// TIA Portal V17 export
// export: Created 2025-03-13T10:29:33.9206583Z, ExportSetting WithDefaults, DisplayName Totally Integrated Automation Portal, DisplayVersion V17 Update 8, DisplayName TIA Portal Openness, DisplayVersion V17 Update 8, DisplayName TIA Portal Version Control Interface, DisplayVersion V17, DisplayName SINAMICS Startdrive Advanced, DisplayVersion V17 SP2, DisplayName SINAMICS Startdrive G110M, G120, G120C, G120D, G120P, G115D, DisplayVersion V17 SP2, DisplayName SINAMICS Startdrive G130, G150, S120, S150, SINAMICS MV, S210, DisplayVersion V17 SP2, DisplayName STEP 7 Professional, DisplayVersion V17 Update 8, DisplayName SINUMERIK ONE STEP 7 Toolbox, DisplayVersion V17 Update 12, DisplayName SINUMERIK 840D sl STEP 7 Toolbox, DisplayVersion V17 Update 12, DisplayName STEP 7 Safety, DisplayVersion V17 Update 6, DisplayName WinCC Advanced, DisplayVersion V17 Update 8
FUNCTION_BLOCK "FB1013_SAFETY_CLADDING"   // FB1013, F_LAD
{ S7_Optimized_Access := 'TRUE' }
AUTHOR : ETXETAR
VERSION : 1.0
// stored: AutoNumber false, IsIECCheckEnabled false, UDAEnableTagReadback false
   VAR
      F_IEC_Timer_PWR_EN_DEL_2 : TOF;
      F_IEC_Timer_PWR_EN_DEL_3 : TOF;
      F_IEC_Timer_PWR_EN_DEL_4 : TOF;
      F_IEC_Timer_PWR_EN_RES_DEL : TON;
      F_IEC_Timer_PWR_EN_FDBCK : TON;
      F_IEC_Timer_GNTR_DR_FDBCK : TON;
      F_IEC_Timer_FIXT_WRK_COND_FDBCK : TON;
      F_IEC_Timer_MACHINE_E_STOP : TON;
      F_IEC_Timer_CLNT_OFF_01R : TOF;
      F_IEC_Timer_CLNT_OFF_01L : TOF;
      F_IEC_Timer_BIMANUAL_CLOSE : TON;
   END_VAR
   // F_IEC_Timer_PWR_EN_FDBCK.PT := T#30ms;
   // F_IEC_Timer_GNTR_DR_FDBCK.PT := T#30ms;
   // F_IEC_Timer_FIXT_WRK_COND_FDBCK.PT := T#30ms;
   // F_IEC_Timer_MACHINE_E_STOP.PT := T#30ms;
   // F_IEC_Timer_BIMANUAL_CLOSE.PT := T#30ms;
BEGIN

REGION Network 1: *************** EMERGENCY STOP ***************
END_REGION

REGION Network 2: FB E-STOP
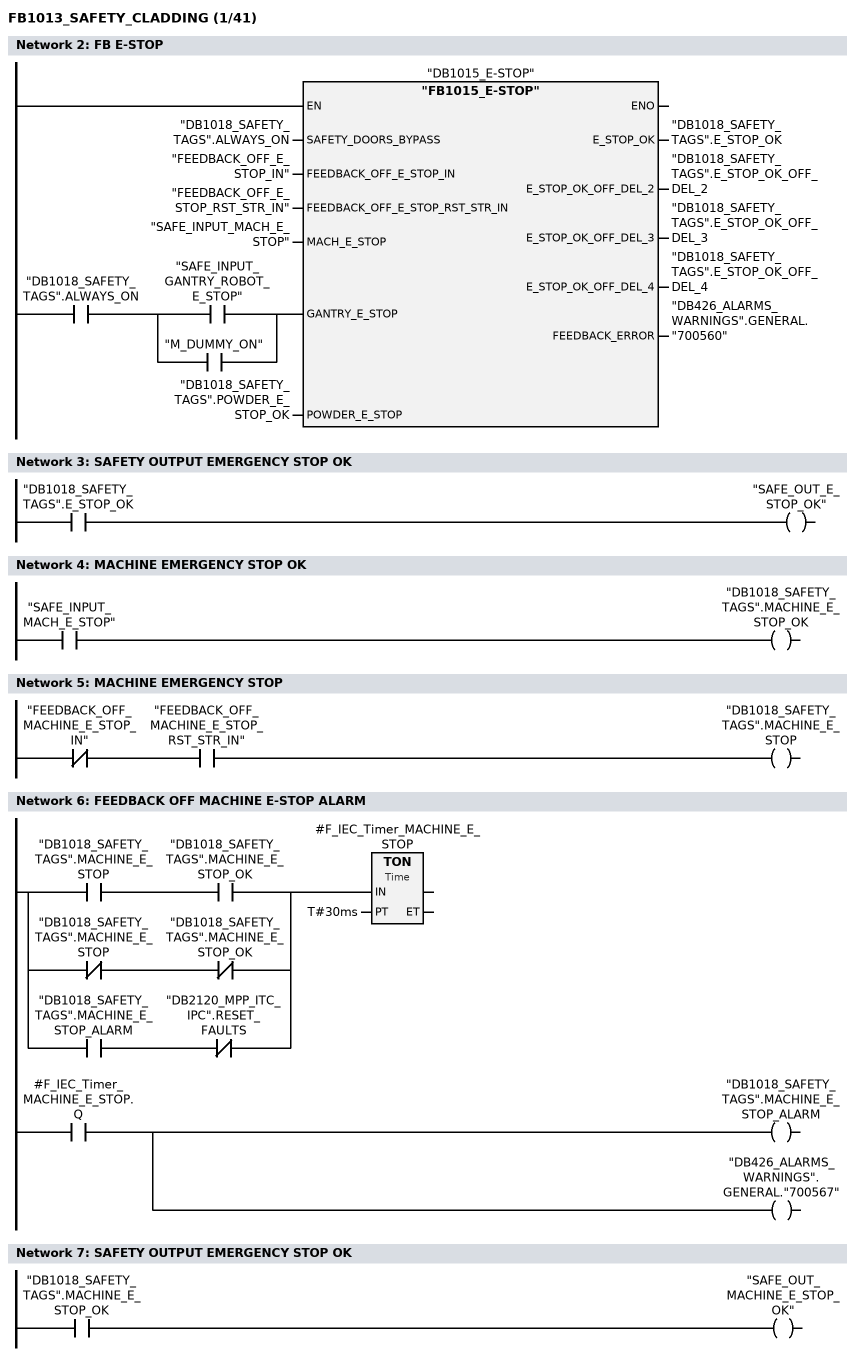
   RUNG wire#powerrail
      "DB1015_E-STOP"(GANTRY_E_STOP := wire#w2, SAFETY_DOORS_BYPASS := "DB1018_SAFETY_TAGS".ALWAYS_ON, FEEDBACK_OFF_E_STOP_IN := "FEEDBACK_OFF_E_STOP_IN", FEEDBACK_OFF_E_STOP_RST_STR_IN := "FEEDBACK_OFF_E_STOP_RST_STR_IN", MACH_E_STOP := "SAFE_INPUT_MACH_E_STOP", POWDER_E_STOP := "DB1018_SAFETY_TAGS".POWDER_E_STOP_OK, E_STOP_OK => "DB1018_SAFETY_TAGS".E_STOP_OK, E_STOP_OK_OFF_DEL_2 => "DB1018_SAFETY_TAGS".E_STOP_OK_OFF_DEL_2, E_STOP_OK_OFF_DEL_3 => "DB1018_SAFETY_TAGS".E_STOP_OK_OFF_DEL_3, E_STOP_OK_OFF_DEL_4 => "DB1018_SAFETY_TAGS".E_STOP_OK_OFF_DEL_4, FEEDBACK_ERROR => "DB426_ALARMS_WARNINGS".GENERAL."700560")
   END_RUNG
   RUNG wire#powerrail
      Contact( "DB1018_SAFETY_TAGS".ALWAYS_ON )
      wire#w1
      Contact( "SAFE_INPUT_GANTRY_ROBOT_E_STOP" )
   END_RUNG wire#w2
   RUNG wire#w1
      Contact( "M_DUMMY_ON" )
   END_RUNG wire#w2
   // the same network as SCL:
   "DB1015_E-STOP"(SAFETY_DOORS_BYPASS := "DB1018_SAFETY_TAGS".ALWAYS_ON,   // "FB1015_E-STOP"
                   FEEDBACK_OFF_E_STOP_IN := "FEEDBACK_OFF_E_STOP_IN",
                   FEEDBACK_OFF_E_STOP_RST_STR_IN := "FEEDBACK_OFF_E_STOP_RST_STR_IN",
                   MACH_E_STOP := "SAFE_INPUT_MACH_E_STOP",
                   GANTRY_E_STOP := "DB1018_SAFETY_TAGS".ALWAYS_ON AND ("SAFE_INPUT_GANTRY_ROBOT_E_STOP" OR "M_DUMMY_ON"),
                   POWDER_E_STOP := "DB1018_SAFETY_TAGS".POWDER_E_STOP_OK,
                   E_STOP_OK => "DB1018_SAFETY_TAGS".E_STOP_OK,
                   E_STOP_OK_OFF_DEL_2 => "DB1018_SAFETY_TAGS".E_STOP_OK_OFF_DEL_2,
                   E_STOP_OK_OFF_DEL_3 => "DB1018_SAFETY_TAGS".E_STOP_OK_OFF_DEL_3,
                   E_STOP_OK_OFF_DEL_4 => "DB1018_SAFETY_TAGS".E_STOP_OK_OFF_DEL_4,
                   FEEDBACK_ERROR => "DB426_ALARMS_WARNINGS".GENERAL."700560");
END_REGION

REGION Network 3: SAFETY OUTPUT EMERGENCY STOP OK
   RUNG wire#powerrail
      Contact( "DB1018_SAFETY_TAGS".E_STOP_OK )
      Coil( "SAFE_OUT_E_STOP_OK" )
   END_RUNG
   // the same network as SCL:
   "SAFE_OUT_E_STOP_OK" := "DB1018_SAFETY_TAGS".E_STOP_OK;
END_REGION

REGION Network 4: MACHINE EMERGENCY STOP OK
   RUNG wire#powerrail
      Contact( "SAFE_INPUT_MACH_E_STOP" )
      Coil( "DB1018_SAFETY_TAGS".MACHINE_E_STOP_OK )
   END_RUNG
   // the same network as SCL:
   "DB1018_SAFETY_TAGS".MACHINE_E_STOP_OK := "SAFE_INPUT_MACH_E_STOP";
END_REGION

REGION Network 5: MACHINE EMERGENCY STOP
   RUNG wire#powerrail
      I_Contact( "FEEDBACK_OFF_MACHINE_E_STOP_IN" )
      Contact( "FEEDBACK_OFF_MACHINE_E_STOP_RST_STR_IN" )
      Coil( "DB1018_SAFETY_TAGS".MACHINE_E_STOP )
   END_RUNG
   // the same network as SCL:
   "DB1018_SAFETY_TAGS".MACHINE_E_STOP := NOT "FEEDBACK_OFF_MACHINE_E_STOP_IN" AND "FEEDBACK_OFF_MACHINE_E_STOP_RST_STR_IN";
END_REGION

REGION Network 6: FEEDBACK OFF MACHINE E-STOP ALARM
   RUNG wire#powerrail
      Contact( "DB1018_SAFETY_TAGS".MACHINE_E_STOP )
      Contact( "DB1018_SAFETY_TAGS".MACHINE_E_STOP_OK )
      wire#w1
      { S7_Templates := "[time_type := Time, codedbool_type := DInt]" } #F_IEC_Timer_MACHINE_E_STOP.TON(pt := T#30ms, et =>)
   END_RUNG
   RUNG wire#powerrail
      I_Contact( "DB1018_SAFETY_TAGS".MACHINE_E_STOP )
      I_Contact( "DB1018_SAFETY_TAGS".MACHINE_E_STOP_OK )
   END_RUNG wire#w1
   RUNG wire#powerrail
      Contact( "DB1018_SAFETY_TAGS".MACHINE_E_STOP_ALARM )
      I_Contact( "DB2120_MPP_ITC_IPC".RESET_FAULTS )
   END_RUNG wire#w1
   RUNG wire#powerrail
      Contact( #F_IEC_Timer_MACHINE_E_STOP.Q )
      wire#w2
      Coil( "DB1018_SAFETY_TAGS".MACHINE_E_STOP_ALARM )
   END_RUNG
   RUNG wire#w2
      Coil( "DB426_ALARMS_WARNINGS".GENERAL."700567" )
   END_RUNG
   // the same network as SCL:
   #F_IEC_Timer_MACHINE_E_STOP.TON(IN := ("DB1018_SAFETY_TAGS".MACHINE_E_STOP AND "DB1018_SAFETY_TAGS".MACHINE_E_STOP_OK) OR (NOT "DB1018_SAFETY_TAGS".MACHINE_E_STOP AND NOT "DB1018_SAFETY_TAGS".MACHINE_E_STOP_OK) OR ("DB1018_SAFETY_TAGS".MACHINE_E_STOP_ALARM AND NOT "DB2120_MPP_ITC_IPC".RESET_FAULTS),
                           PT := T#30ms);
   "DB1018_SAFETY_TAGS".MACHINE_E_STOP_ALARM := #F_IEC_Timer_MACHINE_E_STOP.Q;
   "DB426_ALARMS_WARNINGS".GENERAL."700567" := #F_IEC_Timer_MACHINE_E_STOP.Q;
END_REGION

REGION Network 7: SAFETY OUTPUT EMERGENCY STOP OK
   RUNG wire#powerrail
      Contact( "DB1018_SAFETY_TAGS".MACHINE_E_STOP_OK )
      Coil( "SAFE_OUT_MACHINE_E_STOP_OK" )
   END_RUNG
   // the same network as SCL:
   "SAFE_OUT_MACHINE_E_STOP_OK" := "DB1018_SAFETY_TAGS".MACHINE_E_STOP_OK;
END_REGION

REGION Network 8: *************** SAFETY DOORS UNIT 01 ***************
END_REGION

REGION Network 9: FB SAFETY DOORS MACHINE UNIT 01
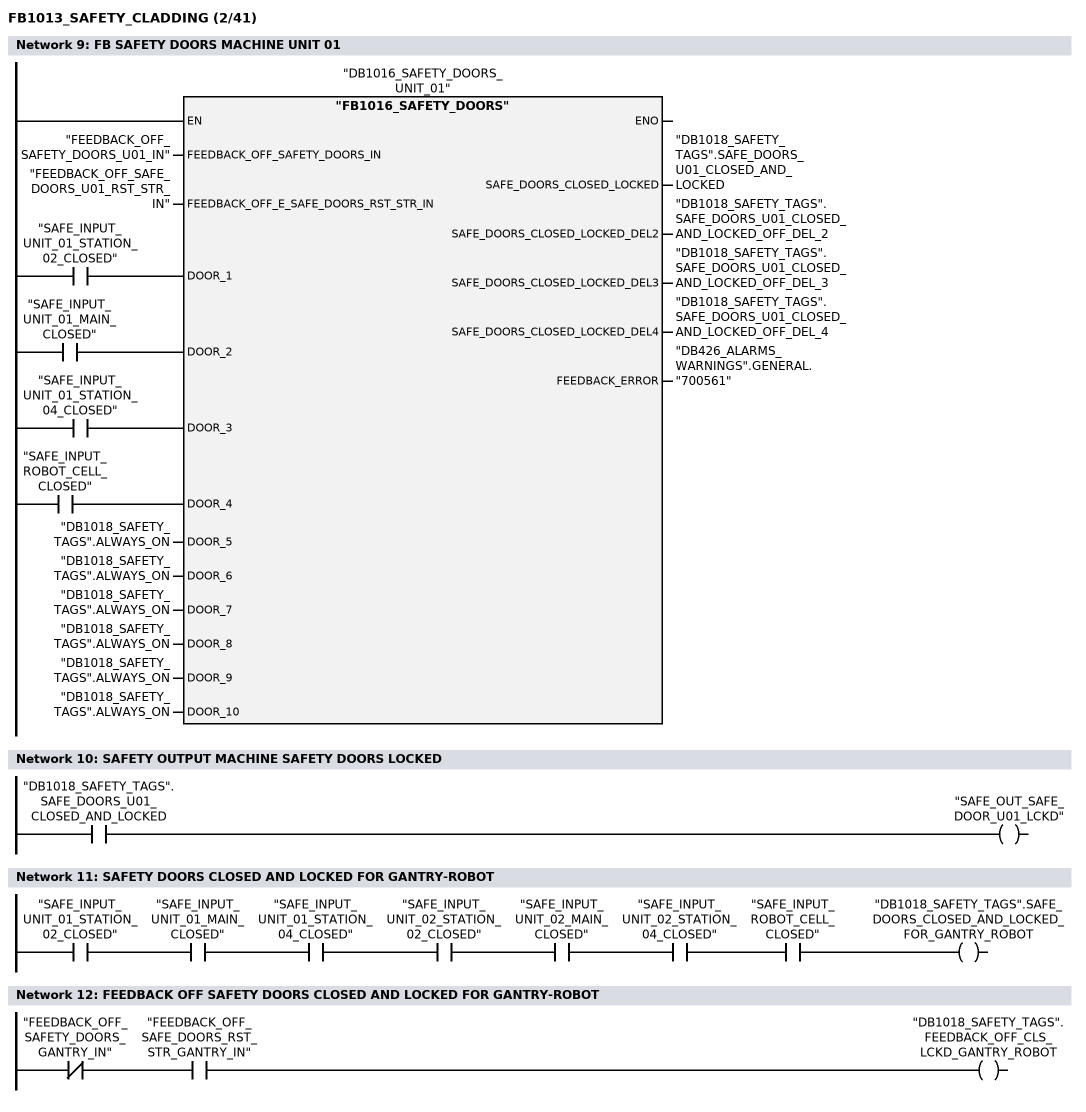
   RUNG wire#powerrail
      "DB1016_SAFETY_DOORS_UNIT_01"(DOOR_1 := wire#w1, DOOR_2 := wire#w2, DOOR_3 := wire#w3, DOOR_4 := wire#w4, FEEDBACK_OFF_SAFETY_DOORS_IN := "FEEDBACK_OFF_SAFETY_DOORS_U01_IN", FEEDBACK_OFF_E_SAFE_DOORS_RST_STR_IN := "FEEDBACK_OFF_SAFE_DOORS_U01_RST_STR_IN", DOOR_5 := "DB1018_SAFETY_TAGS".ALWAYS_ON, DOOR_6 := "DB1018_SAFETY_TAGS".ALWAYS_ON, DOOR_7 := "DB1018_SAFETY_TAGS".ALWAYS_ON, DOOR_8 := "DB1018_SAFETY_TAGS".ALWAYS_ON, DOOR_9 := "DB1018_SAFETY_TAGS".ALWAYS_ON, DOOR_10 := "DB1018_SAFETY_TAGS".ALWAYS_ON, SAFE_DOORS_CLOSED_LOCKED => "DB1018_SAFETY_TAGS".SAFE_DOORS_U01_CLOSED_AND_LOCKED, SAFE_DOORS_CLOSED_LOCKED_DEL2 => "DB1018_SAFETY_TAGS".SAFE_DOORS_U01_CLOSED_AND_LOCKED_OFF_DEL_2, SAFE_DOORS_CLOSED_LOCKED_DEL3 => "DB1018_SAFETY_TAGS".SAFE_DOORS_U01_CLOSED_AND_LOCKED_OFF_DEL_3, SAFE_DOORS_CLOSED_LOCKED_DEL4 => "DB1018_SAFETY_TAGS".SAFE_DOORS_U01_CLOSED_AND_LOCKED_OFF_DEL_4, FEEDBACK_ERROR => "DB426_ALARMS_WARNINGS".GENERAL."700561")
   END_RUNG
   RUNG wire#powerrail
      Contact( "SAFE_INPUT_UNIT_01_STATION_02_CLOSED" )
   END_RUNG wire#w1
   RUNG wire#powerrail
      Contact( "SAFE_INPUT_UNIT_01_MAIN_CLOSED" )
   END_RUNG wire#w2
   RUNG wire#powerrail
      Contact( "SAFE_INPUT_UNIT_01_STATION_04_CLOSED" )
   END_RUNG wire#w3
   RUNG wire#powerrail
      Contact( "SAFE_INPUT_ROBOT_CELL_CLOSED" )
   END_RUNG wire#w4
   // the same network as SCL:
   "DB1016_SAFETY_DOORS_UNIT_01"(FEEDBACK_OFF_SAFETY_DOORS_IN := "FEEDBACK_OFF_SAFETY_DOORS_U01_IN",   // "FB1016_SAFETY_DOORS"
                           FEEDBACK_OFF_E_SAFE_DOORS_RST_STR_IN := "FEEDBACK_OFF_SAFE_DOORS_U01_RST_STR_IN",
                           DOOR_1 := "SAFE_INPUT_UNIT_01_STATION_02_CLOSED",
                           DOOR_2 := "SAFE_INPUT_UNIT_01_MAIN_CLOSED",
                           DOOR_3 := "SAFE_INPUT_UNIT_01_STATION_04_CLOSED",
                           DOOR_4 := "SAFE_INPUT_ROBOT_CELL_CLOSED",
                           DOOR_5 := "DB1018_SAFETY_TAGS".ALWAYS_ON,
                           DOOR_6 := "DB1018_SAFETY_TAGS".ALWAYS_ON,
                           DOOR_7 := "DB1018_SAFETY_TAGS".ALWAYS_ON,
                           DOOR_8 := "DB1018_SAFETY_TAGS".ALWAYS_ON,
                           DOOR_9 := "DB1018_SAFETY_TAGS".ALWAYS_ON,
                           DOOR_10 := "DB1018_SAFETY_TAGS".ALWAYS_ON,
                           SAFE_DOORS_CLOSED_LOCKED => "DB1018_SAFETY_TAGS".SAFE_DOORS_U01_CLOSED_AND_LOCKED,
                           SAFE_DOORS_CLOSED_LOCKED_DEL2 => "DB1018_SAFETY_TAGS".SAFE_DOORS_U01_CLOSED_AND_LOCKED_OFF_DEL_2,
                           SAFE_DOORS_CLOSED_LOCKED_DEL3 => "DB1018_SAFETY_TAGS".SAFE_DOORS_U01_CLOSED_AND_LOCKED_OFF_DEL_3,
                           SAFE_DOORS_CLOSED_LOCKED_DEL4 => "DB1018_SAFETY_TAGS".SAFE_DOORS_U01_CLOSED_AND_LOCKED_OFF_DEL_4,
                           FEEDBACK_ERROR => "DB426_ALARMS_WARNINGS".GENERAL."700561");
END_REGION

REGION Network 10: SAFETY OUTPUT MACHINE SAFETY DOORS LOCKED
   RUNG wire#powerrail
      Contact( "DB1018_SAFETY_TAGS".SAFE_DOORS_U01_CLOSED_AND_LOCKED )
      Coil( "SAFE_OUT_SAFE_DOOR_U01_LCKD" )
   END_RUNG
   // the same network as SCL:
   "SAFE_OUT_SAFE_DOOR_U01_LCKD" := "DB1018_SAFETY_TAGS".SAFE_DOORS_U01_CLOSED_AND_LOCKED;
END_REGION

REGION Network 11: SAFETY DOORS CLOSED AND LOCKED FOR GANTRY-ROBOT
   RUNG wire#powerrail
      Contact( "SAFE_INPUT_UNIT_01_STATION_02_CLOSED" )
      Contact( "SAFE_INPUT_UNIT_01_MAIN_CLOSED" )
      Contact( "SAFE_INPUT_UNIT_01_STATION_04_CLOSED" )
      Contact( "SAFE_INPUT_UNIT_02_STATION_02_CLOSED" )
      Contact( "SAFE_INPUT_UNIT_02_MAIN_CLOSED" )
      Contact( "SAFE_INPUT_UNIT_02_STATION_04_CLOSED" )
      Contact( "SAFE_INPUT_ROBOT_CELL_CLOSED" )
      Coil( "DB1018_SAFETY_TAGS".SAFE_DOORS_CLOSED_AND_LOCKED_FOR_GANTRY_ROBOT )
   END_RUNG
   // the same network as SCL:
   "DB1018_SAFETY_TAGS".SAFE_DOORS_CLOSED_AND_LOCKED_FOR_GANTRY_ROBOT := "SAFE_INPUT_UNIT_01_STATION_02_CLOSED" AND "SAFE_INPUT_UNIT_01_MAIN_CLOSED" AND "SAFE_INPUT_UNIT_01_STATION_04_CLOSED" AND "SAFE_INPUT_UNIT_02_STATION_02_CLOSED" AND "SAFE_INPUT_UNIT_02_MAIN_CLOSED" AND "SAFE_INPUT_UNIT_02_STATION_04_CLOSED" AND "SAFE_INPUT_ROBOT_CELL_CLOSED";
END_REGION

REGION Network 12: FEEDBACK OFF SAFETY DOORS CLOSED AND LOCKED FOR GANTRY-ROBOT
   RUNG wire#powerrail
      I_Contact( "FEEDBACK_OFF_SAFETY_DOORS_GANTRY_IN" )
      Contact( "FEEDBACK_OFF_SAFE_DOORS_RST_STR_GANTRY_IN" )
      Coil( "DB1018_SAFETY_TAGS".FEEDBACK_OFF_CLS_LCKD_GANTRY_ROBOT )
   END_RUNG
   // the same network as SCL:
   "DB1018_SAFETY_TAGS".FEEDBACK_OFF_CLS_LCKD_GANTRY_ROBOT := NOT "FEEDBACK_OFF_SAFETY_DOORS_GANTRY_IN" AND "FEEDBACK_OFF_SAFE_DOORS_RST_STR_GANTRY_IN";
END_REGION

REGION Network 13: FEEDBACK OFF SAFETY DOORS CLOSED AND LOCKED FOR GANTRY-ROBOT ALARM
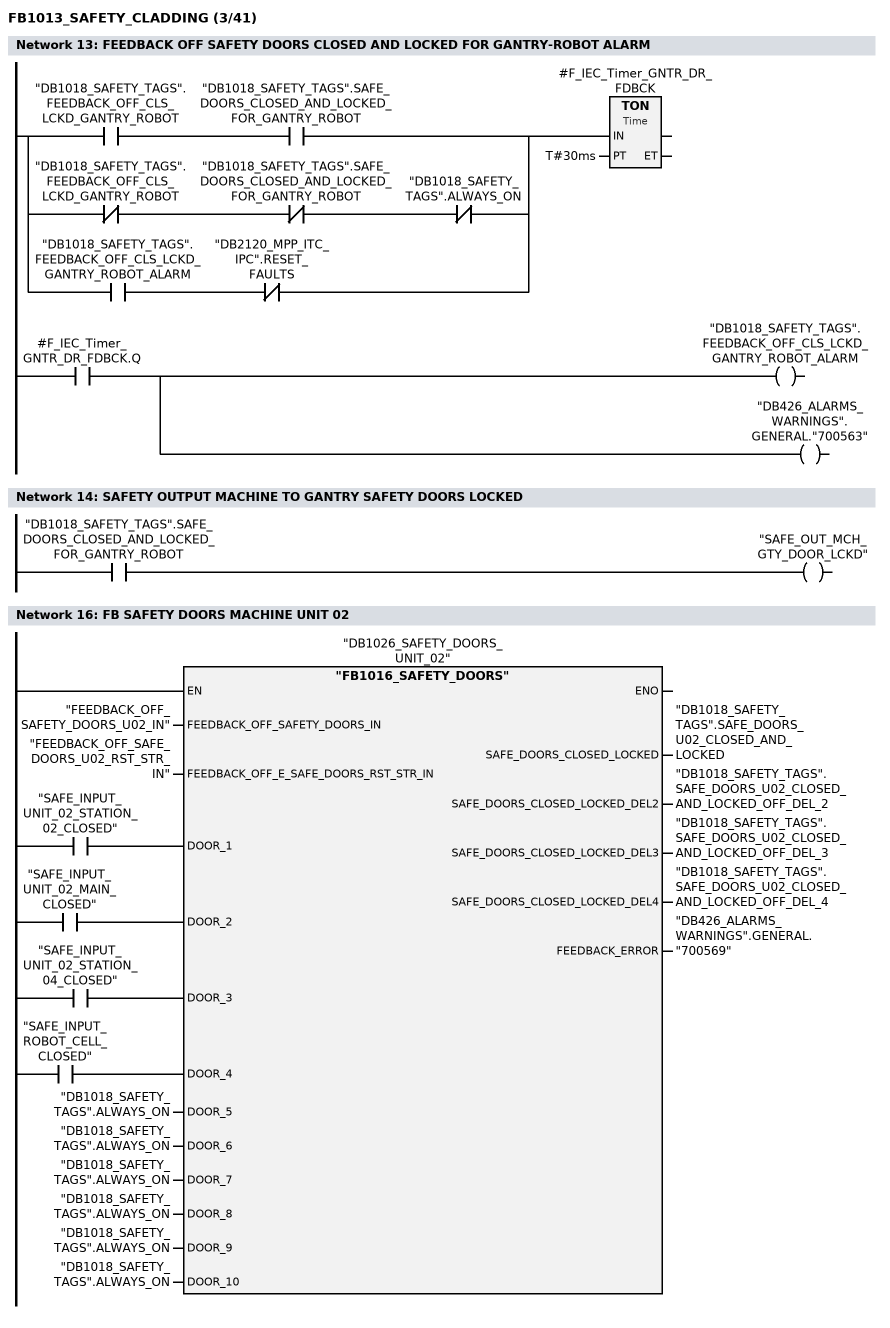
   RUNG wire#powerrail
      Contact( "DB1018_SAFETY_TAGS".FEEDBACK_OFF_CLS_LCKD_GANTRY_ROBOT )
      Contact( "DB1018_SAFETY_TAGS".SAFE_DOORS_CLOSED_AND_LOCKED_FOR_GANTRY_ROBOT )
      wire#w1
      { S7_Templates := "[time_type := Time, codedbool_type := DInt]" } #F_IEC_Timer_GNTR_DR_FDBCK.TON(pt := T#30ms, et =>)
   END_RUNG
   RUNG wire#powerrail
      I_Contact( "DB1018_SAFETY_TAGS".FEEDBACK_OFF_CLS_LCKD_GANTRY_ROBOT )
      I_Contact( "DB1018_SAFETY_TAGS".SAFE_DOORS_CLOSED_AND_LOCKED_FOR_GANTRY_ROBOT )
      I_Contact( "DB1018_SAFETY_TAGS".ALWAYS_ON )
   END_RUNG wire#w1
   RUNG wire#powerrail
      Contact( "DB1018_SAFETY_TAGS".FEEDBACK_OFF_CLS_LCKD_GANTRY_ROBOT_ALARM )
      I_Contact( "DB2120_MPP_ITC_IPC".RESET_FAULTS )
   END_RUNG wire#w1
   RUNG wire#powerrail
      Contact( #F_IEC_Timer_GNTR_DR_FDBCK.Q )
      wire#w2
      Coil( "DB1018_SAFETY_TAGS".FEEDBACK_OFF_CLS_LCKD_GANTRY_ROBOT_ALARM )
   END_RUNG
   RUNG wire#w2
      Coil( "DB426_ALARMS_WARNINGS".GENERAL."700563" )
   END_RUNG
   // the same network as SCL:
   #F_IEC_Timer_GNTR_DR_FDBCK.TON(IN := ("DB1018_SAFETY_TAGS".FEEDBACK_OFF_CLS_LCKD_GANTRY_ROBOT AND "DB1018_SAFETY_TAGS".SAFE_DOORS_CLOSED_AND_LOCKED_FOR_GANTRY_ROBOT) OR (NOT "DB1018_SAFETY_TAGS".FEEDBACK_OFF_CLS_LCKD_GANTRY_ROBOT AND NOT "DB1018_SAFETY_TAGS".SAFE_DOORS_CLOSED_AND_LOCKED_FOR_GANTRY_ROBOT AND NOT "DB1018_SAFETY_TAGS".ALWAYS_ON) OR ("DB1018_SAFETY_TAGS".FEEDBACK_OFF_CLS_LCKD_GANTRY_ROBOT_ALARM AND NOT "DB2120_MPP_ITC_IPC".RESET_FAULTS),
                           PT := T#30ms);
   "DB1018_SAFETY_TAGS".FEEDBACK_OFF_CLS_LCKD_GANTRY_ROBOT_ALARM := #F_IEC_Timer_GNTR_DR_FDBCK.Q;
   "DB426_ALARMS_WARNINGS".GENERAL."700563" := #F_IEC_Timer_GNTR_DR_FDBCK.Q;
END_REGION

REGION Network 14: SAFETY OUTPUT MACHINE TO GANTRY SAFETY DOORS LOCKED
   RUNG wire#powerrail
      Contact( "DB1018_SAFETY_TAGS".SAFE_DOORS_CLOSED_AND_LOCKED_FOR_GANTRY_ROBOT )
      Coil( "SAFE_OUT_MCH_GTY_DOOR_LCKD" )
   END_RUNG
   // the same network as SCL:
   "SAFE_OUT_MCH_GTY_DOOR_LCKD" := "DB1018_SAFETY_TAGS".SAFE_DOORS_CLOSED_AND_LOCKED_FOR_GANTRY_ROBOT;
END_REGION

REGION Network 15: *************** SAFETY DOORS UNIT 02 ***************
END_REGION

REGION Network 16: FB SAFETY DOORS MACHINE UNIT 02
   RUNG wire#powerrail
      "DB1026_SAFETY_DOORS_UNIT_02"(DOOR_1 := wire#w1, DOOR_2 := wire#w2, DOOR_3 := wire#w3, DOOR_4 := wire#w4, FEEDBACK_OFF_SAFETY_DOORS_IN := "FEEDBACK_OFF_SAFETY_DOORS_U02_IN", FEEDBACK_OFF_E_SAFE_DOORS_RST_STR_IN := "FEEDBACK_OFF_SAFE_DOORS_U02_RST_STR_IN", DOOR_5 := "DB1018_SAFETY_TAGS".ALWAYS_ON, DOOR_6 := "DB1018_SAFETY_TAGS".ALWAYS_ON, DOOR_7 := "DB1018_SAFETY_TAGS".ALWAYS_ON, DOOR_8 := "DB1018_SAFETY_TAGS".ALWAYS_ON, DOOR_9 := "DB1018_SAFETY_TAGS".ALWAYS_ON, DOOR_10 := "DB1018_SAFETY_TAGS".ALWAYS_ON, SAFE_DOORS_CLOSED_LOCKED => "DB1018_SAFETY_TAGS".SAFE_DOORS_U02_CLOSED_AND_LOCKED, SAFE_DOORS_CLOSED_LOCKED_DEL2 => "DB1018_SAFETY_TAGS".SAFE_DOORS_U02_CLOSED_AND_LOCKED_OFF_DEL_2, SAFE_DOORS_CLOSED_LOCKED_DEL3 => "DB1018_SAFETY_TAGS".SAFE_DOORS_U02_CLOSED_AND_LOCKED_OFF_DEL_3, SAFE_DOORS_CLOSED_LOCKED_DEL4 => "DB1018_SAFETY_TAGS".SAFE_DOORS_U02_CLOSED_AND_LOCKED_OFF_DEL_4, FEEDBACK_ERROR => "DB426_ALARMS_WARNINGS".GENERAL."700569")
   END_RUNG
   RUNG wire#powerrail
      Contact( "SAFE_INPUT_UNIT_02_STATION_02_CLOSED" )
   END_RUNG wire#w1
   RUNG wire#powerrail
      Contact( "SAFE_INPUT_UNIT_02_MAIN_CLOSED" )
   END_RUNG wire#w2
   RUNG wire#powerrail
      Contact( "SAFE_INPUT_UNIT_02_STATION_04_CLOSED" )
   END_RUNG wire#w3
   RUNG wire#powerrail
      Contact( "SAFE_INPUT_ROBOT_CELL_CLOSED" )
   END_RUNG wire#w4
   // the same network as SCL:
   "DB1026_SAFETY_DOORS_UNIT_02"(FEEDBACK_OFF_SAFETY_DOORS_IN := "FEEDBACK_OFF_SAFETY_DOORS_U02_IN",   // "FB1016_SAFETY_DOORS"
                           FEEDBACK_OFF_E_SAFE_DOORS_RST_STR_IN := "FEEDBACK_OFF_SAFE_DOORS_U02_RST_STR_IN",
                           DOOR_1 := "SAFE_INPUT_UNIT_02_STATION_02_CLOSED",
                           DOOR_2 := "SAFE_INPUT_UNIT_02_MAIN_CLOSED",
                           DOOR_3 := "SAFE_INPUT_UNIT_02_STATION_04_CLOSED",
                           DOOR_4 := "SAFE_INPUT_ROBOT_CELL_CLOSED",
                           DOOR_5 := "DB1018_SAFETY_TAGS".ALWAYS_ON,
                           DOOR_6 := "DB1018_SAFETY_TAGS".ALWAYS_ON,
                           DOOR_7 := "DB1018_SAFETY_TAGS".ALWAYS_ON,
                           DOOR_8 := "DB1018_SAFETY_TAGS".ALWAYS_ON,
                           DOOR_9 := "DB1018_SAFETY_TAGS".ALWAYS_ON,
                           DOOR_10 := "DB1018_SAFETY_TAGS".ALWAYS_ON,
                           SAFE_DOORS_CLOSED_LOCKED => "DB1018_SAFETY_TAGS".SAFE_DOORS_U02_CLOSED_AND_LOCKED,
                           SAFE_DOORS_CLOSED_LOCKED_DEL2 => "DB1018_SAFETY_TAGS".SAFE_DOORS_U02_CLOSED_AND_LOCKED_OFF_DEL_2,
                           SAFE_DOORS_CLOSED_LOCKED_DEL3 => "DB1018_SAFETY_TAGS".SAFE_DOORS_U02_CLOSED_AND_LOCKED_OFF_DEL_3,
                           SAFE_DOORS_CLOSED_LOCKED_DEL4 => "DB1018_SAFETY_TAGS".SAFE_DOORS_U02_CLOSED_AND_LOCKED_OFF_DEL_4,
                           FEEDBACK_ERROR => "DB426_ALARMS_WARNINGS".GENERAL."700569");
END_REGION

REGION Network 17: SAFETY OUTPUT MACHINE SAFETY DOORS LOCKED
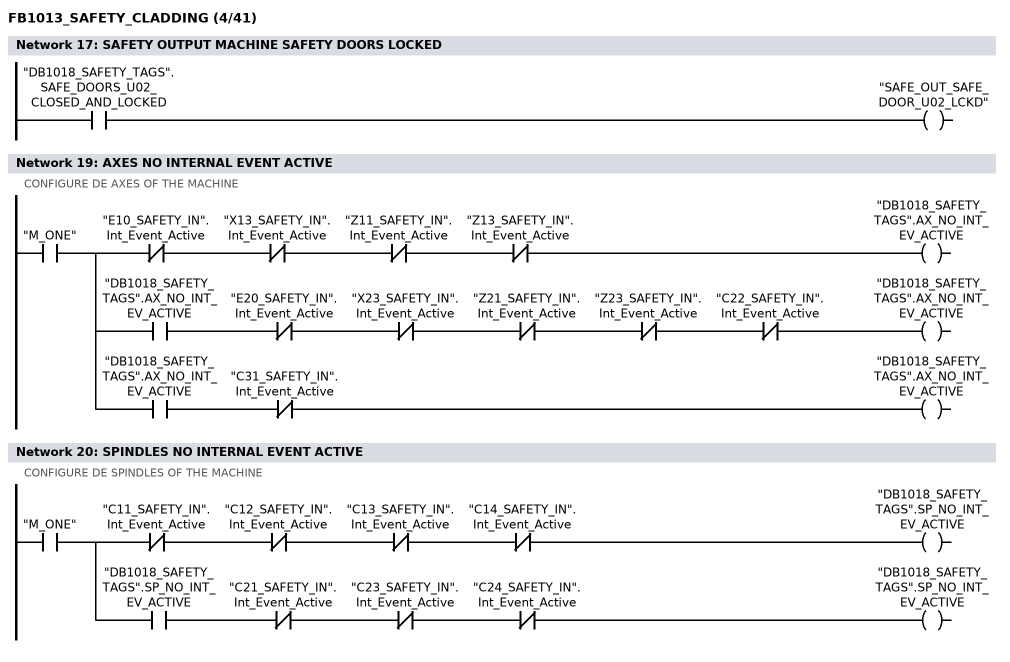
   RUNG wire#powerrail
      Contact( "DB1018_SAFETY_TAGS".SAFE_DOORS_U02_CLOSED_AND_LOCKED )
      Coil( "SAFE_OUT_SAFE_DOOR_U02_LCKD" )
   END_RUNG
   // the same network as SCL:
   "SAFE_OUT_SAFE_DOOR_U02_LCKD" := "DB1018_SAFETY_TAGS".SAFE_DOORS_U02_CLOSED_AND_LOCKED;
END_REGION

REGION Network 18: *************** SPINDLES AND AXES ***************
END_REGION

REGION Network 19: AXES NO INTERNAL EVENT ACTIVE
   // CONFIGURE DE AXES OF THE MACHINE
   RUNG wire#powerrail
      Contact( "M_ONE" )
      wire#w1
      I_Contact( "E10_SAFETY_IN".Int_Event_Active )
      I_Contact( "X13_SAFETY_IN".Int_Event_Active )
      I_Contact( "Z11_SAFETY_IN".Int_Event_Active )
      I_Contact( "Z13_SAFETY_IN".Int_Event_Active )
      Coil( "DB1018_SAFETY_TAGS".AX_NO_INT_EV_ACTIVE )
   END_RUNG
   RUNG wire#w1
      Contact( "DB1018_SAFETY_TAGS".AX_NO_INT_EV_ACTIVE )
      I_Contact( "E20_SAFETY_IN".Int_Event_Active )
      I_Contact( "X23_SAFETY_IN".Int_Event_Active )
      I_Contact( "Z21_SAFETY_IN".Int_Event_Active )
      I_Contact( "Z23_SAFETY_IN".Int_Event_Active )
      I_Contact( "C22_SAFETY_IN".Int_Event_Active )
      Coil( "DB1018_SAFETY_TAGS".AX_NO_INT_EV_ACTIVE )
   END_RUNG
   RUNG wire#w1
      Contact( "DB1018_SAFETY_TAGS".AX_NO_INT_EV_ACTIVE )
      I_Contact( "C31_SAFETY_IN".Int_Event_Active )
      Coil( "DB1018_SAFETY_TAGS".AX_NO_INT_EV_ACTIVE )
   END_RUNG
   // the same network as SCL:
   "DB1018_SAFETY_TAGS".AX_NO_INT_EV_ACTIVE := "M_ONE" AND NOT "E10_SAFETY_IN".Int_Event_Active AND NOT "X13_SAFETY_IN".Int_Event_Active AND NOT "Z11_SAFETY_IN".Int_Event_Active AND NOT "Z13_SAFETY_IN".Int_Event_Active;
   "DB1018_SAFETY_TAGS".AX_NO_INT_EV_ACTIVE := "M_ONE" AND "DB1018_SAFETY_TAGS".AX_NO_INT_EV_ACTIVE AND NOT "E20_SAFETY_IN".Int_Event_Active AND NOT "X23_SAFETY_IN".Int_Event_Active AND NOT "Z21_SAFETY_IN".Int_Event_Active AND NOT "Z23_SAFETY_IN".Int_Event_Active AND NOT "C22_SAFETY_IN".Int_Event_Active;
   "DB1018_SAFETY_TAGS".AX_NO_INT_EV_ACTIVE := "M_ONE" AND "DB1018_SAFETY_TAGS".AX_NO_INT_EV_ACTIVE AND NOT "C31_SAFETY_IN".Int_Event_Active;
END_REGION

REGION Network 20: SPINDLES NO INTERNAL EVENT ACTIVE
   // CONFIGURE DE SPINDLES OF THE MACHINE
   RUNG wire#powerrail
      Contact( "M_ONE" )
      wire#w1
      I_Contact( "C11_SAFETY_IN".Int_Event_Active )
      I_Contact( "C12_SAFETY_IN".Int_Event_Active )
      I_Contact( "C13_SAFETY_IN".Int_Event_Active )
      I_Contact( "C14_SAFETY_IN".Int_Event_Active )
      Coil( "DB1018_SAFETY_TAGS".SP_NO_INT_EV_ACTIVE )
   END_RUNG
   RUNG wire#w1
      Contact( "DB1018_SAFETY_TAGS".SP_NO_INT_EV_ACTIVE )
      I_Contact( "C21_SAFETY_IN".Int_Event_Active )
      I_Contact( "C23_SAFETY_IN".Int_Event_Active )
      I_Contact( "C24_SAFETY_IN".Int_Event_Active )
      Coil( "DB1018_SAFETY_TAGS".SP_NO_INT_EV_ACTIVE )
   END_RUNG
   // the same network as SCL:
   "DB1018_SAFETY_TAGS".SP_NO_INT_EV_ACTIVE := "M_ONE" AND NOT "C11_SAFETY_IN".Int_Event_Active AND NOT "C12_SAFETY_IN".Int_Event_Active AND NOT "C13_SAFETY_IN".Int_Event_Active AND NOT "C14_SAFETY_IN".Int_Event_Active;
   "DB1018_SAFETY_TAGS".SP_NO_INT_EV_ACTIVE := "M_ONE" AND "DB1018_SAFETY_TAGS".SP_NO_INT_EV_ACTIVE AND NOT "C21_SAFETY_IN".Int_Event_Active AND NOT "C23_SAFETY_IN".Int_Event_Active AND NOT "C24_SAFETY_IN".Int_Event_Active;
END_REGION

REGION Network 21: ACKNOLEDGE INTERNAL EVENT ACTIVE
   // CONFIGURE DE AXES OF THE MACHINE
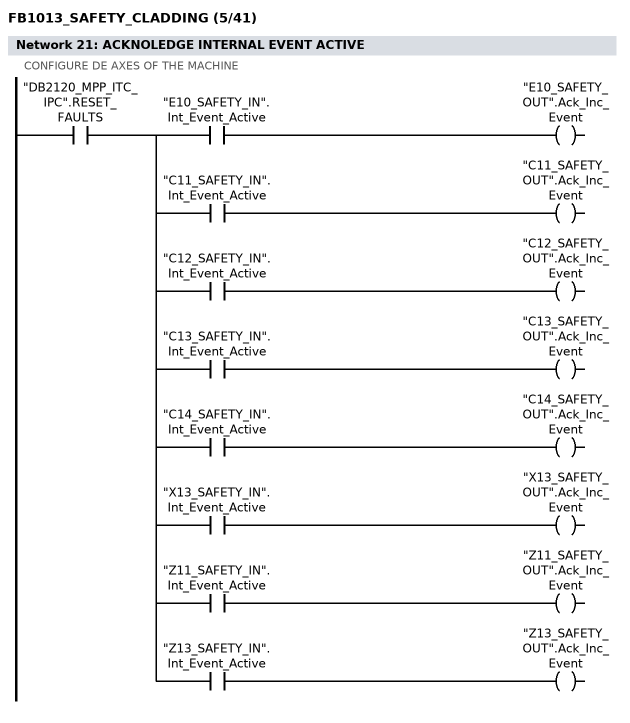
   RUNG wire#powerrail
      Contact( "DB2120_MPP_ITC_IPC".RESET_FAULTS )
      wire#w1
      Contact( "E10_SAFETY_IN".Int_Event_Active )
      Coil( "E10_SAFETY_OUT".Ack_Inc_Event )
   END_RUNG
   RUNG wire#w1
      Contact( "C11_SAFETY_IN".Int_Event_Active )
      Coil( "C11_SAFETY_OUT".Ack_Inc_Event )
   END_RUNG
   RUNG wire#w1
      Contact( "C12_SAFETY_IN".Int_Event_Active )
      Coil( "C12_SAFETY_OUT".Ack_Inc_Event )
   END_RUNG
   RUNG wire#w1
      Contact( "C13_SAFETY_IN".Int_Event_Active )
      Coil( "C13_SAFETY_OUT".Ack_Inc_Event )
   END_RUNG
   RUNG wire#w1
      Contact( "C14_SAFETY_IN".Int_Event_Active )
      Coil( "C14_SAFETY_OUT".Ack_Inc_Event )
   END_RUNG
   RUNG wire#w1
      Contact( "X13_SAFETY_IN".Int_Event_Active )
      Coil( "X13_SAFETY_OUT".Ack_Inc_Event )
   END_RUNG
   RUNG wire#w1
      Contact( "Z11_SAFETY_IN".Int_Event_Active )
      Coil( "Z11_SAFETY_OUT".Ack_Inc_Event )
   END_RUNG
   RUNG wire#w1
      Contact( "Z13_SAFETY_IN".Int_Event_Active )
      Coil( "Z13_SAFETY_OUT".Ack_Inc_Event )
   END_RUNG
   // the same network as SCL:
   "E10_SAFETY_OUT".Ack_Inc_Event := "DB2120_MPP_ITC_IPC".RESET_FAULTS AND "E10_SAFETY_IN".Int_Event_Active;
   "C11_SAFETY_OUT".Ack_Inc_Event := "DB2120_MPP_ITC_IPC".RESET_FAULTS AND "C11_SAFETY_IN".Int_Event_Active;
   "C12_SAFETY_OUT".Ack_Inc_Event := "DB2120_MPP_ITC_IPC".RESET_FAULTS AND "C12_SAFETY_IN".Int_Event_Active;
   "C13_SAFETY_OUT".Ack_Inc_Event := "DB2120_MPP_ITC_IPC".RESET_FAULTS AND "C13_SAFETY_IN".Int_Event_Active;
   "C14_SAFETY_OUT".Ack_Inc_Event := "DB2120_MPP_ITC_IPC".RESET_FAULTS AND "C14_SAFETY_IN".Int_Event_Active;
   "X13_SAFETY_OUT".Ack_Inc_Event := "DB2120_MPP_ITC_IPC".RESET_FAULTS AND "X13_SAFETY_IN".Int_Event_Active;
   "Z11_SAFETY_OUT".Ack_Inc_Event := "DB2120_MPP_ITC_IPC".RESET_FAULTS AND "Z11_SAFETY_IN".Int_Event_Active;
   "Z13_SAFETY_OUT".Ack_Inc_Event := "DB2120_MPP_ITC_IPC".RESET_FAULTS AND "Z13_SAFETY_IN".Int_Event_Active;
END_REGION

REGION Network 22: ACKNOLEDGE INTERNAL EVENT ACTIVE
   // CONFIGURE DE AXES OF THE MACHINE
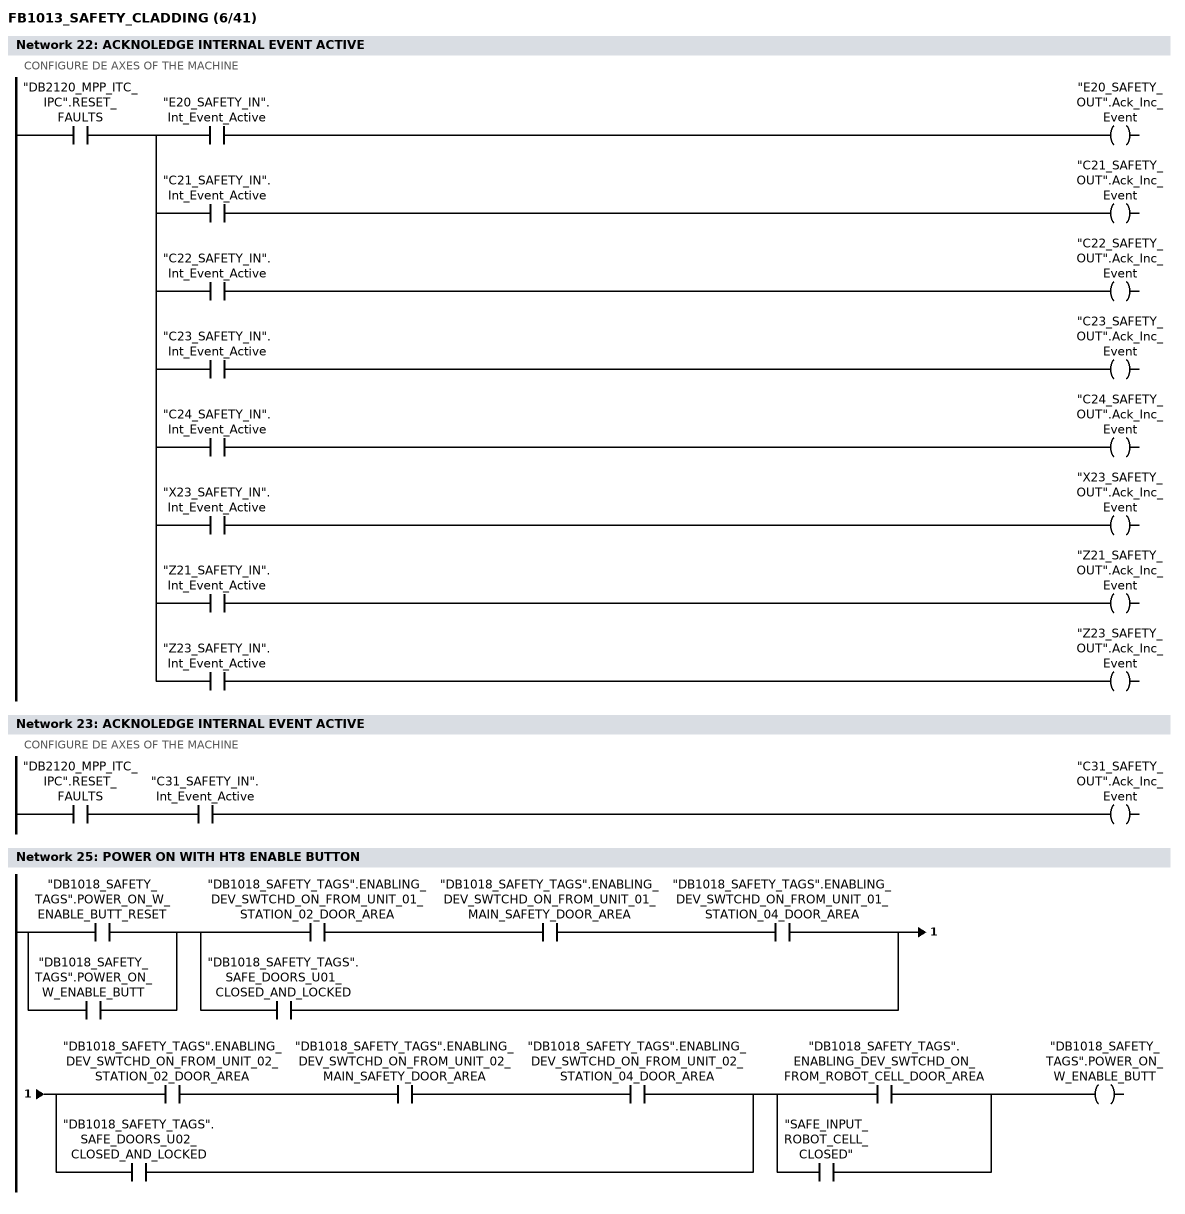
   RUNG wire#powerrail
      Contact( "DB2120_MPP_ITC_IPC".RESET_FAULTS )
      wire#w1
      Contact( "E20_SAFETY_IN".Int_Event_Active )
      Coil( "E20_SAFETY_OUT".Ack_Inc_Event )
   END_RUNG
   RUNG wire#w1
      Contact( "C21_SAFETY_IN".Int_Event_Active )
      Coil( "C21_SAFETY_OUT".Ack_Inc_Event )
   END_RUNG
   RUNG wire#w1
      Contact( "C22_SAFETY_IN".Int_Event_Active )
      Coil( "C22_SAFETY_OUT".Ack_Inc_Event )
   END_RUNG
   RUNG wire#w1
      Contact( "C23_SAFETY_IN".Int_Event_Active )
      Coil( "C23_SAFETY_OUT".Ack_Inc_Event )
   END_RUNG
   RUNG wire#w1
      Contact( "C24_SAFETY_IN".Int_Event_Active )
      Coil( "C24_SAFETY_OUT".Ack_Inc_Event )
   END_RUNG
   RUNG wire#w1
      Contact( "X23_SAFETY_IN".Int_Event_Active )
      Coil( "X23_SAFETY_OUT".Ack_Inc_Event )
   END_RUNG
   RUNG wire#w1
      Contact( "Z21_SAFETY_IN".Int_Event_Active )
      Coil( "Z21_SAFETY_OUT".Ack_Inc_Event )
   END_RUNG
   RUNG wire#w1
      Contact( "Z23_SAFETY_IN".Int_Event_Active )
      Coil( "Z23_SAFETY_OUT".Ack_Inc_Event )
   END_RUNG
   // the same network as SCL:
   "E20_SAFETY_OUT".Ack_Inc_Event := "DB2120_MPP_ITC_IPC".RESET_FAULTS AND "E20_SAFETY_IN".Int_Event_Active;
   "C21_SAFETY_OUT".Ack_Inc_Event := "DB2120_MPP_ITC_IPC".RESET_FAULTS AND "C21_SAFETY_IN".Int_Event_Active;
   "C22_SAFETY_OUT".Ack_Inc_Event := "DB2120_MPP_ITC_IPC".RESET_FAULTS AND "C22_SAFETY_IN".Int_Event_Active;
   "C23_SAFETY_OUT".Ack_Inc_Event := "DB2120_MPP_ITC_IPC".RESET_FAULTS AND "C23_SAFETY_IN".Int_Event_Active;
   "C24_SAFETY_OUT".Ack_Inc_Event := "DB2120_MPP_ITC_IPC".RESET_FAULTS AND "C24_SAFETY_IN".Int_Event_Active;
   "X23_SAFETY_OUT".Ack_Inc_Event := "DB2120_MPP_ITC_IPC".RESET_FAULTS AND "X23_SAFETY_IN".Int_Event_Active;
   "Z21_SAFETY_OUT".Ack_Inc_Event := "DB2120_MPP_ITC_IPC".RESET_FAULTS AND "Z21_SAFETY_IN".Int_Event_Active;
   "Z23_SAFETY_OUT".Ack_Inc_Event := "DB2120_MPP_ITC_IPC".RESET_FAULTS AND "Z23_SAFETY_IN".Int_Event_Active;
END_REGION

REGION Network 23: ACKNOLEDGE INTERNAL EVENT ACTIVE
   // CONFIGURE DE AXES OF THE MACHINE
   RUNG wire#powerrail
      Contact( "DB2120_MPP_ITC_IPC".RESET_FAULTS )
      Contact( "C31_SAFETY_IN".Int_Event_Active )
      Coil( "C31_SAFETY_OUT".Ack_Inc_Event )
   END_RUNG
   // the same network as SCL:
   "C31_SAFETY_OUT".Ack_Inc_Event := "DB2120_MPP_ITC_IPC".RESET_FAULTS AND "C31_SAFETY_IN".Int_Event_Active;
END_REGION

REGION Network 24: *************** POWER ENABLE ***************
END_REGION

REGION Network 25: POWER ON WITH HT8 ENABLE BUTTON
   RUNG wire#powerrail
      Contact( "DB1018_SAFETY_TAGS".POWER_ON_W_ENABLE_BUTT_RESET )
      wire#w1
      Contact( "DB1018_SAFETY_TAGS".ENABLING_DEV_SWTCHD_ON_FROM_UNIT_01_STATION_02_DOOR_AREA )
      Contact( "DB1018_SAFETY_TAGS".ENABLING_DEV_SWTCHD_ON_FROM_UNIT_01_MAIN_SAFETY_DOOR_AREA )
      Contact( "DB1018_SAFETY_TAGS".ENABLING_DEV_SWTCHD_ON_FROM_UNIT_01_STATION_04_DOOR_AREA )
      wire#w2
      Contact( "DB1018_SAFETY_TAGS".ENABLING_DEV_SWTCHD_ON_FROM_UNIT_02_STATION_02_DOOR_AREA )
      Contact( "DB1018_SAFETY_TAGS".ENABLING_DEV_SWTCHD_ON_FROM_UNIT_02_MAIN_SAFETY_DOOR_AREA )
      Contact( "DB1018_SAFETY_TAGS".ENABLING_DEV_SWTCHD_ON_FROM_UNIT_02_STATION_04_DOOR_AREA )
      wire#w3
      Contact( "DB1018_SAFETY_TAGS".ENABLING_DEV_SWTCHD_ON_FROM_ROBOT_CELL_DOOR_AREA )
      wire#w4
      Coil( "DB1018_SAFETY_TAGS".POWER_ON_W_ENABLE_BUTT )
   END_RUNG
   RUNG wire#powerrail
      Contact( "DB1018_SAFETY_TAGS".POWER_ON_W_ENABLE_BUTT )
   END_RUNG wire#w1
   RUNG wire#w1
      Contact( "DB1018_SAFETY_TAGS".SAFE_DOORS_U01_CLOSED_AND_LOCKED )
   END_RUNG wire#w2
   RUNG wire#w2
      Contact( "DB1018_SAFETY_TAGS".SAFE_DOORS_U02_CLOSED_AND_LOCKED )
   END_RUNG wire#w3
   RUNG wire#w3
      Contact( "SAFE_INPUT_ROBOT_CELL_CLOSED" )
   END_RUNG wire#w4
   // the same network as SCL:
   "DB1018_SAFETY_TAGS".POWER_ON_W_ENABLE_BUTT := ("DB1018_SAFETY_TAGS".POWER_ON_W_ENABLE_BUTT_RESET OR "DB1018_SAFETY_TAGS".POWER_ON_W_ENABLE_BUTT) AND (("DB1018_SAFETY_TAGS".ENABLING_DEV_SWTCHD_ON_FROM_UNIT_01_STATION_02_DOOR_AREA AND "DB1018_SAFETY_TAGS".ENABLING_DEV_SWTCHD_ON_FROM_UNIT_01_MAIN_SAFETY_DOOR_AREA AND "DB1018_SAFETY_TAGS".ENABLING_DEV_SWTCHD_ON_FROM_UNIT_01_STATION_04_DOOR_AREA) OR "DB1018_SAFETY_TAGS".SAFE_DOORS_U01_CLOSED_AND_LOCKED) AND (("DB1018_SAFETY_TAGS".ENABLING_DEV_SWTCHD_ON_FROM_UNIT_02_STATION_02_DOOR_AREA AND "DB1018_SAFETY_TAGS".ENABLING_DEV_SWTCHD_ON_FROM_UNIT_02_MAIN_SAFETY_DOOR_AREA AND "DB1018_SAFETY_TAGS".ENABLING_DEV_SWTCHD_ON_FROM_UNIT_02_STATION_04_DOOR_AREA) OR "DB1018_SAFETY_TAGS".SAFE_DOORS_U02_CLOSED_AND_LOCKED) AND ("DB1018_SAFETY_TAGS".ENABLING_DEV_SWTCHD_ON_FROM_ROBOT_CELL_DOOR_AREA OR "SAFE_INPUT_ROBOT_CELL_CLOSED");
END_REGION

REGION Network 26: POWER ON WITH HT8 ENABLE BUTTON OFF DELAYED
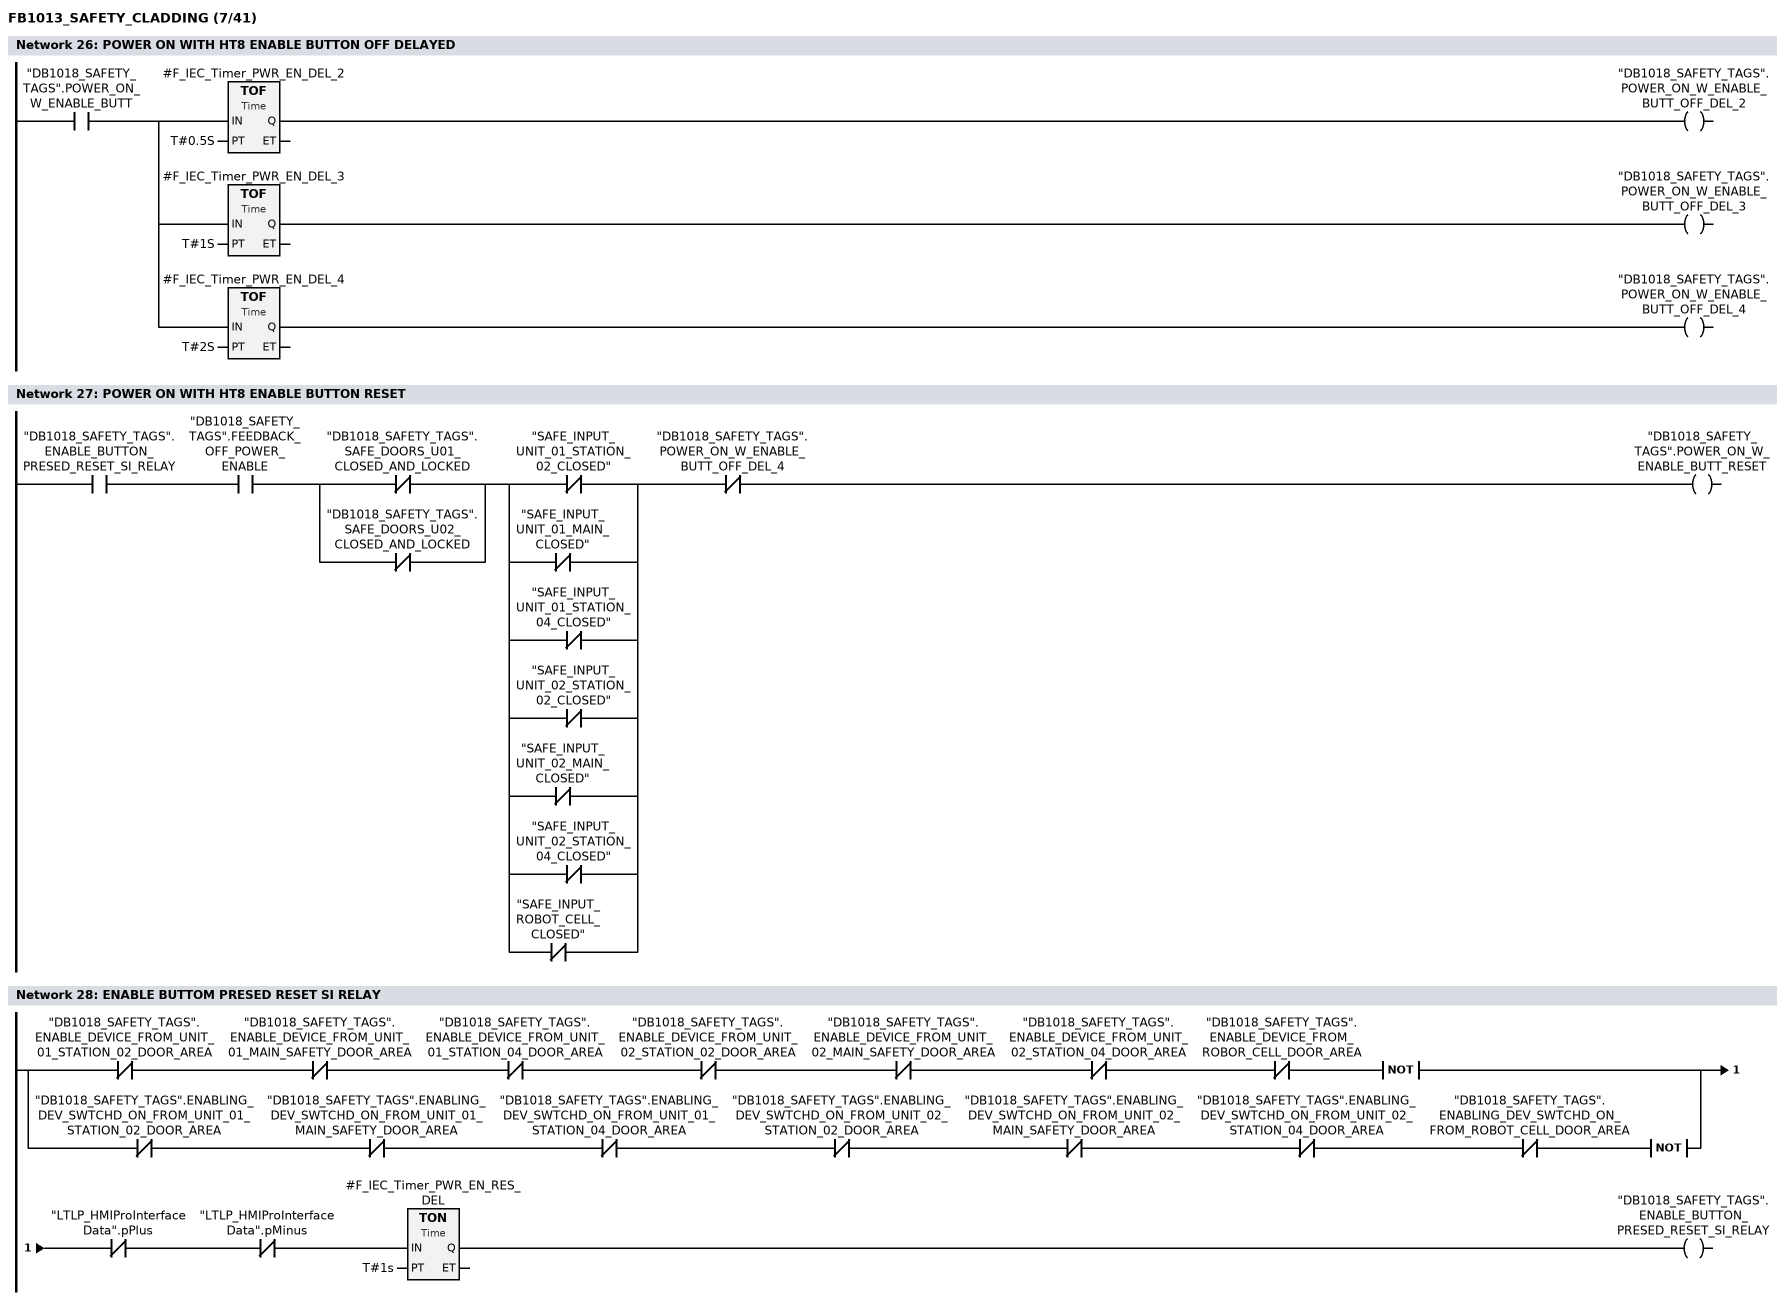
   RUNG wire#powerrail
      Contact( "DB1018_SAFETY_TAGS".POWER_ON_W_ENABLE_BUTT )
      wire#w1
      { S7_Templates := "[time_type := Time, codedbool_type := DInt]" } #F_IEC_Timer_PWR_EN_DEL_2.TOF(pt := T#0.5S, et =>)
      Coil( "DB1018_SAFETY_TAGS".POWER_ON_W_ENABLE_BUTT_OFF_DEL_2 )
   END_RUNG
   RUNG wire#w1
      { S7_Templates := "[time_type := Time, codedbool_type := DInt]" } #F_IEC_Timer_PWR_EN_DEL_3.TOF(pt := T#1S, et =>)
      Coil( "DB1018_SAFETY_TAGS".POWER_ON_W_ENABLE_BUTT_OFF_DEL_3 )
   END_RUNG
   RUNG wire#w1
      { S7_Templates := "[time_type := Time, codedbool_type := DInt]" } #F_IEC_Timer_PWR_EN_DEL_4.TOF(pt := T#2S, et =>)
      Coil( "DB1018_SAFETY_TAGS".POWER_ON_W_ENABLE_BUTT_OFF_DEL_4 )
   END_RUNG
   // the same network as SCL:
   #F_IEC_Timer_PWR_EN_DEL_2.TOF(IN := "DB1018_SAFETY_TAGS".POWER_ON_W_ENABLE_BUTT, PT := T#0.5S);
   "DB1018_SAFETY_TAGS".POWER_ON_W_ENABLE_BUTT_OFF_DEL_2 := #F_IEC_Timer_PWR_EN_DEL_2.Q;
   #F_IEC_Timer_PWR_EN_DEL_3.TOF(IN := "DB1018_SAFETY_TAGS".POWER_ON_W_ENABLE_BUTT, PT := T#1S);
   "DB1018_SAFETY_TAGS".POWER_ON_W_ENABLE_BUTT_OFF_DEL_3 := #F_IEC_Timer_PWR_EN_DEL_3.Q;
   #F_IEC_Timer_PWR_EN_DEL_4.TOF(IN := "DB1018_SAFETY_TAGS".POWER_ON_W_ENABLE_BUTT, PT := T#2S);
   "DB1018_SAFETY_TAGS".POWER_ON_W_ENABLE_BUTT_OFF_DEL_4 := #F_IEC_Timer_PWR_EN_DEL_4.Q;
END_REGION

REGION Network 27: POWER ON WITH HT8 ENABLE BUTTON RESET
   RUNG wire#powerrail
      Contact( "DB1018_SAFETY_TAGS".ENABLE_BUTTON_PRESED_RESET_SI_RELAY )
      Contact( "DB1018_SAFETY_TAGS".FEEDBACK_OFF_POWER_ENABLE )
      wire#w1
      I_Contact( "DB1018_SAFETY_TAGS".SAFE_DOORS_U01_CLOSED_AND_LOCKED )
      wire#w2
      I_Contact( "SAFE_INPUT_UNIT_01_STATION_02_CLOSED" )
      wire#w3
      I_Contact( "DB1018_SAFETY_TAGS".POWER_ON_W_ENABLE_BUTT_OFF_DEL_4 )
      Coil( "DB1018_SAFETY_TAGS".POWER_ON_W_ENABLE_BUTT_RESET )
   END_RUNG
   RUNG wire#w1
      I_Contact( "DB1018_SAFETY_TAGS".SAFE_DOORS_U02_CLOSED_AND_LOCKED )
   END_RUNG wire#w2
   RUNG wire#w2
      I_Contact( "SAFE_INPUT_UNIT_01_MAIN_CLOSED" )
   END_RUNG wire#w3
   RUNG wire#w2
      I_Contact( "SAFE_INPUT_UNIT_01_STATION_04_CLOSED" )
   END_RUNG wire#w3
   RUNG wire#w2
      I_Contact( "SAFE_INPUT_UNIT_02_STATION_02_CLOSED" )
   END_RUNG wire#w3
   RUNG wire#w2
      I_Contact( "SAFE_INPUT_UNIT_02_MAIN_CLOSED" )
   END_RUNG wire#w3
   RUNG wire#w2
      I_Contact( "SAFE_INPUT_UNIT_02_STATION_04_CLOSED" )
   END_RUNG wire#w3
   RUNG wire#w2
      I_Contact( "SAFE_INPUT_ROBOT_CELL_CLOSED" )
   END_RUNG wire#w3
   // the same network as SCL:
   "DB1018_SAFETY_TAGS".POWER_ON_W_ENABLE_BUTT_RESET := "DB1018_SAFETY_TAGS".ENABLE_BUTTON_PRESED_RESET_SI_RELAY AND "DB1018_SAFETY_TAGS".FEEDBACK_OFF_POWER_ENABLE AND (NOT "DB1018_SAFETY_TAGS".SAFE_DOORS_U01_CLOSED_AND_LOCKED OR NOT "DB1018_SAFETY_TAGS".SAFE_DOORS_U02_CLOSED_AND_LOCKED) AND (NOT "SAFE_INPUT_UNIT_01_STATION_02_CLOSED" OR NOT "SAFE_INPUT_UNIT_01_MAIN_CLOSED" OR NOT "SAFE_INPUT_UNIT_01_STATION_04_CLOSED" OR NOT "SAFE_INPUT_UNIT_02_STATION_02_CLOSED" OR NOT "SAFE_INPUT_UNIT_02_MAIN_CLOSED" OR NOT "SAFE_INPUT_UNIT_02_STATION_04_CLOSED" OR NOT "SAFE_INPUT_ROBOT_CELL_CLOSED") AND NOT "DB1018_SAFETY_TAGS".POWER_ON_W_ENABLE_BUTT_OFF_DEL_4;
END_REGION

REGION Network 28: ENABLE BUTTOM PRESED RESET SI RELAY
   RUNG wire#powerrail
      I_Contact( "DB1018_SAFETY_TAGS".ENABLE_DEVICE_FROM_UNIT_01_STATION_02_DOOR_AREA )
      I_Contact( "DB1018_SAFETY_TAGS".ENABLE_DEVICE_FROM_UNIT_01_MAIN_SAFETY_DOOR_AREA )
      I_Contact( "DB1018_SAFETY_TAGS".ENABLE_DEVICE_FROM_UNIT_01_STATION_04_DOOR_AREA )
      I_Contact( "DB1018_SAFETY_TAGS".ENABLE_DEVICE_FROM_UNIT_02_STATION_02_DOOR_AREA )
      I_Contact( "DB1018_SAFETY_TAGS".ENABLE_DEVICE_FROM_UNIT_02_MAIN_SAFETY_DOOR_AREA )
      I_Contact( "DB1018_SAFETY_TAGS".ENABLE_DEVICE_FROM_UNIT_02_STATION_04_DOOR_AREA )
      I_Contact( "DB1018_SAFETY_TAGS".ENABLE_DEVICE_FROM_ROBOR_CELL_DOOR_AREA )
      Not()
      wire#w1
      I_Contact( "LTLP_HMIProInterfaceData".pPlus )
      I_Contact( "LTLP_HMIProInterfaceData".pMinus )
      { S7_Templates := "[time_type := Time, codedbool_type := DInt]" } #F_IEC_Timer_PWR_EN_RES_DEL.TON(pt := T#1s, et =>)
      Coil( "DB1018_SAFETY_TAGS".ENABLE_BUTTON_PRESED_RESET_SI_RELAY )
   END_RUNG
   RUNG wire#powerrail
      I_Contact( "DB1018_SAFETY_TAGS".ENABLING_DEV_SWTCHD_ON_FROM_UNIT_01_STATION_02_DOOR_AREA )
      I_Contact( "DB1018_SAFETY_TAGS".ENABLING_DEV_SWTCHD_ON_FROM_UNIT_01_MAIN_SAFETY_DOOR_AREA )
      I_Contact( "DB1018_SAFETY_TAGS".ENABLING_DEV_SWTCHD_ON_FROM_UNIT_01_STATION_04_DOOR_AREA )
      I_Contact( "DB1018_SAFETY_TAGS".ENABLING_DEV_SWTCHD_ON_FROM_UNIT_02_STATION_02_DOOR_AREA )
      I_Contact( "DB1018_SAFETY_TAGS".ENABLING_DEV_SWTCHD_ON_FROM_UNIT_02_MAIN_SAFETY_DOOR_AREA )
      I_Contact( "DB1018_SAFETY_TAGS".ENABLING_DEV_SWTCHD_ON_FROM_UNIT_02_STATION_04_DOOR_AREA )
      I_Contact( "DB1018_SAFETY_TAGS".ENABLING_DEV_SWTCHD_ON_FROM_ROBOT_CELL_DOOR_AREA )
      Not()
   END_RUNG wire#w1
   // the same network as SCL:
   #F_IEC_Timer_PWR_EN_RES_DEL.TON(IN := (NOT (NOT "DB1018_SAFETY_TAGS".ENABLE_DEVICE_FROM_UNIT_01_STATION_02_DOOR_AREA AND NOT "DB1018_SAFETY_TAGS".ENABLE_DEVICE_FROM_UNIT_01_MAIN_SAFETY_DOOR_AREA AND NOT "DB1018_SAFETY_TAGS".ENABLE_DEVICE_FROM_UNIT_01_STATION_04_DOOR_AREA AND NOT "DB1018_SAFETY_TAGS".ENABLE_DEVICE_FROM_UNIT_02_STATION_02_DOOR_AREA AND NOT "DB1018_SAFETY_TAGS".ENABLE_DEVICE_FROM_UNIT_02_MAIN_SAFETY_DOOR_AREA AND NOT "DB1018_SAFETY_TAGS".ENABLE_DEVICE_FROM_UNIT_02_STATION_04_DOOR_AREA AND NOT "DB1018_SAFETY_TAGS".ENABLE_DEVICE_FROM_ROBOR_CELL_DOOR_AREA) OR NOT (NOT "DB1018_SAFETY_TAGS".ENABLING_DEV_SWTCHD_ON_FROM_UNIT_01_STATION_02_DOOR_AREA AND NOT "DB1018_SAFETY_TAGS".ENABLING_DEV_SWTCHD_ON_FROM_UNIT_01_MAIN_SAFETY_DOOR_AREA AND NOT "DB1018_SAFETY_TAGS".ENABLING_DEV_SWTCHD_ON_FROM_UNIT_01_STATION_04_DOOR_AREA AND NOT "DB1018_SAFETY_TAGS".ENABLING_DEV_SWTCHD_ON_FROM_UNIT_02_STATION_02_DOOR_AREA AND NOT "DB1018_SAFETY_TAGS".ENABLING_DEV_SWTCHD_ON_FROM_UNIT_02_MAIN_SAFETY_DOOR_AREA AND NOT "DB1018_SAFETY_TAGS".ENABLING_DEV_SWTCHD_ON_FROM_UNIT_02_STATION_04_DOOR_AREA AND NOT "DB1018_SAFETY_TAGS".ENABLING_DEV_SWTCHD_ON_FROM_ROBOT_CELL_DOOR_AREA)) AND NOT "LTLP_HMIProInterfaceData".pPlus AND NOT "LTLP_HMIProInterfaceData".pMinus,
                           PT := T#1s);
   "DB1018_SAFETY_TAGS".ENABLE_BUTTON_PRESED_RESET_SI_RELAY := #F_IEC_Timer_PWR_EN_RES_DEL.Q;
END_REGION

REGION Network 29: UNIT 01 STATION 02 SAFETY DOOR OPENED AND ENABLING DEVICE SWITCHED ON
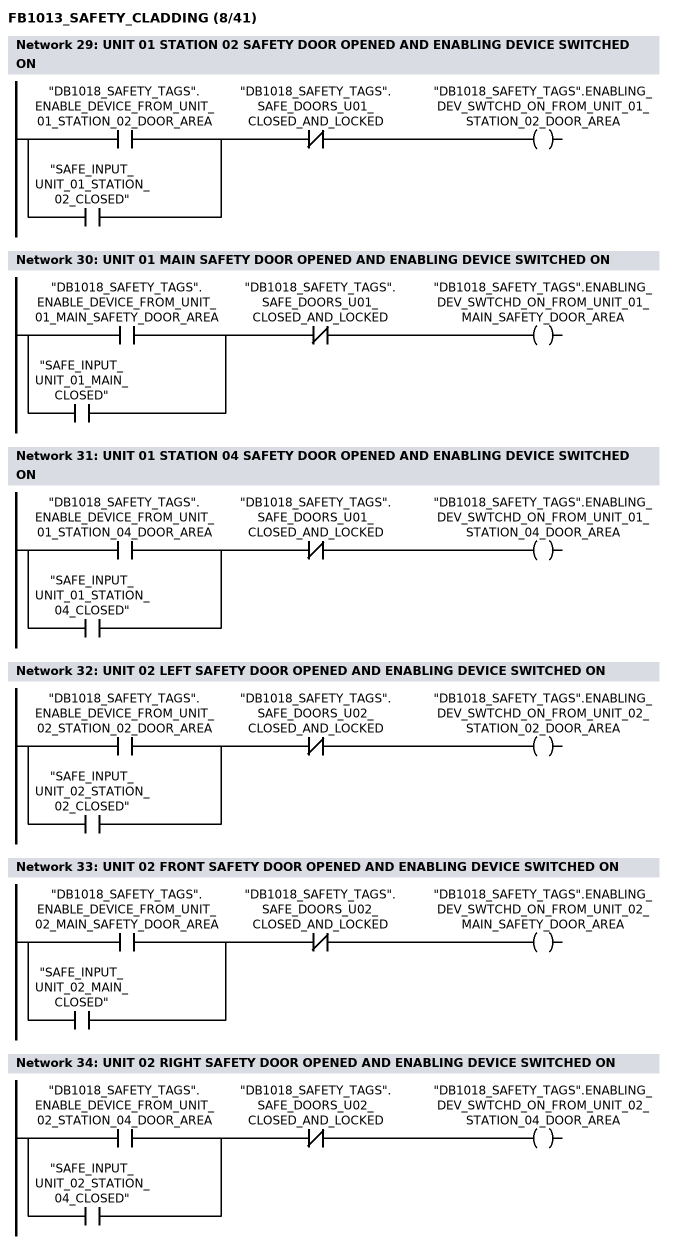
   RUNG wire#powerrail
      Contact( "DB1018_SAFETY_TAGS".ENABLE_DEVICE_FROM_UNIT_01_STATION_02_DOOR_AREA )
      wire#w1
      I_Contact( "DB1018_SAFETY_TAGS".SAFE_DOORS_U01_CLOSED_AND_LOCKED )
      Coil( "DB1018_SAFETY_TAGS".ENABLING_DEV_SWTCHD_ON_FROM_UNIT_01_STATION_02_DOOR_AREA )
   END_RUNG
   RUNG wire#powerrail
      Contact( "SAFE_INPUT_UNIT_01_STATION_02_CLOSED" )
   END_RUNG wire#w1
   // the same network as SCL:
   "DB1018_SAFETY_TAGS".ENABLING_DEV_SWTCHD_ON_FROM_UNIT_01_STATION_02_DOOR_AREA := ("DB1018_SAFETY_TAGS".ENABLE_DEVICE_FROM_UNIT_01_STATION_02_DOOR_AREA OR "SAFE_INPUT_UNIT_01_STATION_02_CLOSED") AND NOT "DB1018_SAFETY_TAGS".SAFE_DOORS_U01_CLOSED_AND_LOCKED;
END_REGION

REGION Network 30: UNIT 01 MAIN SAFETY DOOR OPENED AND ENABLING DEVICE SWITCHED ON
   RUNG wire#powerrail
      Contact( "DB1018_SAFETY_TAGS".ENABLE_DEVICE_FROM_UNIT_01_MAIN_SAFETY_DOOR_AREA )
      wire#w1
      I_Contact( "DB1018_SAFETY_TAGS".SAFE_DOORS_U01_CLOSED_AND_LOCKED )
      Coil( "DB1018_SAFETY_TAGS".ENABLING_DEV_SWTCHD_ON_FROM_UNIT_01_MAIN_SAFETY_DOOR_AREA )
   END_RUNG
   RUNG wire#powerrail
      Contact( "SAFE_INPUT_UNIT_01_MAIN_CLOSED" )
   END_RUNG wire#w1
   // the same network as SCL:
   "DB1018_SAFETY_TAGS".ENABLING_DEV_SWTCHD_ON_FROM_UNIT_01_MAIN_SAFETY_DOOR_AREA := ("DB1018_SAFETY_TAGS".ENABLE_DEVICE_FROM_UNIT_01_MAIN_SAFETY_DOOR_AREA OR "SAFE_INPUT_UNIT_01_MAIN_CLOSED") AND NOT "DB1018_SAFETY_TAGS".SAFE_DOORS_U01_CLOSED_AND_LOCKED;
END_REGION

REGION Network 31: UNIT 01 STATION 04 SAFETY DOOR OPENED AND ENABLING DEVICE SWITCHED ON
   RUNG wire#powerrail
      Contact( "DB1018_SAFETY_TAGS".ENABLE_DEVICE_FROM_UNIT_01_STATION_04_DOOR_AREA )
      wire#w1
      I_Contact( "DB1018_SAFETY_TAGS".SAFE_DOORS_U01_CLOSED_AND_LOCKED )
      Coil( "DB1018_SAFETY_TAGS".ENABLING_DEV_SWTCHD_ON_FROM_UNIT_01_STATION_04_DOOR_AREA )
   END_RUNG
   RUNG wire#powerrail
      Contact( "SAFE_INPUT_UNIT_01_STATION_04_CLOSED" )
   END_RUNG wire#w1
   // the same network as SCL:
   "DB1018_SAFETY_TAGS".ENABLING_DEV_SWTCHD_ON_FROM_UNIT_01_STATION_04_DOOR_AREA := ("DB1018_SAFETY_TAGS".ENABLE_DEVICE_FROM_UNIT_01_STATION_04_DOOR_AREA OR "SAFE_INPUT_UNIT_01_STATION_04_CLOSED") AND NOT "DB1018_SAFETY_TAGS".SAFE_DOORS_U01_CLOSED_AND_LOCKED;
END_REGION

REGION Network 32: UNIT 02 LEFT SAFETY DOOR OPENED AND ENABLING DEVICE SWITCHED ON
   RUNG wire#powerrail
      Contact( "DB1018_SAFETY_TAGS".ENABLE_DEVICE_FROM_UNIT_02_STATION_02_DOOR_AREA )
      wire#w1
      I_Contact( "DB1018_SAFETY_TAGS".SAFE_DOORS_U02_CLOSED_AND_LOCKED )
      Coil( "DB1018_SAFETY_TAGS".ENABLING_DEV_SWTCHD_ON_FROM_UNIT_02_STATION_02_DOOR_AREA )
   END_RUNG
   RUNG wire#powerrail
      Contact( "SAFE_INPUT_UNIT_02_STATION_02_CLOSED" )
   END_RUNG wire#w1
   // the same network as SCL:
   "DB1018_SAFETY_TAGS".ENABLING_DEV_SWTCHD_ON_FROM_UNIT_02_STATION_02_DOOR_AREA := ("DB1018_SAFETY_TAGS".ENABLE_DEVICE_FROM_UNIT_02_STATION_02_DOOR_AREA OR "SAFE_INPUT_UNIT_02_STATION_02_CLOSED") AND NOT "DB1018_SAFETY_TAGS".SAFE_DOORS_U02_CLOSED_AND_LOCKED;
END_REGION

REGION Network 33: UNIT 02 FRONT SAFETY DOOR OPENED AND ENABLING DEVICE SWITCHED ON
   RUNG wire#powerrail
      Contact( "DB1018_SAFETY_TAGS".ENABLE_DEVICE_FROM_UNIT_02_MAIN_SAFETY_DOOR_AREA )
      wire#w1
      I_Contact( "DB1018_SAFETY_TAGS".SAFE_DOORS_U02_CLOSED_AND_LOCKED )
      Coil( "DB1018_SAFETY_TAGS".ENABLING_DEV_SWTCHD_ON_FROM_UNIT_02_MAIN_SAFETY_DOOR_AREA )
   END_RUNG
   RUNG wire#powerrail
      Contact( "SAFE_INPUT_UNIT_02_MAIN_CLOSED" )
   END_RUNG wire#w1
   // the same network as SCL:
   "DB1018_SAFETY_TAGS".ENABLING_DEV_SWTCHD_ON_FROM_UNIT_02_MAIN_SAFETY_DOOR_AREA := ("DB1018_SAFETY_TAGS".ENABLE_DEVICE_FROM_UNIT_02_MAIN_SAFETY_DOOR_AREA OR "SAFE_INPUT_UNIT_02_MAIN_CLOSED") AND NOT "DB1018_SAFETY_TAGS".SAFE_DOORS_U02_CLOSED_AND_LOCKED;
END_REGION

REGION Network 34: UNIT 02 RIGHT SAFETY DOOR OPENED AND ENABLING DEVICE SWITCHED ON
   RUNG wire#powerrail
      Contact( "DB1018_SAFETY_TAGS".ENABLE_DEVICE_FROM_UNIT_02_STATION_04_DOOR_AREA )
      wire#w1
      I_Contact( "DB1018_SAFETY_TAGS".SAFE_DOORS_U02_CLOSED_AND_LOCKED )
      Coil( "DB1018_SAFETY_TAGS".ENABLING_DEV_SWTCHD_ON_FROM_UNIT_02_STATION_04_DOOR_AREA )
   END_RUNG
   RUNG wire#powerrail
      Contact( "SAFE_INPUT_UNIT_02_STATION_04_CLOSED" )
   END_RUNG wire#w1
   // the same network as SCL:
   "DB1018_SAFETY_TAGS".ENABLING_DEV_SWTCHD_ON_FROM_UNIT_02_STATION_04_DOOR_AREA := ("DB1018_SAFETY_TAGS".ENABLE_DEVICE_FROM_UNIT_02_STATION_04_DOOR_AREA OR "SAFE_INPUT_UNIT_02_STATION_04_CLOSED") AND NOT "DB1018_SAFETY_TAGS".SAFE_DOORS_U02_CLOSED_AND_LOCKED;
END_REGION

REGION Network 35: ROBOT CELL SAFETY DOOR OPENED AND ENABLING DEVICE SWITCHED ON
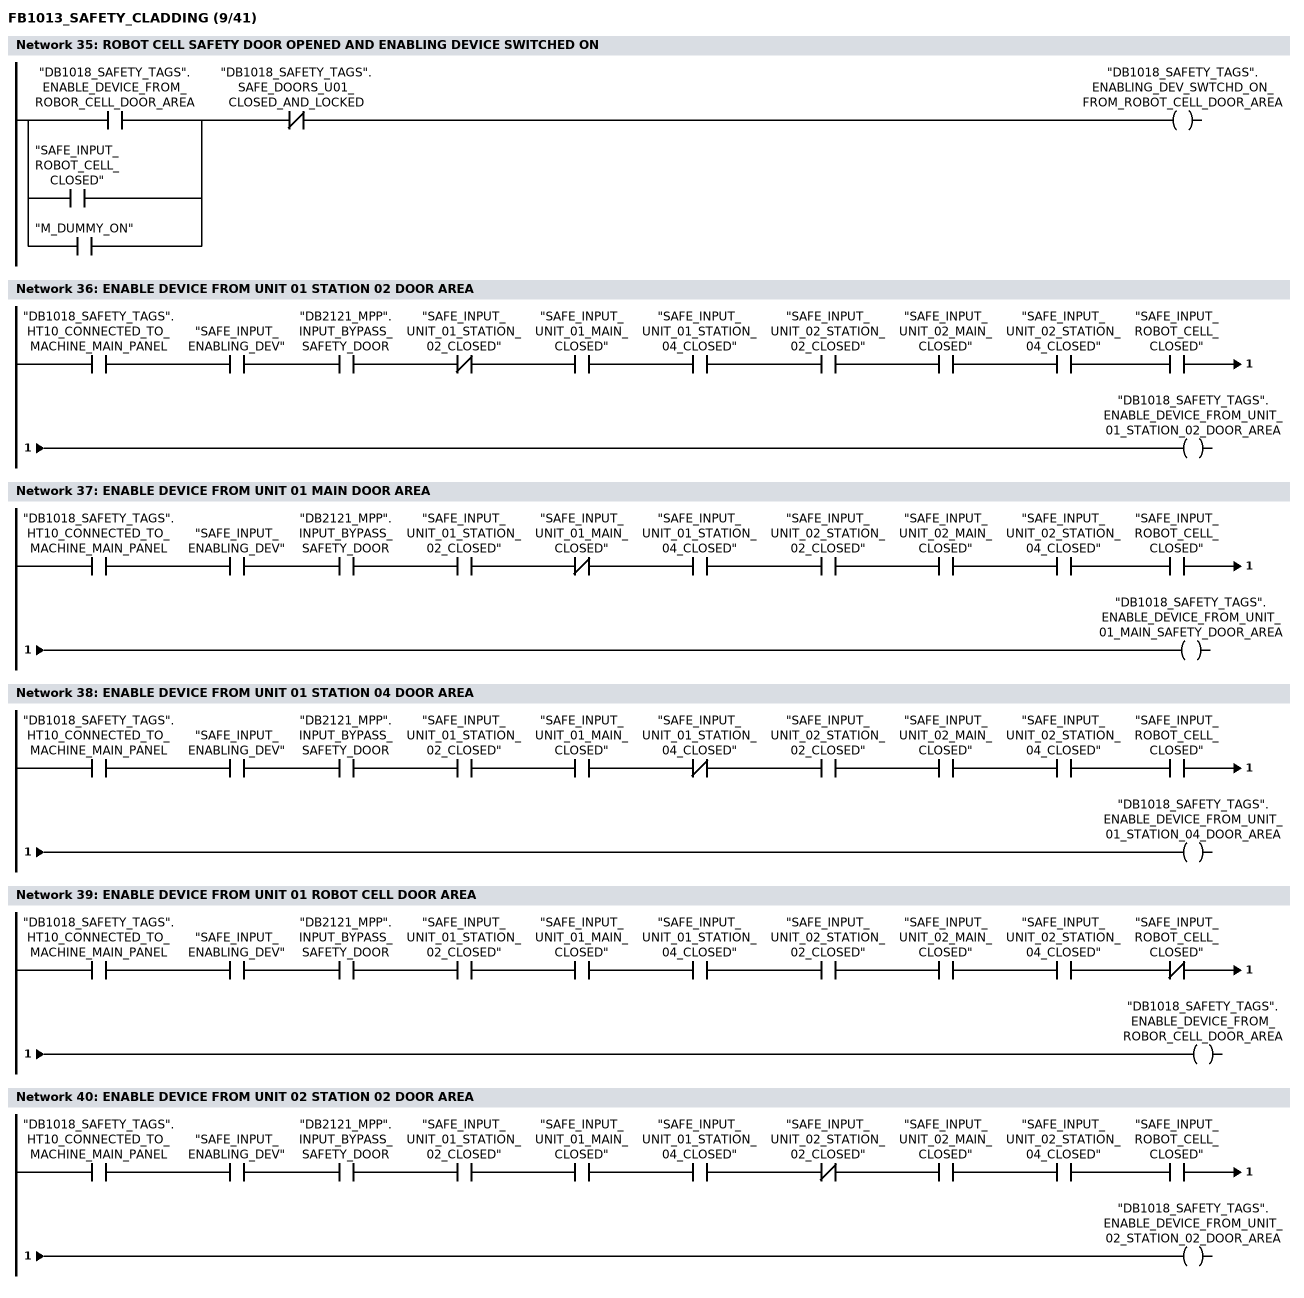
   RUNG wire#powerrail
      Contact( "DB1018_SAFETY_TAGS".ENABLE_DEVICE_FROM_ROBOR_CELL_DOOR_AREA )
      wire#w1
      I_Contact( "DB1018_SAFETY_TAGS".SAFE_DOORS_U01_CLOSED_AND_LOCKED )
      Coil( "DB1018_SAFETY_TAGS".ENABLING_DEV_SWTCHD_ON_FROM_ROBOT_CELL_DOOR_AREA )
   END_RUNG
   RUNG wire#powerrail
      Contact( "SAFE_INPUT_ROBOT_CELL_CLOSED" )
   END_RUNG wire#w1
   RUNG wire#powerrail
      Contact( "M_DUMMY_ON" )
   END_RUNG wire#w1
   // the same network as SCL:
   "DB1018_SAFETY_TAGS".ENABLING_DEV_SWTCHD_ON_FROM_ROBOT_CELL_DOOR_AREA := ("DB1018_SAFETY_TAGS".ENABLE_DEVICE_FROM_ROBOR_CELL_DOOR_AREA OR "SAFE_INPUT_ROBOT_CELL_CLOSED" OR "M_DUMMY_ON") AND NOT "DB1018_SAFETY_TAGS".SAFE_DOORS_U01_CLOSED_AND_LOCKED;
END_REGION

REGION Network 36: ENABLE DEVICE FROM UNIT 01 STATION 02 DOOR AREA
   RUNG wire#powerrail
      Contact( "DB1018_SAFETY_TAGS".HT10_CONNECTED_TO_MACHINE_MAIN_PANEL )
      Contact( "SAFE_INPUT_ENABLING_DEV" )
      Contact( "DB2121_MPP".INPUT_BYPASS_SAFETY_DOOR )
      I_Contact( "SAFE_INPUT_UNIT_01_STATION_02_CLOSED" )
      Contact( "SAFE_INPUT_UNIT_01_MAIN_CLOSED" )
      Contact( "SAFE_INPUT_UNIT_01_STATION_04_CLOSED" )
      Contact( "SAFE_INPUT_UNIT_02_STATION_02_CLOSED" )
      Contact( "SAFE_INPUT_UNIT_02_MAIN_CLOSED" )
      Contact( "SAFE_INPUT_UNIT_02_STATION_04_CLOSED" )
      Contact( "SAFE_INPUT_ROBOT_CELL_CLOSED" )
      Coil( "DB1018_SAFETY_TAGS".ENABLE_DEVICE_FROM_UNIT_01_STATION_02_DOOR_AREA )
   END_RUNG
   // the same network as SCL:
   "DB1018_SAFETY_TAGS".ENABLE_DEVICE_FROM_UNIT_01_STATION_02_DOOR_AREA := "DB1018_SAFETY_TAGS".HT10_CONNECTED_TO_MACHINE_MAIN_PANEL AND "SAFE_INPUT_ENABLING_DEV" AND "DB2121_MPP".INPUT_BYPASS_SAFETY_DOOR AND NOT "SAFE_INPUT_UNIT_01_STATION_02_CLOSED" AND "SAFE_INPUT_UNIT_01_MAIN_CLOSED" AND "SAFE_INPUT_UNIT_01_STATION_04_CLOSED" AND "SAFE_INPUT_UNIT_02_STATION_02_CLOSED" AND "SAFE_INPUT_UNIT_02_MAIN_CLOSED" AND "SAFE_INPUT_UNIT_02_STATION_04_CLOSED" AND "SAFE_INPUT_ROBOT_CELL_CLOSED";
END_REGION

REGION Network 37: ENABLE DEVICE FROM UNIT 01 MAIN DOOR AREA
   RUNG wire#powerrail
      Contact( "DB1018_SAFETY_TAGS".HT10_CONNECTED_TO_MACHINE_MAIN_PANEL )
      Contact( "SAFE_INPUT_ENABLING_DEV" )
      Contact( "DB2121_MPP".INPUT_BYPASS_SAFETY_DOOR )
      Contact( "SAFE_INPUT_UNIT_01_STATION_02_CLOSED" )
      I_Contact( "SAFE_INPUT_UNIT_01_MAIN_CLOSED" )
      Contact( "SAFE_INPUT_UNIT_01_STATION_04_CLOSED" )
      Contact( "SAFE_INPUT_UNIT_02_STATION_02_CLOSED" )
      Contact( "SAFE_INPUT_UNIT_02_MAIN_CLOSED" )
      Contact( "SAFE_INPUT_UNIT_02_STATION_04_CLOSED" )
      Contact( "SAFE_INPUT_ROBOT_CELL_CLOSED" )
      Coil( "DB1018_SAFETY_TAGS".ENABLE_DEVICE_FROM_UNIT_01_MAIN_SAFETY_DOOR_AREA )
   END_RUNG
   // the same network as SCL:
   "DB1018_SAFETY_TAGS".ENABLE_DEVICE_FROM_UNIT_01_MAIN_SAFETY_DOOR_AREA := "DB1018_SAFETY_TAGS".HT10_CONNECTED_TO_MACHINE_MAIN_PANEL AND "SAFE_INPUT_ENABLING_DEV" AND "DB2121_MPP".INPUT_BYPASS_SAFETY_DOOR AND "SAFE_INPUT_UNIT_01_STATION_02_CLOSED" AND NOT "SAFE_INPUT_UNIT_01_MAIN_CLOSED" AND "SAFE_INPUT_UNIT_01_STATION_04_CLOSED" AND "SAFE_INPUT_UNIT_02_STATION_02_CLOSED" AND "SAFE_INPUT_UNIT_02_MAIN_CLOSED" AND "SAFE_INPUT_UNIT_02_STATION_04_CLOSED" AND "SAFE_INPUT_ROBOT_CELL_CLOSED";
END_REGION

REGION Network 38: ENABLE DEVICE FROM UNIT 01 STATION 04 DOOR AREA
   RUNG wire#powerrail
      Contact( "DB1018_SAFETY_TAGS".HT10_CONNECTED_TO_MACHINE_MAIN_PANEL )
      Contact( "SAFE_INPUT_ENABLING_DEV" )
      Contact( "DB2121_MPP".INPUT_BYPASS_SAFETY_DOOR )
      Contact( "SAFE_INPUT_UNIT_01_STATION_02_CLOSED" )
      Contact( "SAFE_INPUT_UNIT_01_MAIN_CLOSED" )
      I_Contact( "SAFE_INPUT_UNIT_01_STATION_04_CLOSED" )
      Contact( "SAFE_INPUT_UNIT_02_STATION_02_CLOSED" )
      Contact( "SAFE_INPUT_UNIT_02_MAIN_CLOSED" )
      Contact( "SAFE_INPUT_UNIT_02_STATION_04_CLOSED" )
      Contact( "SAFE_INPUT_ROBOT_CELL_CLOSED" )
      Coil( "DB1018_SAFETY_TAGS".ENABLE_DEVICE_FROM_UNIT_01_STATION_04_DOOR_AREA )
   END_RUNG
   // the same network as SCL:
   "DB1018_SAFETY_TAGS".ENABLE_DEVICE_FROM_UNIT_01_STATION_04_DOOR_AREA := "DB1018_SAFETY_TAGS".HT10_CONNECTED_TO_MACHINE_MAIN_PANEL AND "SAFE_INPUT_ENABLING_DEV" AND "DB2121_MPP".INPUT_BYPASS_SAFETY_DOOR AND "SAFE_INPUT_UNIT_01_STATION_02_CLOSED" AND "SAFE_INPUT_UNIT_01_MAIN_CLOSED" AND NOT "SAFE_INPUT_UNIT_01_STATION_04_CLOSED" AND "SAFE_INPUT_UNIT_02_STATION_02_CLOSED" AND "SAFE_INPUT_UNIT_02_MAIN_CLOSED" AND "SAFE_INPUT_UNIT_02_STATION_04_CLOSED" AND "SAFE_INPUT_ROBOT_CELL_CLOSED";
END_REGION

REGION Network 39: ENABLE DEVICE FROM UNIT 01 ROBOT CELL DOOR AREA
   RUNG wire#powerrail
      Contact( "DB1018_SAFETY_TAGS".HT10_CONNECTED_TO_MACHINE_MAIN_PANEL )
      Contact( "SAFE_INPUT_ENABLING_DEV" )
      Contact( "DB2121_MPP".INPUT_BYPASS_SAFETY_DOOR )
      Contact( "SAFE_INPUT_UNIT_01_STATION_02_CLOSED" )
      Contact( "SAFE_INPUT_UNIT_01_MAIN_CLOSED" )
      Contact( "SAFE_INPUT_UNIT_01_STATION_04_CLOSED" )
      Contact( "SAFE_INPUT_UNIT_02_STATION_02_CLOSED" )
      Contact( "SAFE_INPUT_UNIT_02_MAIN_CLOSED" )
      Contact( "SAFE_INPUT_UNIT_02_STATION_04_CLOSED" )
      I_Contact( "SAFE_INPUT_ROBOT_CELL_CLOSED" )
      Coil( "DB1018_SAFETY_TAGS".ENABLE_DEVICE_FROM_ROBOR_CELL_DOOR_AREA )
   END_RUNG
   // the same network as SCL:
   "DB1018_SAFETY_TAGS".ENABLE_DEVICE_FROM_ROBOR_CELL_DOOR_AREA := "DB1018_SAFETY_TAGS".HT10_CONNECTED_TO_MACHINE_MAIN_PANEL AND "SAFE_INPUT_ENABLING_DEV" AND "DB2121_MPP".INPUT_BYPASS_SAFETY_DOOR AND "SAFE_INPUT_UNIT_01_STATION_02_CLOSED" AND "SAFE_INPUT_UNIT_01_MAIN_CLOSED" AND "SAFE_INPUT_UNIT_01_STATION_04_CLOSED" AND "SAFE_INPUT_UNIT_02_STATION_02_CLOSED" AND "SAFE_INPUT_UNIT_02_MAIN_CLOSED" AND "SAFE_INPUT_UNIT_02_STATION_04_CLOSED" AND NOT "SAFE_INPUT_ROBOT_CELL_CLOSED";
END_REGION

REGION Network 40: ENABLE DEVICE FROM UNIT 02 STATION 02 DOOR AREA
   RUNG wire#powerrail
      Contact( "DB1018_SAFETY_TAGS".HT10_CONNECTED_TO_MACHINE_MAIN_PANEL )
      Contact( "SAFE_INPUT_ENABLING_DEV" )
      Contact( "DB2121_MPP".INPUT_BYPASS_SAFETY_DOOR )
      Contact( "SAFE_INPUT_UNIT_01_STATION_02_CLOSED" )
      Contact( "SAFE_INPUT_UNIT_01_MAIN_CLOSED" )
      Contact( "SAFE_INPUT_UNIT_01_STATION_04_CLOSED" )
      I_Contact( "SAFE_INPUT_UNIT_02_STATION_02_CLOSED" )
      Contact( "SAFE_INPUT_UNIT_02_MAIN_CLOSED" )
      Contact( "SAFE_INPUT_UNIT_02_STATION_04_CLOSED" )
      Contact( "SAFE_INPUT_ROBOT_CELL_CLOSED" )
      Coil( "DB1018_SAFETY_TAGS".ENABLE_DEVICE_FROM_UNIT_02_STATION_02_DOOR_AREA )
   END_RUNG
   // the same network as SCL:
   "DB1018_SAFETY_TAGS".ENABLE_DEVICE_FROM_UNIT_02_STATION_02_DOOR_AREA := "DB1018_SAFETY_TAGS".HT10_CONNECTED_TO_MACHINE_MAIN_PANEL AND "SAFE_INPUT_ENABLING_DEV" AND "DB2121_MPP".INPUT_BYPASS_SAFETY_DOOR AND "SAFE_INPUT_UNIT_01_STATION_02_CLOSED" AND "SAFE_INPUT_UNIT_01_MAIN_CLOSED" AND "SAFE_INPUT_UNIT_01_STATION_04_CLOSED" AND NOT "SAFE_INPUT_UNIT_02_STATION_02_CLOSED" AND "SAFE_INPUT_UNIT_02_MAIN_CLOSED" AND "SAFE_INPUT_UNIT_02_STATION_04_CLOSED" AND "SAFE_INPUT_ROBOT_CELL_CLOSED";
END_REGION

REGION Network 41: ENABLE DEVICE FROM UNIT 02 MAIN DOOR AREA
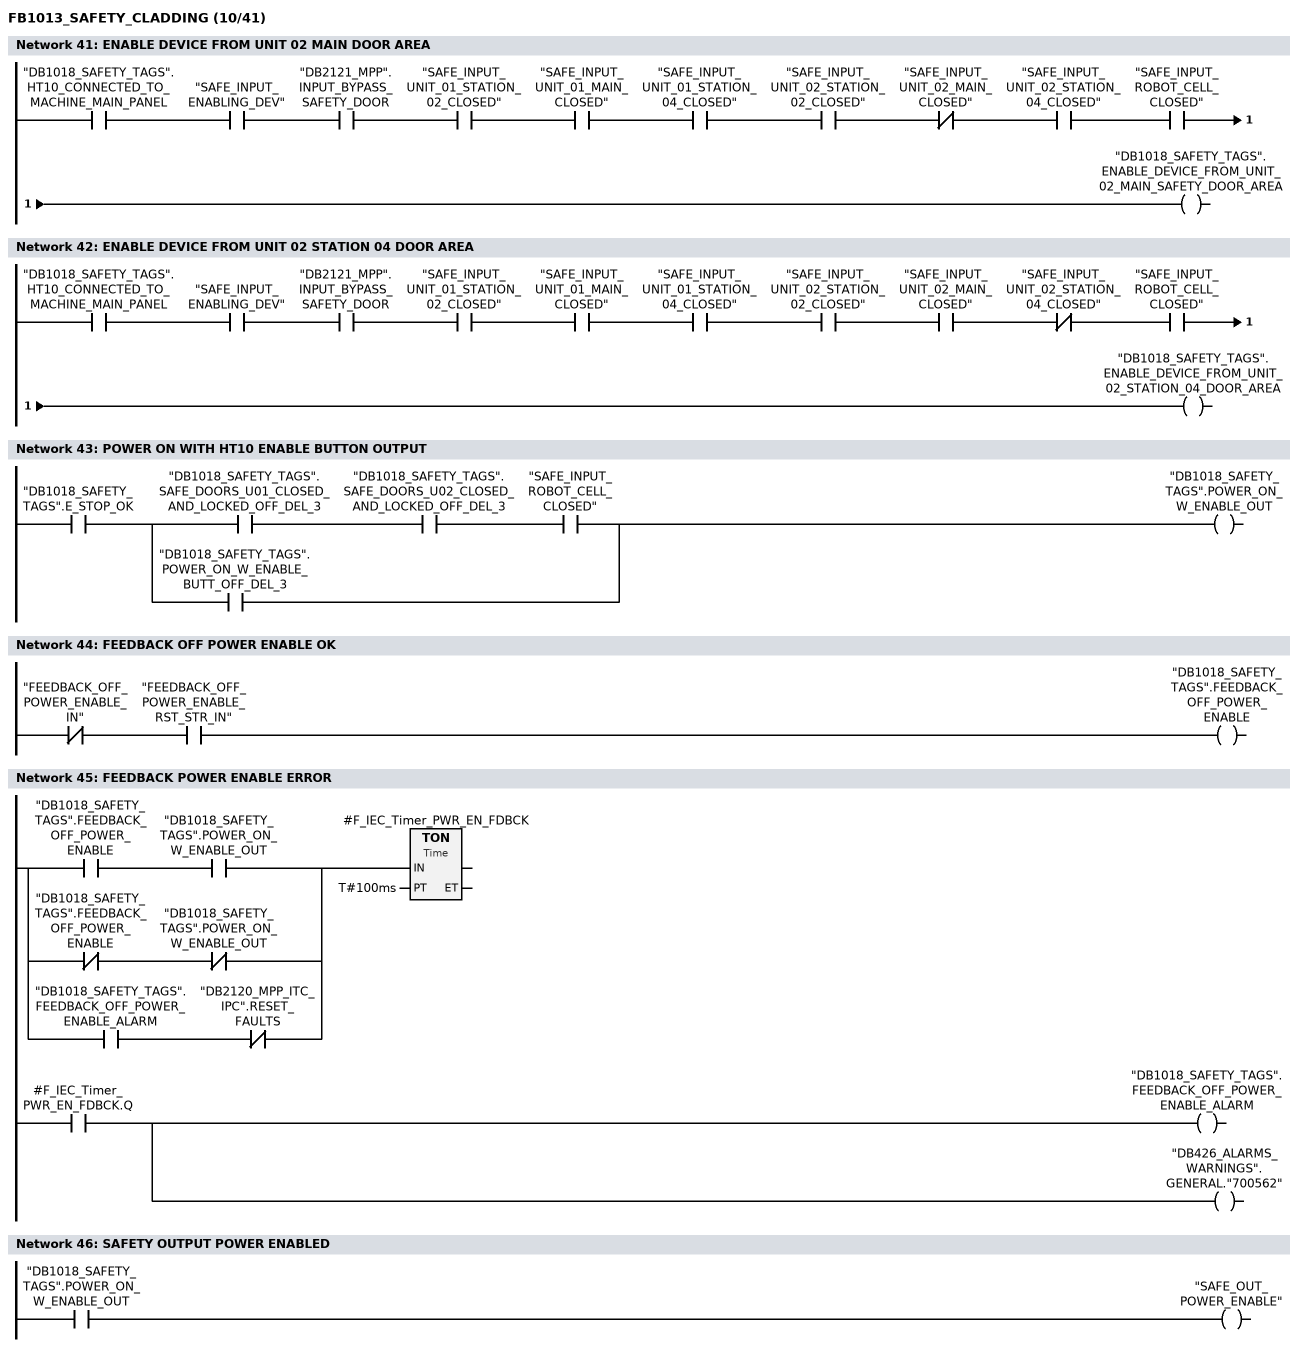
   RUNG wire#powerrail
      Contact( "DB1018_SAFETY_TAGS".HT10_CONNECTED_TO_MACHINE_MAIN_PANEL )
      Contact( "SAFE_INPUT_ENABLING_DEV" )
      Contact( "DB2121_MPP".INPUT_BYPASS_SAFETY_DOOR )
      Contact( "SAFE_INPUT_UNIT_01_STATION_02_CLOSED" )
      Contact( "SAFE_INPUT_UNIT_01_MAIN_CLOSED" )
      Contact( "SAFE_INPUT_UNIT_01_STATION_04_CLOSED" )
      Contact( "SAFE_INPUT_UNIT_02_STATION_02_CLOSED" )
      I_Contact( "SAFE_INPUT_UNIT_02_MAIN_CLOSED" )
      Contact( "SAFE_INPUT_UNIT_02_STATION_04_CLOSED" )
      Contact( "SAFE_INPUT_ROBOT_CELL_CLOSED" )
      Coil( "DB1018_SAFETY_TAGS".ENABLE_DEVICE_FROM_UNIT_02_MAIN_SAFETY_DOOR_AREA )
   END_RUNG
   // the same network as SCL:
   "DB1018_SAFETY_TAGS".ENABLE_DEVICE_FROM_UNIT_02_MAIN_SAFETY_DOOR_AREA := "DB1018_SAFETY_TAGS".HT10_CONNECTED_TO_MACHINE_MAIN_PANEL AND "SAFE_INPUT_ENABLING_DEV" AND "DB2121_MPP".INPUT_BYPASS_SAFETY_DOOR AND "SAFE_INPUT_UNIT_01_STATION_02_CLOSED" AND "SAFE_INPUT_UNIT_01_MAIN_CLOSED" AND "SAFE_INPUT_UNIT_01_STATION_04_CLOSED" AND "SAFE_INPUT_UNIT_02_STATION_02_CLOSED" AND NOT "SAFE_INPUT_UNIT_02_MAIN_CLOSED" AND "SAFE_INPUT_UNIT_02_STATION_04_CLOSED" AND "SAFE_INPUT_ROBOT_CELL_CLOSED";
END_REGION

REGION Network 42: ENABLE DEVICE FROM UNIT 02 STATION 04 DOOR AREA
   RUNG wire#powerrail
      Contact( "DB1018_SAFETY_TAGS".HT10_CONNECTED_TO_MACHINE_MAIN_PANEL )
      Contact( "SAFE_INPUT_ENABLING_DEV" )
      Contact( "DB2121_MPP".INPUT_BYPASS_SAFETY_DOOR )
      Contact( "SAFE_INPUT_UNIT_01_STATION_02_CLOSED" )
      Contact( "SAFE_INPUT_UNIT_01_MAIN_CLOSED" )
      Contact( "SAFE_INPUT_UNIT_01_STATION_04_CLOSED" )
      Contact( "SAFE_INPUT_UNIT_02_STATION_02_CLOSED" )
      Contact( "SAFE_INPUT_UNIT_02_MAIN_CLOSED" )
      I_Contact( "SAFE_INPUT_UNIT_02_STATION_04_CLOSED" )
      Contact( "SAFE_INPUT_ROBOT_CELL_CLOSED" )
      Coil( "DB1018_SAFETY_TAGS".ENABLE_DEVICE_FROM_UNIT_02_STATION_04_DOOR_AREA )
   END_RUNG
   // the same network as SCL:
   "DB1018_SAFETY_TAGS".ENABLE_DEVICE_FROM_UNIT_02_STATION_04_DOOR_AREA := "DB1018_SAFETY_TAGS".HT10_CONNECTED_TO_MACHINE_MAIN_PANEL AND "SAFE_INPUT_ENABLING_DEV" AND "DB2121_MPP".INPUT_BYPASS_SAFETY_DOOR AND "SAFE_INPUT_UNIT_01_STATION_02_CLOSED" AND "SAFE_INPUT_UNIT_01_MAIN_CLOSED" AND "SAFE_INPUT_UNIT_01_STATION_04_CLOSED" AND "SAFE_INPUT_UNIT_02_STATION_02_CLOSED" AND "SAFE_INPUT_UNIT_02_MAIN_CLOSED" AND NOT "SAFE_INPUT_UNIT_02_STATION_04_CLOSED" AND "SAFE_INPUT_ROBOT_CELL_CLOSED";
END_REGION

REGION Network 43: POWER ON WITH HT10 ENABLE BUTTON OUTPUT
   RUNG wire#powerrail
      Contact( "DB1018_SAFETY_TAGS".E_STOP_OK )
      wire#w1
      Contact( "DB1018_SAFETY_TAGS".SAFE_DOORS_U01_CLOSED_AND_LOCKED_OFF_DEL_3 )
      Contact( "DB1018_SAFETY_TAGS".SAFE_DOORS_U02_CLOSED_AND_LOCKED_OFF_DEL_3 )
      Contact( "SAFE_INPUT_ROBOT_CELL_CLOSED" )
      wire#w2
      Coil( "DB1018_SAFETY_TAGS".POWER_ON_W_ENABLE_OUT )
   END_RUNG
   RUNG wire#w1
      Contact( "DB1018_SAFETY_TAGS".POWER_ON_W_ENABLE_BUTT_OFF_DEL_3 )
   END_RUNG wire#w2
   // the same network as SCL:
   "DB1018_SAFETY_TAGS".POWER_ON_W_ENABLE_OUT := "DB1018_SAFETY_TAGS".E_STOP_OK AND (("DB1018_SAFETY_TAGS".SAFE_DOORS_U01_CLOSED_AND_LOCKED_OFF_DEL_3 AND "DB1018_SAFETY_TAGS".SAFE_DOORS_U02_CLOSED_AND_LOCKED_OFF_DEL_3 AND "SAFE_INPUT_ROBOT_CELL_CLOSED") OR "DB1018_SAFETY_TAGS".POWER_ON_W_ENABLE_BUTT_OFF_DEL_3);
END_REGION

REGION Network 44: FEEDBACK OFF POWER ENABLE OK
   RUNG wire#powerrail
      I_Contact( "FEEDBACK_OFF_POWER_ENABLE_IN" )
      Contact( "FEEDBACK_OFF_POWER_ENABLE_RST_STR_IN" )
      Coil( "DB1018_SAFETY_TAGS".FEEDBACK_OFF_POWER_ENABLE )
   END_RUNG
   // the same network as SCL:
   "DB1018_SAFETY_TAGS".FEEDBACK_OFF_POWER_ENABLE := NOT "FEEDBACK_OFF_POWER_ENABLE_IN" AND "FEEDBACK_OFF_POWER_ENABLE_RST_STR_IN";
END_REGION

REGION Network 45: FEEDBACK POWER ENABLE ERROR
   RUNG wire#powerrail
      Contact( "DB1018_SAFETY_TAGS".FEEDBACK_OFF_POWER_ENABLE )
      Contact( "DB1018_SAFETY_TAGS".POWER_ON_W_ENABLE_OUT )
      wire#w1
      { S7_Templates := "[time_type := Time, codedbool_type := DInt]" } #F_IEC_Timer_PWR_EN_FDBCK.TON(pt := T#100ms, et =>)
   END_RUNG
   RUNG wire#powerrail
      I_Contact( "DB1018_SAFETY_TAGS".FEEDBACK_OFF_POWER_ENABLE )
      I_Contact( "DB1018_SAFETY_TAGS".POWER_ON_W_ENABLE_OUT )
   END_RUNG wire#w1
   RUNG wire#powerrail
      Contact( "DB1018_SAFETY_TAGS".FEEDBACK_OFF_POWER_ENABLE_ALARM )
      I_Contact( "DB2120_MPP_ITC_IPC".RESET_FAULTS )
   END_RUNG wire#w1
   RUNG wire#powerrail
      Contact( #F_IEC_Timer_PWR_EN_FDBCK.Q )
      wire#w2
      Coil( "DB1018_SAFETY_TAGS".FEEDBACK_OFF_POWER_ENABLE_ALARM )
   END_RUNG
   RUNG wire#w2
      Coil( "DB426_ALARMS_WARNINGS".GENERAL."700562" )
   END_RUNG
   // the same network as SCL:
   #F_IEC_Timer_PWR_EN_FDBCK.TON(IN := ("DB1018_SAFETY_TAGS".FEEDBACK_OFF_POWER_ENABLE AND "DB1018_SAFETY_TAGS".POWER_ON_W_ENABLE_OUT) OR (NOT "DB1018_SAFETY_TAGS".FEEDBACK_OFF_POWER_ENABLE AND NOT "DB1018_SAFETY_TAGS".POWER_ON_W_ENABLE_OUT) OR ("DB1018_SAFETY_TAGS".FEEDBACK_OFF_POWER_ENABLE_ALARM AND NOT "DB2120_MPP_ITC_IPC".RESET_FAULTS),
                           PT := T#100ms);
   "DB1018_SAFETY_TAGS".FEEDBACK_OFF_POWER_ENABLE_ALARM := #F_IEC_Timer_PWR_EN_FDBCK.Q;
   "DB426_ALARMS_WARNINGS".GENERAL."700562" := #F_IEC_Timer_PWR_EN_FDBCK.Q;
END_REGION

REGION Network 46: SAFETY OUTPUT POWER ENABLED
   RUNG wire#powerrail
      Contact( "DB1018_SAFETY_TAGS".POWER_ON_W_ENABLE_OUT )
      Coil( "SAFE_OUT_POWER_ENABLE" )
   END_RUNG
   // the same network as SCL:
   "SAFE_OUT_POWER_ENABLE" := "DB1018_SAFETY_TAGS".POWER_ON_W_ENABLE_OUT;
END_REGION

REGION Network 47: *************** LASER SOURCE ENABLE ***************
END_REGION

REGION Network 48: LASER SOURCE ENABLE CONDITIONS
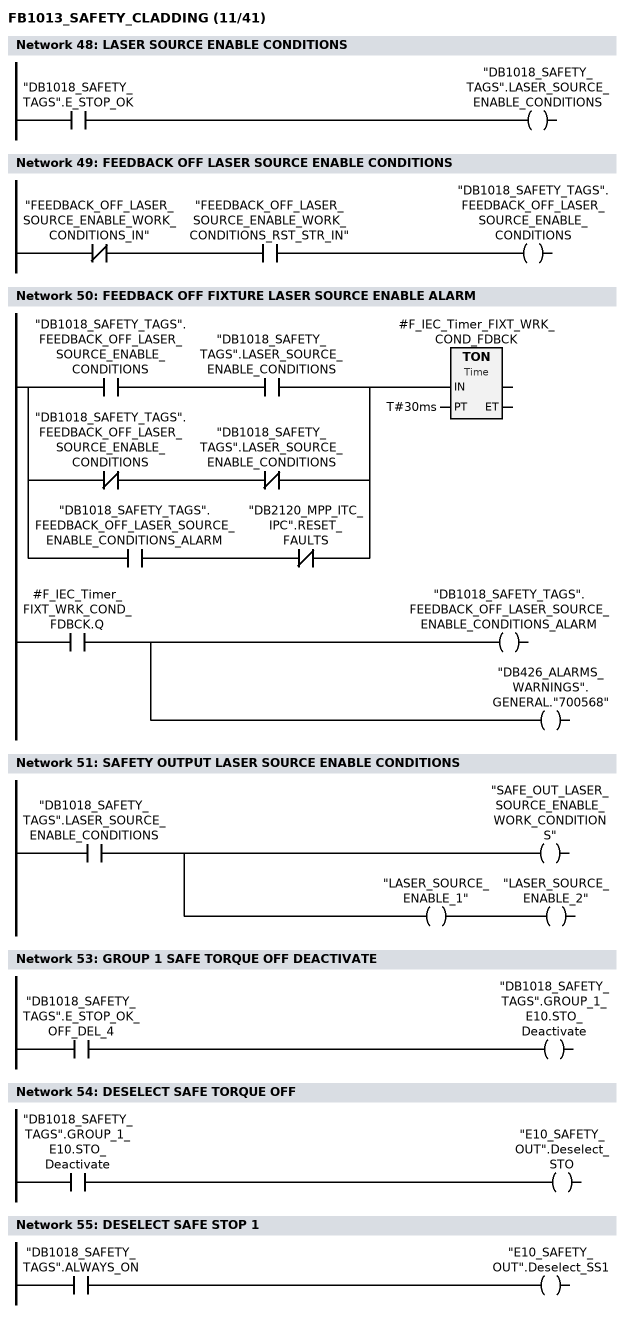
   RUNG wire#powerrail
      Contact( "DB1018_SAFETY_TAGS".E_STOP_OK )
      Coil( "DB1018_SAFETY_TAGS".LASER_SOURCE_ENABLE_CONDITIONS )
   END_RUNG
   // the same network as SCL:
   "DB1018_SAFETY_TAGS".LASER_SOURCE_ENABLE_CONDITIONS := "DB1018_SAFETY_TAGS".E_STOP_OK;
END_REGION

REGION Network 49: FEEDBACK OFF LASER SOURCE ENABLE CONDITIONS
   RUNG wire#powerrail
      I_Contact( "FEEDBACK_OFF_LASER_SOURCE_ENABLE_WORK_CONDITIONS_IN" )
      Contact( "FEEDBACK_OFF_LASER_SOURCE_ENABLE_WORK_CONDITIONS_RST_STR_IN" )
      Coil( "DB1018_SAFETY_TAGS".FEEDBACK_OFF_LASER_SOURCE_ENABLE_CONDITIONS )
   END_RUNG
   // the same network as SCL:
   "DB1018_SAFETY_TAGS".FEEDBACK_OFF_LASER_SOURCE_ENABLE_CONDITIONS := NOT "FEEDBACK_OFF_LASER_SOURCE_ENABLE_WORK_CONDITIONS_IN" AND "FEEDBACK_OFF_LASER_SOURCE_ENABLE_WORK_CONDITIONS_RST_STR_IN";
END_REGION

REGION Network 50: FEEDBACK OFF FIXTURE LASER SOURCE ENABLE ALARM
   RUNG wire#powerrail
      Contact( "DB1018_SAFETY_TAGS".FEEDBACK_OFF_LASER_SOURCE_ENABLE_CONDITIONS )
      Contact( "DB1018_SAFETY_TAGS".LASER_SOURCE_ENABLE_CONDITIONS )
      wire#w1
      { S7_Templates := "[time_type := Time, codedbool_type := DInt]" } #F_IEC_Timer_FIXT_WRK_COND_FDBCK.TON(pt := T#30ms, et =>)
   END_RUNG
   RUNG wire#powerrail
      I_Contact( "DB1018_SAFETY_TAGS".FEEDBACK_OFF_LASER_SOURCE_ENABLE_CONDITIONS )
      I_Contact( "DB1018_SAFETY_TAGS".LASER_SOURCE_ENABLE_CONDITIONS )
   END_RUNG wire#w1
   RUNG wire#powerrail
      Contact( "DB1018_SAFETY_TAGS".FEEDBACK_OFF_LASER_SOURCE_ENABLE_CONDITIONS_ALARM )
      I_Contact( "DB2120_MPP_ITC_IPC".RESET_FAULTS )
   END_RUNG wire#w1
   RUNG wire#powerrail
      Contact( #F_IEC_Timer_FIXT_WRK_COND_FDBCK.Q )
      wire#w2
      Coil( "DB1018_SAFETY_TAGS".FEEDBACK_OFF_LASER_SOURCE_ENABLE_CONDITIONS_ALARM )
   END_RUNG
   RUNG wire#w2
      Coil( "DB426_ALARMS_WARNINGS".GENERAL."700568" )
   END_RUNG
   // the same network as SCL:
   #F_IEC_Timer_FIXT_WRK_COND_FDBCK.TON(IN := ("DB1018_SAFETY_TAGS".FEEDBACK_OFF_LASER_SOURCE_ENABLE_CONDITIONS AND "DB1018_SAFETY_TAGS".LASER_SOURCE_ENABLE_CONDITIONS) OR (NOT "DB1018_SAFETY_TAGS".FEEDBACK_OFF_LASER_SOURCE_ENABLE_CONDITIONS AND NOT "DB1018_SAFETY_TAGS".LASER_SOURCE_ENABLE_CONDITIONS) OR ("DB1018_SAFETY_TAGS".FEEDBACK_OFF_LASER_SOURCE_ENABLE_CONDITIONS_ALARM AND NOT "DB2120_MPP_ITC_IPC".RESET_FAULTS),
                           PT := T#30ms);
   "DB1018_SAFETY_TAGS".FEEDBACK_OFF_LASER_SOURCE_ENABLE_CONDITIONS_ALARM := #F_IEC_Timer_FIXT_WRK_COND_FDBCK.Q;
   "DB426_ALARMS_WARNINGS".GENERAL."700568" := #F_IEC_Timer_FIXT_WRK_COND_FDBCK.Q;
END_REGION

REGION Network 51: SAFETY OUTPUT LASER SOURCE ENABLE CONDITIONS
   RUNG wire#powerrail
      Contact( "DB1018_SAFETY_TAGS".LASER_SOURCE_ENABLE_CONDITIONS )
      wire#w1
      Coil( "SAFE_OUT_LASER_SOURCE_ENABLE_WORK_CONDITIONS" )
   END_RUNG
   RUNG wire#w1
      Coil( "LASER_SOURCE_ENABLE_1" )
      Coil( "LASER_SOURCE_ENABLE_2" )
   END_RUNG
   // the same network as SCL:
   "SAFE_OUT_LASER_SOURCE_ENABLE_WORK_CONDITIONS" := "DB1018_SAFETY_TAGS".LASER_SOURCE_ENABLE_CONDITIONS;
   "LASER_SOURCE_ENABLE_1" := "DB1018_SAFETY_TAGS".LASER_SOURCE_ENABLE_CONDITIONS;
   "LASER_SOURCE_ENABLE_2" := "DB1018_SAFETY_TAGS".LASER_SOURCE_ENABLE_CONDITIONS;
END_REGION

REGION Network 52: *************** GROUP 1 - E10 ***************
END_REGION

REGION Network 53: GROUP 1 SAFE TORQUE OFF DEACTIVATE
   RUNG wire#powerrail
      Contact( "DB1018_SAFETY_TAGS".E_STOP_OK_OFF_DEL_4 )
      Coil( "DB1018_SAFETY_TAGS".GROUP_1_E10.STO_Deactivate )
   END_RUNG
   // the same network as SCL:
   "DB1018_SAFETY_TAGS".GROUP_1_E10.STO_Deactivate := "DB1018_SAFETY_TAGS".E_STOP_OK_OFF_DEL_4;
END_REGION

REGION Network 54: DESELECT SAFE TORQUE OFF
   RUNG wire#powerrail
      Contact( "DB1018_SAFETY_TAGS".GROUP_1_E10.STO_Deactivate )
      Coil( "E10_SAFETY_OUT".Deselect_STO )
   END_RUNG
   // the same network as SCL:
   "E10_SAFETY_OUT".Deselect_STO := "DB1018_SAFETY_TAGS".GROUP_1_E10.STO_Deactivate;
END_REGION

REGION Network 55: DESELECT SAFE STOP 1
   RUNG wire#powerrail
      Contact( "DB1018_SAFETY_TAGS".ALWAYS_ON )
      Coil( "E10_SAFETY_OUT".Deselect_SS1 )
   END_RUNG
   // the same network as SCL:
   "E10_SAFETY_OUT".Deselect_SS1 := "DB1018_SAFETY_TAGS".ALWAYS_ON;
END_REGION

REGION Network 56: GROUP 1 SAFE STOP 2 DEACTIVATE
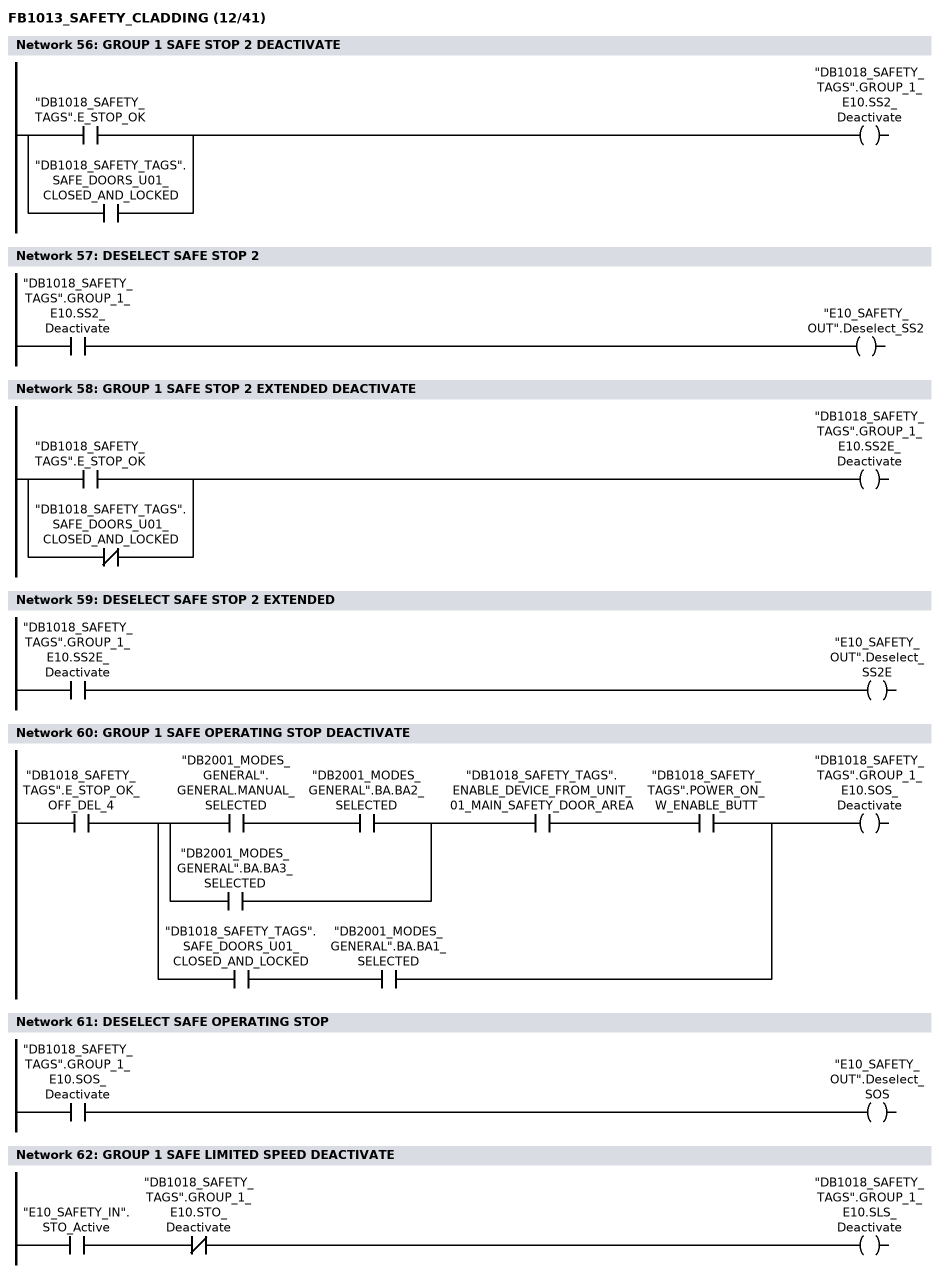
   RUNG wire#powerrail
      Contact( "DB1018_SAFETY_TAGS".E_STOP_OK )
      wire#w1
      Coil( "DB1018_SAFETY_TAGS".GROUP_1_E10.SS2_Deactivate )
   END_RUNG
   RUNG wire#powerrail
      Contact( "DB1018_SAFETY_TAGS".SAFE_DOORS_U01_CLOSED_AND_LOCKED )
   END_RUNG wire#w1
   // the same network as SCL:
   "DB1018_SAFETY_TAGS".GROUP_1_E10.SS2_Deactivate := "DB1018_SAFETY_TAGS".E_STOP_OK OR "DB1018_SAFETY_TAGS".SAFE_DOORS_U01_CLOSED_AND_LOCKED;
END_REGION

REGION Network 57: DESELECT SAFE STOP 2
   RUNG wire#powerrail
      Contact( "DB1018_SAFETY_TAGS".GROUP_1_E10.SS2_Deactivate )
      Coil( "E10_SAFETY_OUT".Deselect_SS2 )
   END_RUNG
   // the same network as SCL:
   "E10_SAFETY_OUT".Deselect_SS2 := "DB1018_SAFETY_TAGS".GROUP_1_E10.SS2_Deactivate;
END_REGION

REGION Network 58: GROUP 1 SAFE STOP 2 EXTENDED DEACTIVATE
   RUNG wire#powerrail
      Contact( "DB1018_SAFETY_TAGS".E_STOP_OK )
      wire#w1
      Coil( "DB1018_SAFETY_TAGS".GROUP_1_E10.SS2E_Deactivate )
   END_RUNG
   RUNG wire#powerrail
      I_Contact( "DB1018_SAFETY_TAGS".SAFE_DOORS_U01_CLOSED_AND_LOCKED )
   END_RUNG wire#w1
   // the same network as SCL:
   "DB1018_SAFETY_TAGS".GROUP_1_E10.SS2E_Deactivate := "DB1018_SAFETY_TAGS".E_STOP_OK OR NOT "DB1018_SAFETY_TAGS".SAFE_DOORS_U01_CLOSED_AND_LOCKED;
END_REGION

REGION Network 59: DESELECT SAFE STOP 2 EXTENDED
   RUNG wire#powerrail
      Contact( "DB1018_SAFETY_TAGS".GROUP_1_E10.SS2E_Deactivate )
      Coil( "E10_SAFETY_OUT".Deselect_SS2E )
   END_RUNG
   // the same network as SCL:
   "E10_SAFETY_OUT".Deselect_SS2E := "DB1018_SAFETY_TAGS".GROUP_1_E10.SS2E_Deactivate;
END_REGION

REGION Network 60: GROUP 1 SAFE OPERATING STOP DEACTIVATE
   RUNG wire#powerrail
      Contact( "DB1018_SAFETY_TAGS".E_STOP_OK_OFF_DEL_4 )
      wire#w1
      Contact( "DB2001_MODES_GENERAL".GENERAL.MANUAL_SELECTED )
      Contact( "DB2001_MODES_GENERAL".BA.BA2_SELECTED )
      wire#w2
      Contact( "DB1018_SAFETY_TAGS".ENABLE_DEVICE_FROM_UNIT_01_MAIN_SAFETY_DOOR_AREA )
      Contact( "DB1018_SAFETY_TAGS".POWER_ON_W_ENABLE_BUTT )
      wire#w3
      Coil( "DB1018_SAFETY_TAGS".GROUP_1_E10.SOS_Deactivate )
   END_RUNG
   RUNG wire#w1
      Contact( "DB2001_MODES_GENERAL".BA.BA3_SELECTED )
   END_RUNG wire#w2
   RUNG wire#w1
      Contact( "DB1018_SAFETY_TAGS".SAFE_DOORS_U01_CLOSED_AND_LOCKED )
      Contact( "DB2001_MODES_GENERAL".BA.BA1_SELECTED )
   END_RUNG wire#w3
   // the same network as SCL:
   "DB1018_SAFETY_TAGS".GROUP_1_E10.SOS_Deactivate := "DB1018_SAFETY_TAGS".E_STOP_OK_OFF_DEL_4 AND (((("DB2001_MODES_GENERAL".GENERAL.MANUAL_SELECTED AND "DB2001_MODES_GENERAL".BA.BA2_SELECTED) OR "DB2001_MODES_GENERAL".BA.BA3_SELECTED) AND "DB1018_SAFETY_TAGS".ENABLE_DEVICE_FROM_UNIT_01_MAIN_SAFETY_DOOR_AREA AND "DB1018_SAFETY_TAGS".POWER_ON_W_ENABLE_BUTT) OR ("DB1018_SAFETY_TAGS".SAFE_DOORS_U01_CLOSED_AND_LOCKED AND "DB2001_MODES_GENERAL".BA.BA1_SELECTED));
END_REGION

REGION Network 61: DESELECT SAFE OPERATING STOP
   RUNG wire#powerrail
      Contact( "DB1018_SAFETY_TAGS".GROUP_1_E10.SOS_Deactivate )
      Coil( "E10_SAFETY_OUT".Deselect_SOS )
   END_RUNG
   // the same network as SCL:
   "E10_SAFETY_OUT".Deselect_SOS := "DB1018_SAFETY_TAGS".GROUP_1_E10.SOS_Deactivate;
END_REGION

REGION Network 62: GROUP 1 SAFE LIMITED SPEED DEACTIVATE
   RUNG wire#powerrail
      Contact( "E10_SAFETY_IN".STO_Active )
      I_Contact( "DB1018_SAFETY_TAGS".GROUP_1_E10.STO_Deactivate )
      Coil( "DB1018_SAFETY_TAGS".GROUP_1_E10.SLS_Deactivate )
   END_RUNG
   // the same network as SCL:
   "DB1018_SAFETY_TAGS".GROUP_1_E10.SLS_Deactivate := "E10_SAFETY_IN".STO_Active AND NOT "DB1018_SAFETY_TAGS".GROUP_1_E10.STO_Deactivate;
END_REGION

REGION Network 63: DESELECT SAFE LIMITED SPEED
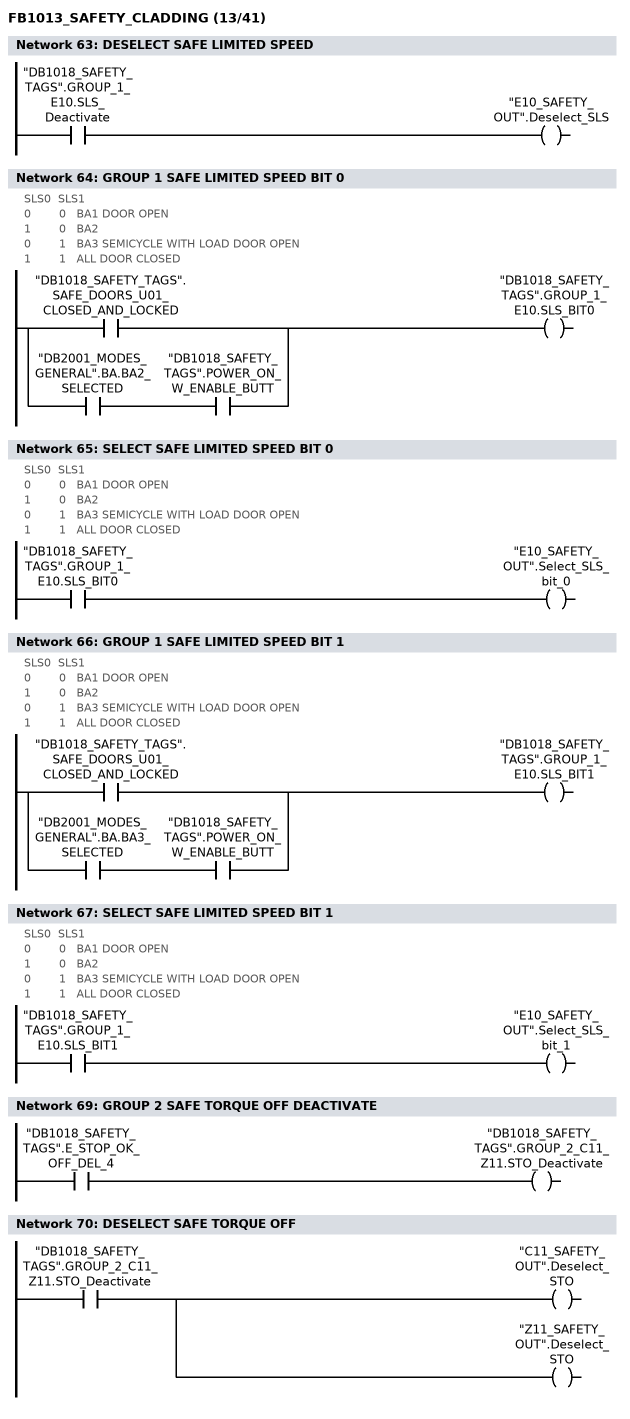
   RUNG wire#powerrail
      Contact( "DB1018_SAFETY_TAGS".GROUP_1_E10.SLS_Deactivate )
      Coil( "E10_SAFETY_OUT".Deselect_SLS )
   END_RUNG
   // the same network as SCL:
   "E10_SAFETY_OUT".Deselect_SLS := "DB1018_SAFETY_TAGS".GROUP_1_E10.SLS_Deactivate;
END_REGION

REGION Network 64: GROUP 1 SAFE LIMITED SPEED BIT 0
   // SLS0  SLS1
   //    0        0   BA1 DOOR OPEN
   //    1        0   BA2
   //    0        1   BA3 SEMICYCLE WITH LOAD DOOR OPEN
   //    1        1   ALL DOOR CLOSED
   RUNG wire#powerrail
      Contact( "DB1018_SAFETY_TAGS".SAFE_DOORS_U01_CLOSED_AND_LOCKED )
      wire#w1
      Coil( "DB1018_SAFETY_TAGS".GROUP_1_E10.SLS_BIT0 )
   END_RUNG
   RUNG wire#powerrail
      Contact( "DB2001_MODES_GENERAL".BA.BA2_SELECTED )
      Contact( "DB1018_SAFETY_TAGS".POWER_ON_W_ENABLE_BUTT )
   END_RUNG wire#w1
   // the same network as SCL:
   "DB1018_SAFETY_TAGS".GROUP_1_E10.SLS_BIT0 := "DB1018_SAFETY_TAGS".SAFE_DOORS_U01_CLOSED_AND_LOCKED OR ("DB2001_MODES_GENERAL".BA.BA2_SELECTED AND "DB1018_SAFETY_TAGS".POWER_ON_W_ENABLE_BUTT);
END_REGION

REGION Network 65: SELECT SAFE LIMITED SPEED BIT 0
   // SLS0  SLS1
   //    0        0   BA1 DOOR OPEN
   //    1        0   BA2
   //    0        1   BA3 SEMICYCLE WITH LOAD DOOR OPEN
   //    1        1   ALL DOOR CLOSED
   RUNG wire#powerrail
      Contact( "DB1018_SAFETY_TAGS".GROUP_1_E10.SLS_BIT0 )
      Coil( "E10_SAFETY_OUT".Select_SLS_bit_0 )
   END_RUNG
   // the same network as SCL:
   "E10_SAFETY_OUT".Select_SLS_bit_0 := "DB1018_SAFETY_TAGS".GROUP_1_E10.SLS_BIT0;
END_REGION

REGION Network 66: GROUP 1 SAFE LIMITED SPEED BIT 1
   // SLS0  SLS1
   //    0        0   BA1 DOOR OPEN
   //    1        0   BA2
   //    0        1   BA3 SEMICYCLE WITH LOAD DOOR OPEN
   //    1        1   ALL DOOR CLOSED
   RUNG wire#powerrail
      Contact( "DB1018_SAFETY_TAGS".SAFE_DOORS_U01_CLOSED_AND_LOCKED )
      wire#w1
      Coil( "DB1018_SAFETY_TAGS".GROUP_1_E10.SLS_BIT1 )
   END_RUNG
   RUNG wire#powerrail
      Contact( "DB2001_MODES_GENERAL".BA.BA3_SELECTED )
      Contact( "DB1018_SAFETY_TAGS".POWER_ON_W_ENABLE_BUTT )
   END_RUNG wire#w1
   // the same network as SCL:
   "DB1018_SAFETY_TAGS".GROUP_1_E10.SLS_BIT1 := "DB1018_SAFETY_TAGS".SAFE_DOORS_U01_CLOSED_AND_LOCKED OR ("DB2001_MODES_GENERAL".BA.BA3_SELECTED AND "DB1018_SAFETY_TAGS".POWER_ON_W_ENABLE_BUTT);
END_REGION

REGION Network 67: SELECT SAFE LIMITED SPEED BIT 1
   // SLS0  SLS1
   //    0        0   BA1 DOOR OPEN
   //    1        0   BA2
   //    0        1   BA3 SEMICYCLE WITH LOAD DOOR OPEN
   //    1        1   ALL DOOR CLOSED
   RUNG wire#powerrail
      Contact( "DB1018_SAFETY_TAGS".GROUP_1_E10.SLS_BIT1 )
      Coil( "E10_SAFETY_OUT".Select_SLS_bit_1 )
   END_RUNG
   // the same network as SCL:
   "E10_SAFETY_OUT".Select_SLS_bit_1 := "DB1018_SAFETY_TAGS".GROUP_1_E10.SLS_BIT1;
END_REGION

REGION Network 68: *************** GROUP 2 - C11 / W11 ***************
END_REGION

REGION Network 69: GROUP 2 SAFE TORQUE OFF DEACTIVATE
   RUNG wire#powerrail
      Contact( "DB1018_SAFETY_TAGS".E_STOP_OK_OFF_DEL_4 )
      Coil( "DB1018_SAFETY_TAGS".GROUP_2_C11_Z11.STO_Deactivate )
   END_RUNG
   // the same network as SCL:
   "DB1018_SAFETY_TAGS".GROUP_2_C11_Z11.STO_Deactivate := "DB1018_SAFETY_TAGS".E_STOP_OK_OFF_DEL_4;
END_REGION

REGION Network 70: DESELECT SAFE TORQUE OFF
   RUNG wire#powerrail
      Contact( "DB1018_SAFETY_TAGS".GROUP_2_C11_Z11.STO_Deactivate )
      wire#w1
      Coil( "C11_SAFETY_OUT".Deselect_STO )
   END_RUNG
   RUNG wire#w1
      Coil( "Z11_SAFETY_OUT".Deselect_STO )
   END_RUNG
   // the same network as SCL:
   "C11_SAFETY_OUT".Deselect_STO := "DB1018_SAFETY_TAGS".GROUP_2_C11_Z11.STO_Deactivate;
   "Z11_SAFETY_OUT".Deselect_STO := "DB1018_SAFETY_TAGS".GROUP_2_C11_Z11.STO_Deactivate;
END_REGION

REGION Network 71: DESELECT SAFE STOP 1
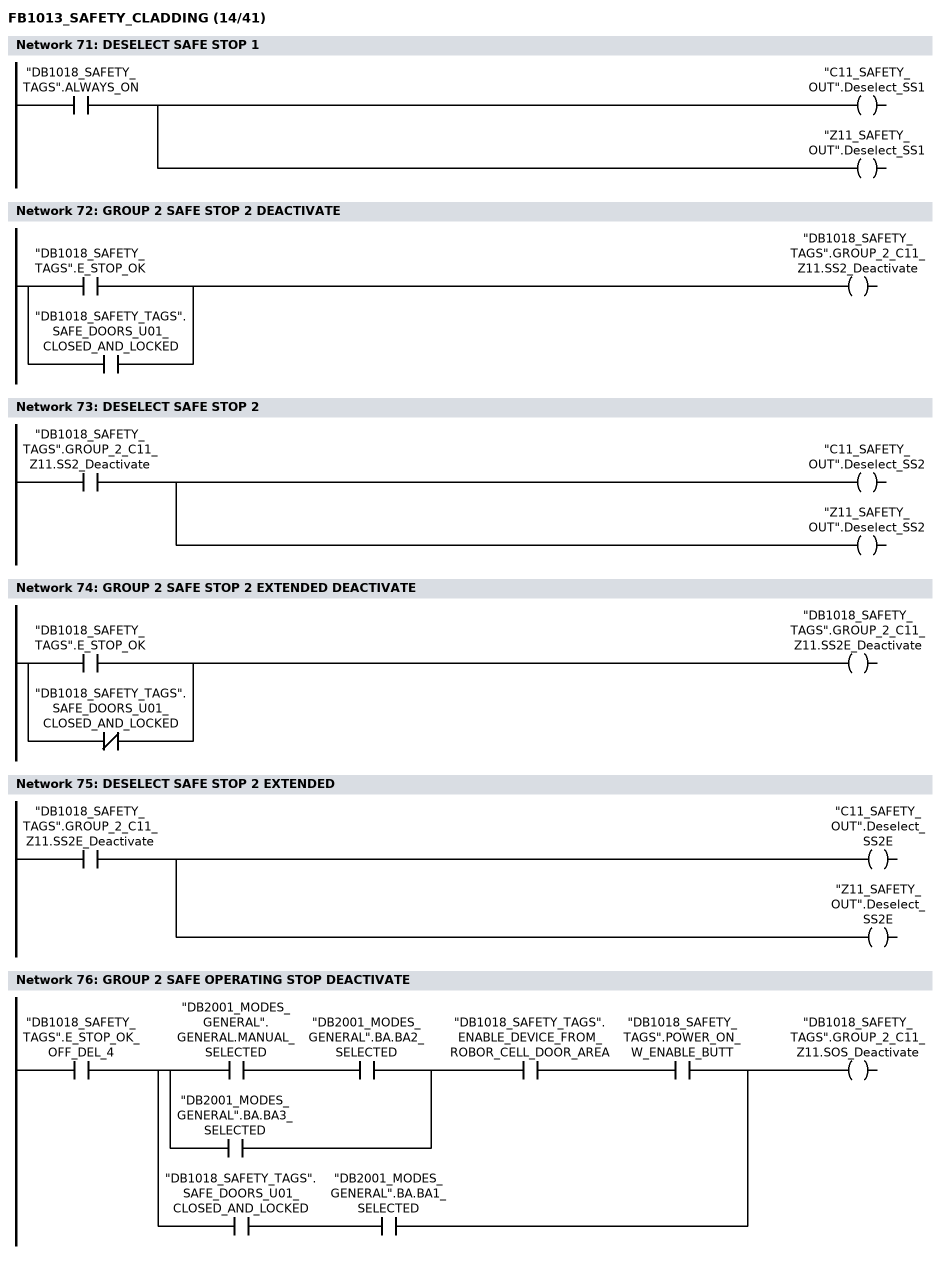
   RUNG wire#powerrail
      Contact( "DB1018_SAFETY_TAGS".ALWAYS_ON )
      wire#w1
      Coil( "C11_SAFETY_OUT".Deselect_SS1 )
   END_RUNG
   RUNG wire#w1
      Coil( "Z11_SAFETY_OUT".Deselect_SS1 )
   END_RUNG
   // the same network as SCL:
   "C11_SAFETY_OUT".Deselect_SS1 := "DB1018_SAFETY_TAGS".ALWAYS_ON;
   "Z11_SAFETY_OUT".Deselect_SS1 := "DB1018_SAFETY_TAGS".ALWAYS_ON;
END_REGION

REGION Network 72: GROUP 2 SAFE STOP 2 DEACTIVATE
   RUNG wire#powerrail
      Contact( "DB1018_SAFETY_TAGS".E_STOP_OK )
      wire#w1
      Coil( "DB1018_SAFETY_TAGS".GROUP_2_C11_Z11.SS2_Deactivate )
   END_RUNG
   RUNG wire#powerrail
      Contact( "DB1018_SAFETY_TAGS".SAFE_DOORS_U01_CLOSED_AND_LOCKED )
   END_RUNG wire#w1
   // the same network as SCL:
   "DB1018_SAFETY_TAGS".GROUP_2_C11_Z11.SS2_Deactivate := "DB1018_SAFETY_TAGS".E_STOP_OK OR "DB1018_SAFETY_TAGS".SAFE_DOORS_U01_CLOSED_AND_LOCKED;
END_REGION

REGION Network 73: DESELECT SAFE STOP 2
   RUNG wire#powerrail
      Contact( "DB1018_SAFETY_TAGS".GROUP_2_C11_Z11.SS2_Deactivate )
      wire#w1
      Coil( "C11_SAFETY_OUT".Deselect_SS2 )
   END_RUNG
   RUNG wire#w1
      Coil( "Z11_SAFETY_OUT".Deselect_SS2 )
   END_RUNG
   // the same network as SCL:
   "C11_SAFETY_OUT".Deselect_SS2 := "DB1018_SAFETY_TAGS".GROUP_2_C11_Z11.SS2_Deactivate;
   "Z11_SAFETY_OUT".Deselect_SS2 := "DB1018_SAFETY_TAGS".GROUP_2_C11_Z11.SS2_Deactivate;
END_REGION

REGION Network 74: GROUP 2 SAFE STOP 2 EXTENDED DEACTIVATE
   RUNG wire#powerrail
      Contact( "DB1018_SAFETY_TAGS".E_STOP_OK )
      wire#w1
      Coil( "DB1018_SAFETY_TAGS".GROUP_2_C11_Z11.SS2E_Deactivate )
   END_RUNG
   RUNG wire#powerrail
      I_Contact( "DB1018_SAFETY_TAGS".SAFE_DOORS_U01_CLOSED_AND_LOCKED )
   END_RUNG wire#w1
   // the same network as SCL:
   "DB1018_SAFETY_TAGS".GROUP_2_C11_Z11.SS2E_Deactivate := "DB1018_SAFETY_TAGS".E_STOP_OK OR NOT "DB1018_SAFETY_TAGS".SAFE_DOORS_U01_CLOSED_AND_LOCKED;
END_REGION

REGION Network 75: DESELECT SAFE STOP 2 EXTENDED
   RUNG wire#powerrail
      Contact( "DB1018_SAFETY_TAGS".GROUP_2_C11_Z11.SS2E_Deactivate )
      wire#w1
      Coil( "C11_SAFETY_OUT".Deselect_SS2E )
   END_RUNG
   RUNG wire#w1
      Coil( "Z11_SAFETY_OUT".Deselect_SS2E )
   END_RUNG
   // the same network as SCL:
   "C11_SAFETY_OUT".Deselect_SS2E := "DB1018_SAFETY_TAGS".GROUP_2_C11_Z11.SS2E_Deactivate;
   "Z11_SAFETY_OUT".Deselect_SS2E := "DB1018_SAFETY_TAGS".GROUP_2_C11_Z11.SS2E_Deactivate;
END_REGION

REGION Network 76: GROUP 2 SAFE OPERATING STOP DEACTIVATE
   RUNG wire#powerrail
      Contact( "DB1018_SAFETY_TAGS".E_STOP_OK_OFF_DEL_4 )
      wire#w1
      Contact( "DB2001_MODES_GENERAL".GENERAL.MANUAL_SELECTED )
      Contact( "DB2001_MODES_GENERAL".BA.BA2_SELECTED )
      wire#w2
      Contact( "DB1018_SAFETY_TAGS".ENABLE_DEVICE_FROM_ROBOR_CELL_DOOR_AREA )
      Contact( "DB1018_SAFETY_TAGS".POWER_ON_W_ENABLE_BUTT )
      wire#w3
      Coil( "DB1018_SAFETY_TAGS".GROUP_2_C11_Z11.SOS_Deactivate )
   END_RUNG
   RUNG wire#w1
      Contact( "DB2001_MODES_GENERAL".BA.BA3_SELECTED )
   END_RUNG wire#w2
   RUNG wire#w1
      Contact( "DB1018_SAFETY_TAGS".SAFE_DOORS_U01_CLOSED_AND_LOCKED )
      Contact( "DB2001_MODES_GENERAL".BA.BA1_SELECTED )
   END_RUNG wire#w3
   // the same network as SCL:
   "DB1018_SAFETY_TAGS".GROUP_2_C11_Z11.SOS_Deactivate := "DB1018_SAFETY_TAGS".E_STOP_OK_OFF_DEL_4 AND (((("DB2001_MODES_GENERAL".GENERAL.MANUAL_SELECTED AND "DB2001_MODES_GENERAL".BA.BA2_SELECTED) OR "DB2001_MODES_GENERAL".BA.BA3_SELECTED) AND "DB1018_SAFETY_TAGS".ENABLE_DEVICE_FROM_ROBOR_CELL_DOOR_AREA AND "DB1018_SAFETY_TAGS".POWER_ON_W_ENABLE_BUTT) OR ("DB1018_SAFETY_TAGS".SAFE_DOORS_U01_CLOSED_AND_LOCKED AND "DB2001_MODES_GENERAL".BA.BA1_SELECTED));
END_REGION

REGION Network 77: DESELECT SAFE OPERATING STOP
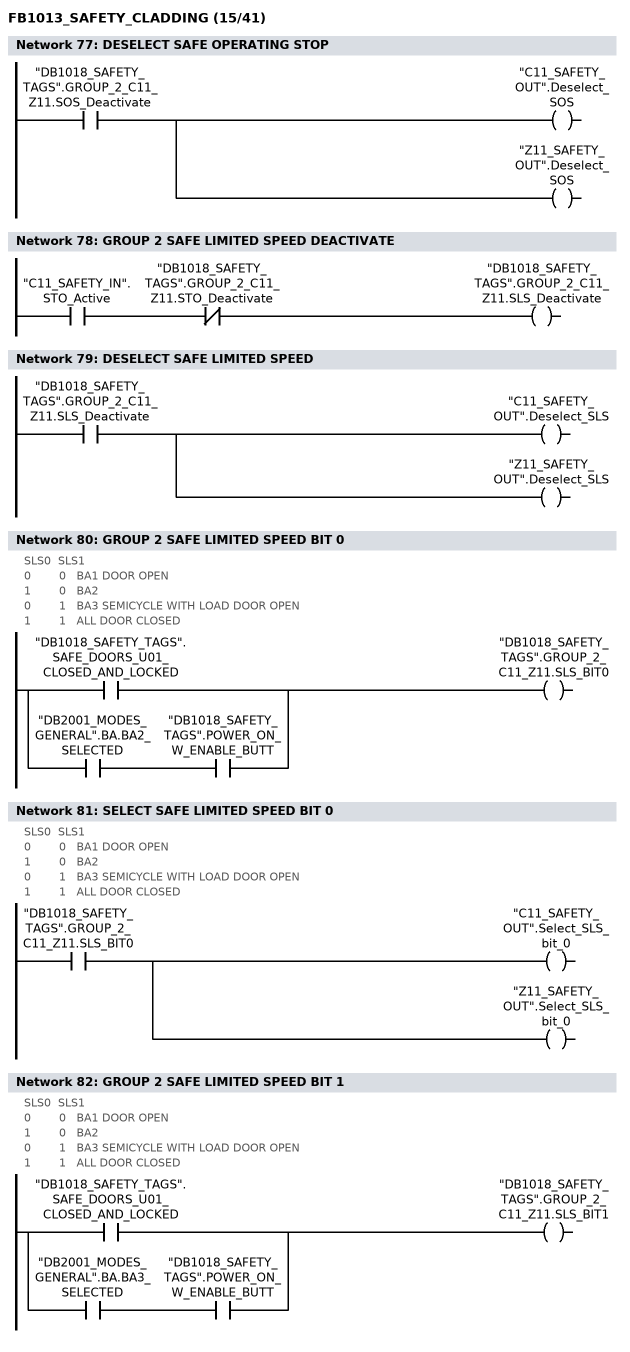
   RUNG wire#powerrail
      Contact( "DB1018_SAFETY_TAGS".GROUP_2_C11_Z11.SOS_Deactivate )
      wire#w1
      Coil( "C11_SAFETY_OUT".Deselect_SOS )
   END_RUNG
   RUNG wire#w1
      Coil( "Z11_SAFETY_OUT".Deselect_SOS )
   END_RUNG
   // the same network as SCL:
   "C11_SAFETY_OUT".Deselect_SOS := "DB1018_SAFETY_TAGS".GROUP_2_C11_Z11.SOS_Deactivate;
   "Z11_SAFETY_OUT".Deselect_SOS := "DB1018_SAFETY_TAGS".GROUP_2_C11_Z11.SOS_Deactivate;
END_REGION

REGION Network 78: GROUP 2 SAFE LIMITED SPEED DEACTIVATE
   RUNG wire#powerrail
      Contact( "C11_SAFETY_IN".STO_Active )
      I_Contact( "DB1018_SAFETY_TAGS".GROUP_2_C11_Z11.STO_Deactivate )
      Coil( "DB1018_SAFETY_TAGS".GROUP_2_C11_Z11.SLS_Deactivate )
   END_RUNG
   // the same network as SCL:
   "DB1018_SAFETY_TAGS".GROUP_2_C11_Z11.SLS_Deactivate := "C11_SAFETY_IN".STO_Active AND NOT "DB1018_SAFETY_TAGS".GROUP_2_C11_Z11.STO_Deactivate;
END_REGION

REGION Network 79: DESELECT SAFE LIMITED SPEED
   RUNG wire#powerrail
      Contact( "DB1018_SAFETY_TAGS".GROUP_2_C11_Z11.SLS_Deactivate )
      wire#w1
      Coil( "C11_SAFETY_OUT".Deselect_SLS )
   END_RUNG
   RUNG wire#w1
      Coil( "Z11_SAFETY_OUT".Deselect_SLS )
   END_RUNG
   // the same network as SCL:
   "C11_SAFETY_OUT".Deselect_SLS := "DB1018_SAFETY_TAGS".GROUP_2_C11_Z11.SLS_Deactivate;
   "Z11_SAFETY_OUT".Deselect_SLS := "DB1018_SAFETY_TAGS".GROUP_2_C11_Z11.SLS_Deactivate;
END_REGION

REGION Network 80: GROUP 2 SAFE LIMITED SPEED BIT 0
   // SLS0  SLS1
   //    0        0   BA1 DOOR OPEN
   //    1        0   BA2
   //    0        1   BA3 SEMICYCLE WITH LOAD DOOR OPEN
   //    1        1   ALL DOOR CLOSED
   RUNG wire#powerrail
      Contact( "DB1018_SAFETY_TAGS".SAFE_DOORS_U01_CLOSED_AND_LOCKED )
      wire#w1
      Coil( "DB1018_SAFETY_TAGS".GROUP_2_C11_Z11.SLS_BIT0 )
   END_RUNG
   RUNG wire#powerrail
      Contact( "DB2001_MODES_GENERAL".BA.BA2_SELECTED )
      Contact( "DB1018_SAFETY_TAGS".POWER_ON_W_ENABLE_BUTT )
   END_RUNG wire#w1
   // the same network as SCL:
   "DB1018_SAFETY_TAGS".GROUP_2_C11_Z11.SLS_BIT0 := "DB1018_SAFETY_TAGS".SAFE_DOORS_U01_CLOSED_AND_LOCKED OR ("DB2001_MODES_GENERAL".BA.BA2_SELECTED AND "DB1018_SAFETY_TAGS".POWER_ON_W_ENABLE_BUTT);
END_REGION

REGION Network 81: SELECT SAFE LIMITED SPEED BIT 0
   // SLS0  SLS1
   //    0        0   BA1 DOOR OPEN
   //    1        0   BA2
   //    0        1   BA3 SEMICYCLE WITH LOAD DOOR OPEN
   //    1        1   ALL DOOR CLOSED
   RUNG wire#powerrail
      Contact( "DB1018_SAFETY_TAGS".GROUP_2_C11_Z11.SLS_BIT0 )
      wire#w1
      Coil( "C11_SAFETY_OUT".Select_SLS_bit_0 )
   END_RUNG
   RUNG wire#w1
      Coil( "Z11_SAFETY_OUT".Select_SLS_bit_0 )
   END_RUNG
   // the same network as SCL:
   "C11_SAFETY_OUT".Select_SLS_bit_0 := "DB1018_SAFETY_TAGS".GROUP_2_C11_Z11.SLS_BIT0;
   "Z11_SAFETY_OUT".Select_SLS_bit_0 := "DB1018_SAFETY_TAGS".GROUP_2_C11_Z11.SLS_BIT0;
END_REGION

REGION Network 82: GROUP 2 SAFE LIMITED SPEED BIT 1
   // SLS0  SLS1
   //    0        0   BA1 DOOR OPEN
   //    1        0   BA2
   //    0        1   BA3 SEMICYCLE WITH LOAD DOOR OPEN
   //    1        1   ALL DOOR CLOSED
   RUNG wire#powerrail
      Contact( "DB1018_SAFETY_TAGS".SAFE_DOORS_U01_CLOSED_AND_LOCKED )
      wire#w1
      Coil( "DB1018_SAFETY_TAGS".GROUP_2_C11_Z11.SLS_BIT1 )
   END_RUNG
   RUNG wire#powerrail
      Contact( "DB2001_MODES_GENERAL".BA.BA3_SELECTED )
      Contact( "DB1018_SAFETY_TAGS".POWER_ON_W_ENABLE_BUTT )
   END_RUNG wire#w1
   // the same network as SCL:
   "DB1018_SAFETY_TAGS".GROUP_2_C11_Z11.SLS_BIT1 := "DB1018_SAFETY_TAGS".SAFE_DOORS_U01_CLOSED_AND_LOCKED OR ("DB2001_MODES_GENERAL".BA.BA3_SELECTED AND "DB1018_SAFETY_TAGS".POWER_ON_W_ENABLE_BUTT);
END_REGION

REGION Network 83: SELECT SAFE LIMITED SPEED BIT 1
   // SLS0  SLS1
   //    0        0   BA1 DOOR OPEN
   //    1        0   BA2
   //    0        1   BA3 SEMICYCLE WITH LOAD DOOR OPEN
   //    1        1   ALL DOOR CLOSED
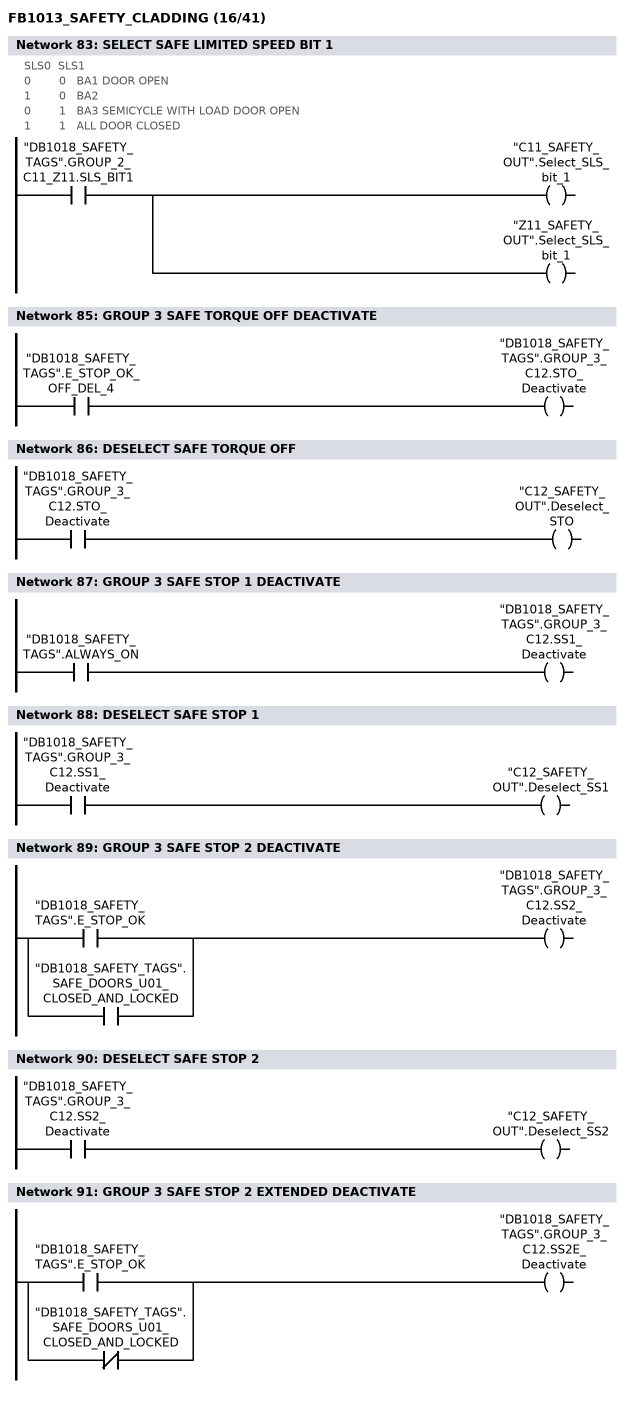
   RUNG wire#powerrail
      Contact( "DB1018_SAFETY_TAGS".GROUP_2_C11_Z11.SLS_BIT1 )
      wire#w1
      Coil( "C11_SAFETY_OUT".Select_SLS_bit_1 )
   END_RUNG
   RUNG wire#w1
      Coil( "Z11_SAFETY_OUT".Select_SLS_bit_1 )
   END_RUNG
   // the same network as SCL:
   "C11_SAFETY_OUT".Select_SLS_bit_1 := "DB1018_SAFETY_TAGS".GROUP_2_C11_Z11.SLS_BIT1;
   "Z11_SAFETY_OUT".Select_SLS_bit_1 := "DB1018_SAFETY_TAGS".GROUP_2_C11_Z11.SLS_BIT1;
END_REGION

REGION Network 84: *************** GROUP 3 - C12 ***************
END_REGION

REGION Network 85: GROUP 3 SAFE TORQUE OFF DEACTIVATE
   RUNG wire#powerrail
      Contact( "DB1018_SAFETY_TAGS".E_STOP_OK_OFF_DEL_4 )
      Coil( "DB1018_SAFETY_TAGS".GROUP_3_C12.STO_Deactivate )
   END_RUNG
   // the same network as SCL:
   "DB1018_SAFETY_TAGS".GROUP_3_C12.STO_Deactivate := "DB1018_SAFETY_TAGS".E_STOP_OK_OFF_DEL_4;
END_REGION

REGION Network 86: DESELECT SAFE TORQUE OFF
   RUNG wire#powerrail
      Contact( "DB1018_SAFETY_TAGS".GROUP_3_C12.STO_Deactivate )
      Coil( "C12_SAFETY_OUT".Deselect_STO )
   END_RUNG
   // the same network as SCL:
   "C12_SAFETY_OUT".Deselect_STO := "DB1018_SAFETY_TAGS".GROUP_3_C12.STO_Deactivate;
END_REGION

REGION Network 87: GROUP 3 SAFE STOP 1 DEACTIVATE
   RUNG wire#powerrail
      Contact( "DB1018_SAFETY_TAGS".ALWAYS_ON )
      Coil( "DB1018_SAFETY_TAGS".GROUP_3_C12.SS1_Deactivate )
   END_RUNG
   // the same network as SCL:
   "DB1018_SAFETY_TAGS".GROUP_3_C12.SS1_Deactivate := "DB1018_SAFETY_TAGS".ALWAYS_ON;
END_REGION

REGION Network 88: DESELECT SAFE STOP 1
   RUNG wire#powerrail
      Contact( "DB1018_SAFETY_TAGS".GROUP_3_C12.SS1_Deactivate )
      Coil( "C12_SAFETY_OUT".Deselect_SS1 )
   END_RUNG
   // the same network as SCL:
   "C12_SAFETY_OUT".Deselect_SS1 := "DB1018_SAFETY_TAGS".GROUP_3_C12.SS1_Deactivate;
END_REGION

REGION Network 89: GROUP 3 SAFE STOP 2 DEACTIVATE
   RUNG wire#powerrail
      Contact( "DB1018_SAFETY_TAGS".E_STOP_OK )
      wire#w1
      Coil( "DB1018_SAFETY_TAGS".GROUP_3_C12.SS2_Deactivate )
   END_RUNG
   RUNG wire#powerrail
      Contact( "DB1018_SAFETY_TAGS".SAFE_DOORS_U01_CLOSED_AND_LOCKED )
   END_RUNG wire#w1
   // the same network as SCL:
   "DB1018_SAFETY_TAGS".GROUP_3_C12.SS2_Deactivate := "DB1018_SAFETY_TAGS".E_STOP_OK OR "DB1018_SAFETY_TAGS".SAFE_DOORS_U01_CLOSED_AND_LOCKED;
END_REGION

REGION Network 90: DESELECT SAFE STOP 2
   RUNG wire#powerrail
      Contact( "DB1018_SAFETY_TAGS".GROUP_3_C12.SS2_Deactivate )
      Coil( "C12_SAFETY_OUT".Deselect_SS2 )
   END_RUNG
   // the same network as SCL:
   "C12_SAFETY_OUT".Deselect_SS2 := "DB1018_SAFETY_TAGS".GROUP_3_C12.SS2_Deactivate;
END_REGION

REGION Network 91: GROUP 3 SAFE STOP 2 EXTENDED DEACTIVATE
   RUNG wire#powerrail
      Contact( "DB1018_SAFETY_TAGS".E_STOP_OK )
      wire#w1
      Coil( "DB1018_SAFETY_TAGS".GROUP_3_C12.SS2E_Deactivate )
   END_RUNG
   RUNG wire#powerrail
      I_Contact( "DB1018_SAFETY_TAGS".SAFE_DOORS_U01_CLOSED_AND_LOCKED )
   END_RUNG wire#w1
   // the same network as SCL:
   "DB1018_SAFETY_TAGS".GROUP_3_C12.SS2E_Deactivate := "DB1018_SAFETY_TAGS".E_STOP_OK OR NOT "DB1018_SAFETY_TAGS".SAFE_DOORS_U01_CLOSED_AND_LOCKED;
END_REGION

REGION Network 92: DESELECT SAFE STOP 2 EXTENDED
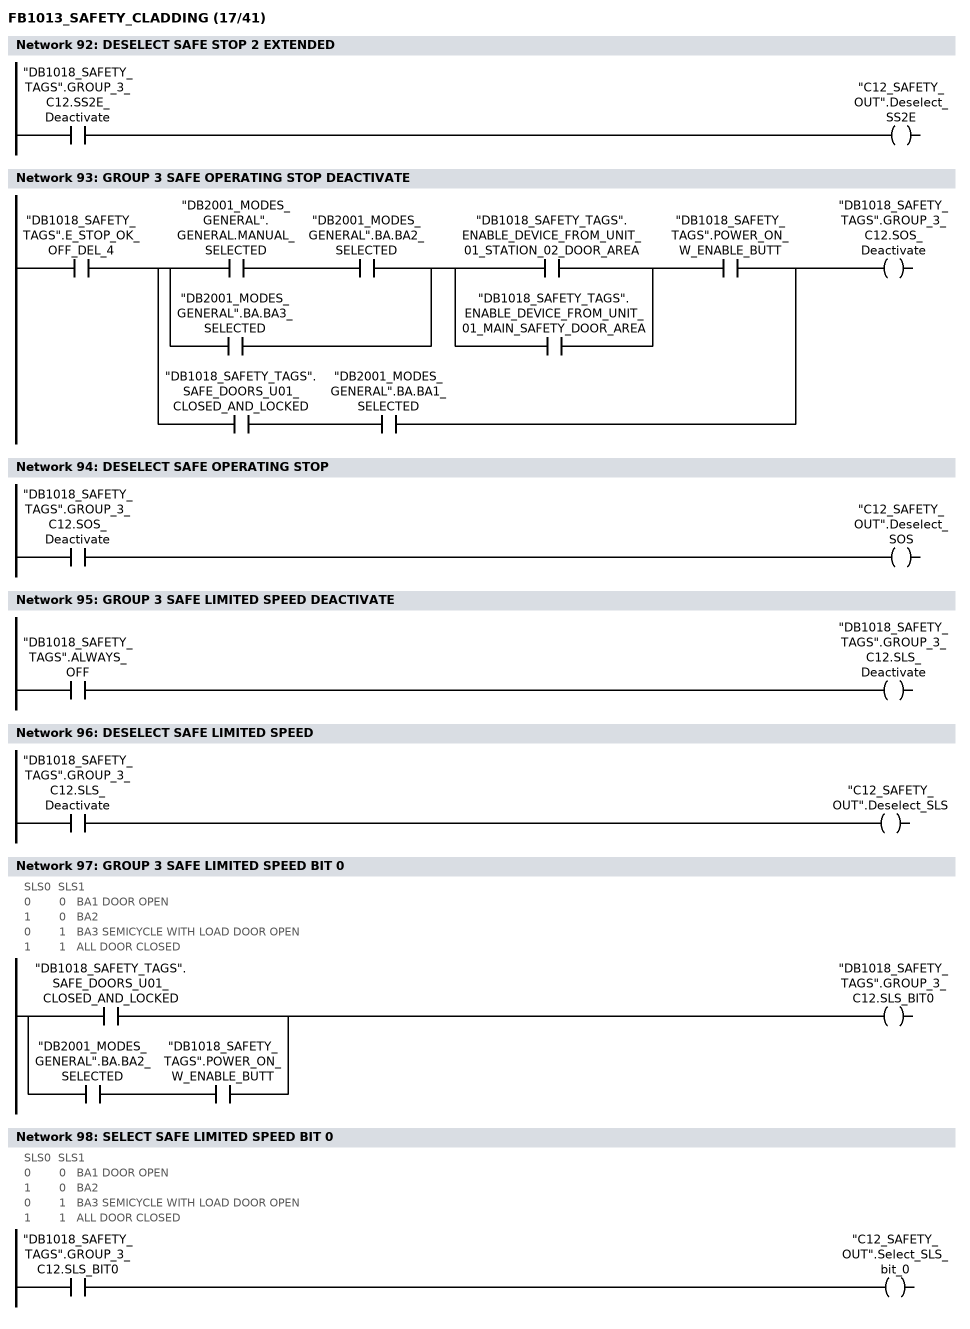
   RUNG wire#powerrail
      Contact( "DB1018_SAFETY_TAGS".GROUP_3_C12.SS2E_Deactivate )
      Coil( "C12_SAFETY_OUT".Deselect_SS2E )
   END_RUNG
   // the same network as SCL:
   "C12_SAFETY_OUT".Deselect_SS2E := "DB1018_SAFETY_TAGS".GROUP_3_C12.SS2E_Deactivate;
END_REGION

REGION Network 93: GROUP 3 SAFE OPERATING STOP DEACTIVATE
   RUNG wire#powerrail
      Contact( "DB1018_SAFETY_TAGS".E_STOP_OK_OFF_DEL_4 )
      wire#w1
      Contact( "DB2001_MODES_GENERAL".GENERAL.MANUAL_SELECTED )
      Contact( "DB2001_MODES_GENERAL".BA.BA2_SELECTED )
      wire#w2
      Contact( "DB1018_SAFETY_TAGS".ENABLE_DEVICE_FROM_UNIT_01_STATION_02_DOOR_AREA )
      wire#w3
      Contact( "DB1018_SAFETY_TAGS".POWER_ON_W_ENABLE_BUTT )
      wire#w4
      Coil( "DB1018_SAFETY_TAGS".GROUP_3_C12.SOS_Deactivate )
   END_RUNG
   RUNG wire#w1
      Contact( "DB2001_MODES_GENERAL".BA.BA3_SELECTED )
   END_RUNG wire#w2
   RUNG wire#w2
      Contact( "DB1018_SAFETY_TAGS".ENABLE_DEVICE_FROM_UNIT_01_MAIN_SAFETY_DOOR_AREA )
   END_RUNG wire#w3
   RUNG wire#w1
      Contact( "DB1018_SAFETY_TAGS".SAFE_DOORS_U01_CLOSED_AND_LOCKED )
      Contact( "DB2001_MODES_GENERAL".BA.BA1_SELECTED )
   END_RUNG wire#w4
   // the same network as SCL:
   "DB1018_SAFETY_TAGS".GROUP_3_C12.SOS_Deactivate := "DB1018_SAFETY_TAGS".E_STOP_OK_OFF_DEL_4 AND (((("DB2001_MODES_GENERAL".GENERAL.MANUAL_SELECTED AND "DB2001_MODES_GENERAL".BA.BA2_SELECTED) OR "DB2001_MODES_GENERAL".BA.BA3_SELECTED) AND ("DB1018_SAFETY_TAGS".ENABLE_DEVICE_FROM_UNIT_01_STATION_02_DOOR_AREA OR "DB1018_SAFETY_TAGS".ENABLE_DEVICE_FROM_UNIT_01_MAIN_SAFETY_DOOR_AREA) AND "DB1018_SAFETY_TAGS".POWER_ON_W_ENABLE_BUTT) OR ("DB1018_SAFETY_TAGS".SAFE_DOORS_U01_CLOSED_AND_LOCKED AND "DB2001_MODES_GENERAL".BA.BA1_SELECTED));
END_REGION

REGION Network 94: DESELECT SAFE OPERATING STOP
   RUNG wire#powerrail
      Contact( "DB1018_SAFETY_TAGS".GROUP_3_C12.SOS_Deactivate )
      Coil( "C12_SAFETY_OUT".Deselect_SOS )
   END_RUNG
   // the same network as SCL:
   "C12_SAFETY_OUT".Deselect_SOS := "DB1018_SAFETY_TAGS".GROUP_3_C12.SOS_Deactivate;
END_REGION

REGION Network 95: GROUP 3 SAFE LIMITED SPEED DEACTIVATE
   RUNG wire#powerrail
      Contact( "DB1018_SAFETY_TAGS".ALWAYS_OFF )
      Coil( "DB1018_SAFETY_TAGS".GROUP_3_C12.SLS_Deactivate )
   END_RUNG
   // the same network as SCL:
   "DB1018_SAFETY_TAGS".GROUP_3_C12.SLS_Deactivate := "DB1018_SAFETY_TAGS".ALWAYS_OFF;
END_REGION

REGION Network 96: DESELECT SAFE LIMITED SPEED
   RUNG wire#powerrail
      Contact( "DB1018_SAFETY_TAGS".GROUP_3_C12.SLS_Deactivate )
      Coil( "C12_SAFETY_OUT".Deselect_SLS )
   END_RUNG
   // the same network as SCL:
   "C12_SAFETY_OUT".Deselect_SLS := "DB1018_SAFETY_TAGS".GROUP_3_C12.SLS_Deactivate;
END_REGION

REGION Network 97: GROUP 3 SAFE LIMITED SPEED BIT 0
   // SLS0  SLS1
   //    0        0   BA1 DOOR OPEN
   //    1        0   BA2
   //    0        1   BA3 SEMICYCLE WITH LOAD DOOR OPEN
   //    1        1   ALL DOOR CLOSED
   RUNG wire#powerrail
      Contact( "DB1018_SAFETY_TAGS".SAFE_DOORS_U01_CLOSED_AND_LOCKED )
      wire#w1
      Coil( "DB1018_SAFETY_TAGS".GROUP_3_C12.SLS_BIT0 )
   END_RUNG
   RUNG wire#powerrail
      Contact( "DB2001_MODES_GENERAL".BA.BA2_SELECTED )
      Contact( "DB1018_SAFETY_TAGS".POWER_ON_W_ENABLE_BUTT )
   END_RUNG wire#w1
   // the same network as SCL:
   "DB1018_SAFETY_TAGS".GROUP_3_C12.SLS_BIT0 := "DB1018_SAFETY_TAGS".SAFE_DOORS_U01_CLOSED_AND_LOCKED OR ("DB2001_MODES_GENERAL".BA.BA2_SELECTED AND "DB1018_SAFETY_TAGS".POWER_ON_W_ENABLE_BUTT);
END_REGION

REGION Network 98: SELECT SAFE LIMITED SPEED BIT 0
   // SLS0  SLS1
   //    0        0   BA1 DOOR OPEN
   //    1        0   BA2
   //    0        1   BA3 SEMICYCLE WITH LOAD DOOR OPEN
   //    1        1   ALL DOOR CLOSED
   RUNG wire#powerrail
      Contact( "DB1018_SAFETY_TAGS".GROUP_3_C12.SLS_BIT0 )
      Coil( "C12_SAFETY_OUT".Select_SLS_bit_0 )
   END_RUNG
   // the same network as SCL:
   "C12_SAFETY_OUT".Select_SLS_bit_0 := "DB1018_SAFETY_TAGS".GROUP_3_C12.SLS_BIT0;
END_REGION

REGION Network 99: GROUP 3 SAFE LIMITED SPEED BIT 1
   // SLS0  SLS1
   //    0        0   BA1 DOOR OPEN
   //    1        0   BA2
   //    0        1   BA3 SEMICYCLE WITH LOAD DOOR OPEN
   //    1        1   ALL DOOR CLOSED
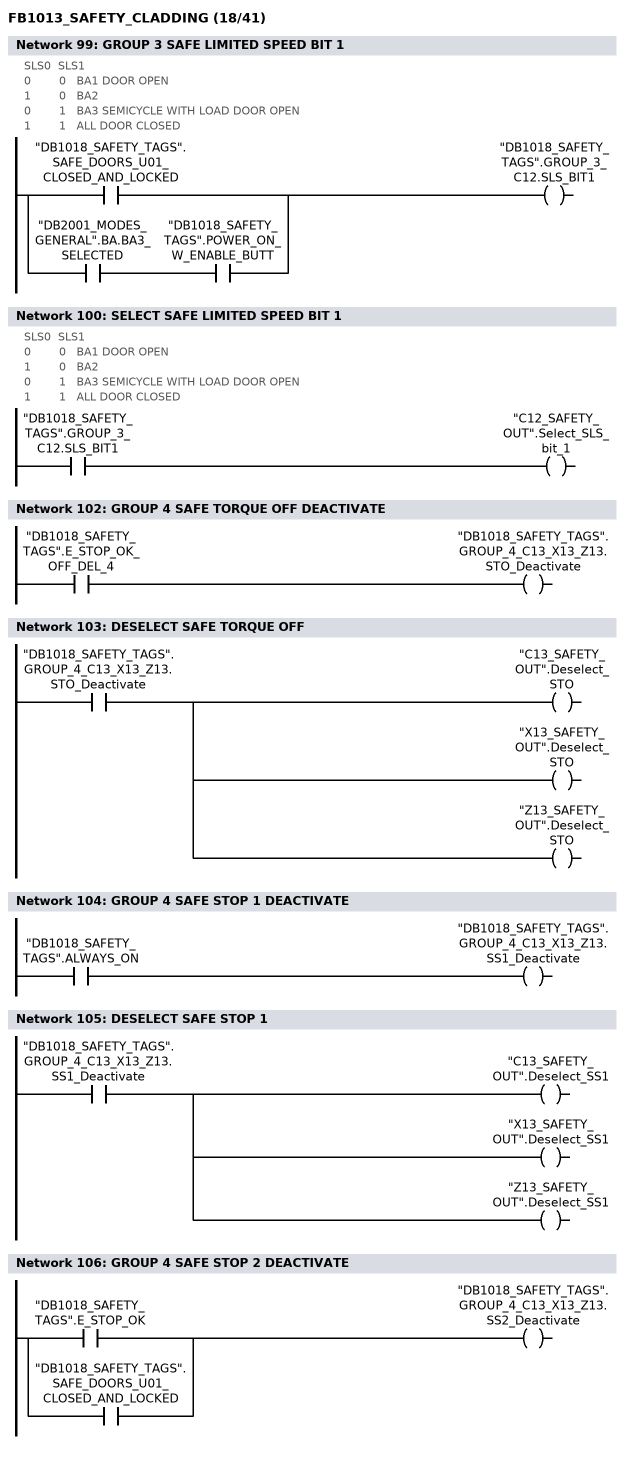
   RUNG wire#powerrail
      Contact( "DB1018_SAFETY_TAGS".SAFE_DOORS_U01_CLOSED_AND_LOCKED )
      wire#w1
      Coil( "DB1018_SAFETY_TAGS".GROUP_3_C12.SLS_BIT1 )
   END_RUNG
   RUNG wire#powerrail
      Contact( "DB2001_MODES_GENERAL".BA.BA3_SELECTED )
      Contact( "DB1018_SAFETY_TAGS".POWER_ON_W_ENABLE_BUTT )
   END_RUNG wire#w1
   // the same network as SCL:
   "DB1018_SAFETY_TAGS".GROUP_3_C12.SLS_BIT1 := "DB1018_SAFETY_TAGS".SAFE_DOORS_U01_CLOSED_AND_LOCKED OR ("DB2001_MODES_GENERAL".BA.BA3_SELECTED AND "DB1018_SAFETY_TAGS".POWER_ON_W_ENABLE_BUTT);
END_REGION

REGION Network 100: SELECT SAFE LIMITED SPEED BIT 1
   // SLS0  SLS1
   //    0        0   BA1 DOOR OPEN
   //    1        0   BA2
   //    0        1   BA3 SEMICYCLE WITH LOAD DOOR OPEN
   //    1        1   ALL DOOR CLOSED
   RUNG wire#powerrail
      Contact( "DB1018_SAFETY_TAGS".GROUP_3_C12.SLS_BIT1 )
      Coil( "C12_SAFETY_OUT".Select_SLS_bit_1 )
   END_RUNG
   // the same network as SCL:
   "C12_SAFETY_OUT".Select_SLS_bit_1 := "DB1018_SAFETY_TAGS".GROUP_3_C12.SLS_BIT1;
END_REGION

REGION Network 101: *************** GROUP 4 - C13 / X13 / Z13 ***************
END_REGION

REGION Network 102: GROUP 4 SAFE TORQUE OFF DEACTIVATE
   RUNG wire#powerrail
      Contact( "DB1018_SAFETY_TAGS".E_STOP_OK_OFF_DEL_4 )
      Coil( "DB1018_SAFETY_TAGS".GROUP_4_C13_X13_Z13.STO_Deactivate )
   END_RUNG
   // the same network as SCL:
   "DB1018_SAFETY_TAGS".GROUP_4_C13_X13_Z13.STO_Deactivate := "DB1018_SAFETY_TAGS".E_STOP_OK_OFF_DEL_4;
END_REGION

REGION Network 103: DESELECT SAFE TORQUE OFF
   RUNG wire#powerrail
      Contact( "DB1018_SAFETY_TAGS".GROUP_4_C13_X13_Z13.STO_Deactivate )
      wire#w1
      Coil( "C13_SAFETY_OUT".Deselect_STO )
   END_RUNG
   RUNG wire#w1
      Coil( "X13_SAFETY_OUT".Deselect_STO )
   END_RUNG
   RUNG wire#w1
      Coil( "Z13_SAFETY_OUT".Deselect_STO )
   END_RUNG
   // the same network as SCL:
   "C13_SAFETY_OUT".Deselect_STO := "DB1018_SAFETY_TAGS".GROUP_4_C13_X13_Z13.STO_Deactivate;
   "X13_SAFETY_OUT".Deselect_STO := "DB1018_SAFETY_TAGS".GROUP_4_C13_X13_Z13.STO_Deactivate;
   "Z13_SAFETY_OUT".Deselect_STO := "DB1018_SAFETY_TAGS".GROUP_4_C13_X13_Z13.STO_Deactivate;
END_REGION

REGION Network 104: GROUP 4 SAFE STOP 1 DEACTIVATE
   RUNG wire#powerrail
      Contact( "DB1018_SAFETY_TAGS".ALWAYS_ON )
      Coil( "DB1018_SAFETY_TAGS".GROUP_4_C13_X13_Z13.SS1_Deactivate )
   END_RUNG
   // the same network as SCL:
   "DB1018_SAFETY_TAGS".GROUP_4_C13_X13_Z13.SS1_Deactivate := "DB1018_SAFETY_TAGS".ALWAYS_ON;
END_REGION

REGION Network 105: DESELECT SAFE STOP 1
   RUNG wire#powerrail
      Contact( "DB1018_SAFETY_TAGS".GROUP_4_C13_X13_Z13.SS1_Deactivate )
      wire#w1
      Coil( "C13_SAFETY_OUT".Deselect_SS1 )
   END_RUNG
   RUNG wire#w1
      Coil( "X13_SAFETY_OUT".Deselect_SS1 )
   END_RUNG
   RUNG wire#w1
      Coil( "Z13_SAFETY_OUT".Deselect_SS1 )
   END_RUNG
   // the same network as SCL:
   "C13_SAFETY_OUT".Deselect_SS1 := "DB1018_SAFETY_TAGS".GROUP_4_C13_X13_Z13.SS1_Deactivate;
   "X13_SAFETY_OUT".Deselect_SS1 := "DB1018_SAFETY_TAGS".GROUP_4_C13_X13_Z13.SS1_Deactivate;
   "Z13_SAFETY_OUT".Deselect_SS1 := "DB1018_SAFETY_TAGS".GROUP_4_C13_X13_Z13.SS1_Deactivate;
END_REGION

REGION Network 106: GROUP 4 SAFE STOP 2 DEACTIVATE
   RUNG wire#powerrail
      Contact( "DB1018_SAFETY_TAGS".E_STOP_OK )
      wire#w1
      Coil( "DB1018_SAFETY_TAGS".GROUP_4_C13_X13_Z13.SS2_Deactivate )
   END_RUNG
   RUNG wire#powerrail
      Contact( "DB1018_SAFETY_TAGS".SAFE_DOORS_U01_CLOSED_AND_LOCKED )
   END_RUNG wire#w1
   // the same network as SCL:
   "DB1018_SAFETY_TAGS".GROUP_4_C13_X13_Z13.SS2_Deactivate := "DB1018_SAFETY_TAGS".E_STOP_OK OR "DB1018_SAFETY_TAGS".SAFE_DOORS_U01_CLOSED_AND_LOCKED;
END_REGION

REGION Network 107: DESELECT SAFE STOP 2
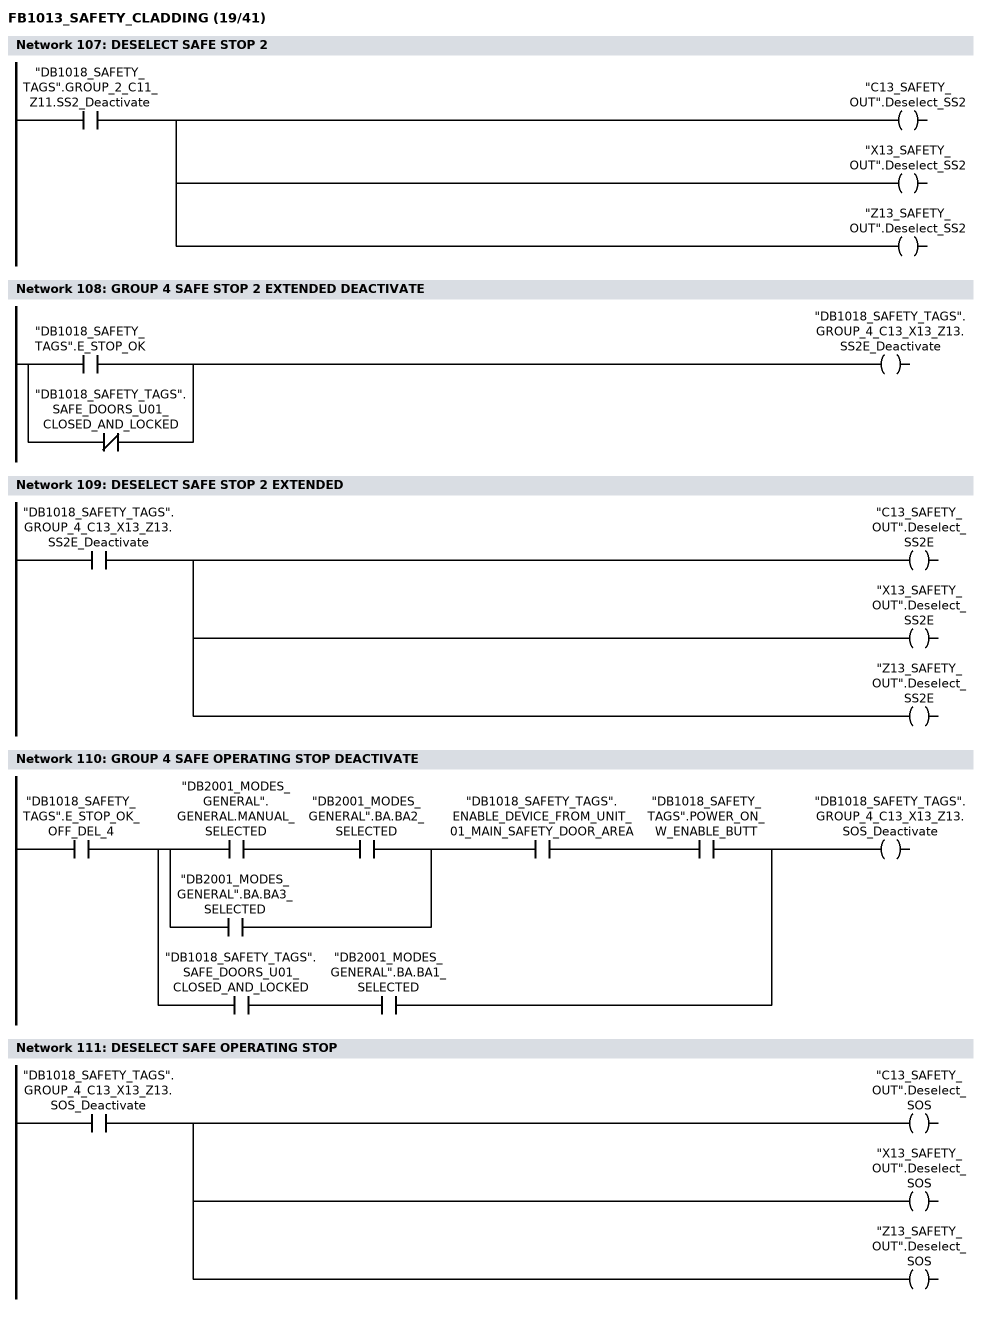
   RUNG wire#powerrail
      Contact( "DB1018_SAFETY_TAGS".GROUP_2_C11_Z11.SS2_Deactivate )
      wire#w1
      Coil( "C13_SAFETY_OUT".Deselect_SS2 )
   END_RUNG
   RUNG wire#w1
      Coil( "X13_SAFETY_OUT".Deselect_SS2 )
   END_RUNG
   RUNG wire#w1
      Coil( "Z13_SAFETY_OUT".Deselect_SS2 )
   END_RUNG
   // the same network as SCL:
   "C13_SAFETY_OUT".Deselect_SS2 := "DB1018_SAFETY_TAGS".GROUP_2_C11_Z11.SS2_Deactivate;
   "X13_SAFETY_OUT".Deselect_SS2 := "DB1018_SAFETY_TAGS".GROUP_2_C11_Z11.SS2_Deactivate;
   "Z13_SAFETY_OUT".Deselect_SS2 := "DB1018_SAFETY_TAGS".GROUP_2_C11_Z11.SS2_Deactivate;
END_REGION

REGION Network 108: GROUP 4 SAFE STOP 2 EXTENDED DEACTIVATE
   RUNG wire#powerrail
      Contact( "DB1018_SAFETY_TAGS".E_STOP_OK )
      wire#w1
      Coil( "DB1018_SAFETY_TAGS".GROUP_4_C13_X13_Z13.SS2E_Deactivate )
   END_RUNG
   RUNG wire#powerrail
      I_Contact( "DB1018_SAFETY_TAGS".SAFE_DOORS_U01_CLOSED_AND_LOCKED )
   END_RUNG wire#w1
   // the same network as SCL:
   "DB1018_SAFETY_TAGS".GROUP_4_C13_X13_Z13.SS2E_Deactivate := "DB1018_SAFETY_TAGS".E_STOP_OK OR NOT "DB1018_SAFETY_TAGS".SAFE_DOORS_U01_CLOSED_AND_LOCKED;
END_REGION

REGION Network 109: DESELECT SAFE STOP 2 EXTENDED
   RUNG wire#powerrail
      Contact( "DB1018_SAFETY_TAGS".GROUP_4_C13_X13_Z13.SS2E_Deactivate )
      wire#w1
      Coil( "C13_SAFETY_OUT".Deselect_SS2E )
   END_RUNG
   RUNG wire#w1
      Coil( "X13_SAFETY_OUT".Deselect_SS2E )
   END_RUNG
   RUNG wire#w1
      Coil( "Z13_SAFETY_OUT".Deselect_SS2E )
   END_RUNG
   // the same network as SCL:
   "C13_SAFETY_OUT".Deselect_SS2E := "DB1018_SAFETY_TAGS".GROUP_4_C13_X13_Z13.SS2E_Deactivate;
   "X13_SAFETY_OUT".Deselect_SS2E := "DB1018_SAFETY_TAGS".GROUP_4_C13_X13_Z13.SS2E_Deactivate;
   "Z13_SAFETY_OUT".Deselect_SS2E := "DB1018_SAFETY_TAGS".GROUP_4_C13_X13_Z13.SS2E_Deactivate;
END_REGION

REGION Network 110: GROUP 4 SAFE OPERATING STOP DEACTIVATE
   RUNG wire#powerrail
      Contact( "DB1018_SAFETY_TAGS".E_STOP_OK_OFF_DEL_4 )
      wire#w1
      Contact( "DB2001_MODES_GENERAL".GENERAL.MANUAL_SELECTED )
      Contact( "DB2001_MODES_GENERAL".BA.BA2_SELECTED )
      wire#w2
      Contact( "DB1018_SAFETY_TAGS".ENABLE_DEVICE_FROM_UNIT_01_MAIN_SAFETY_DOOR_AREA )
      Contact( "DB1018_SAFETY_TAGS".POWER_ON_W_ENABLE_BUTT )
      wire#w3
      Coil( "DB1018_SAFETY_TAGS".GROUP_4_C13_X13_Z13.SOS_Deactivate )
   END_RUNG
   RUNG wire#w1
      Contact( "DB2001_MODES_GENERAL".BA.BA3_SELECTED )
   END_RUNG wire#w2
   RUNG wire#w1
      Contact( "DB1018_SAFETY_TAGS".SAFE_DOORS_U01_CLOSED_AND_LOCKED )
      Contact( "DB2001_MODES_GENERAL".BA.BA1_SELECTED )
   END_RUNG wire#w3
   // the same network as SCL:
   "DB1018_SAFETY_TAGS".GROUP_4_C13_X13_Z13.SOS_Deactivate := "DB1018_SAFETY_TAGS".E_STOP_OK_OFF_DEL_4 AND (((("DB2001_MODES_GENERAL".GENERAL.MANUAL_SELECTED AND "DB2001_MODES_GENERAL".BA.BA2_SELECTED) OR "DB2001_MODES_GENERAL".BA.BA3_SELECTED) AND "DB1018_SAFETY_TAGS".ENABLE_DEVICE_FROM_UNIT_01_MAIN_SAFETY_DOOR_AREA AND "DB1018_SAFETY_TAGS".POWER_ON_W_ENABLE_BUTT) OR ("DB1018_SAFETY_TAGS".SAFE_DOORS_U01_CLOSED_AND_LOCKED AND "DB2001_MODES_GENERAL".BA.BA1_SELECTED));
END_REGION

REGION Network 111: DESELECT SAFE OPERATING STOP
   RUNG wire#powerrail
      Contact( "DB1018_SAFETY_TAGS".GROUP_4_C13_X13_Z13.SOS_Deactivate )
      wire#w1
      Coil( "C13_SAFETY_OUT".Deselect_SOS )
   END_RUNG
   RUNG wire#w1
      Coil( "X13_SAFETY_OUT".Deselect_SOS )
   END_RUNG
   RUNG wire#w1
      Coil( "Z13_SAFETY_OUT".Deselect_SOS )
   END_RUNG
   // the same network as SCL:
   "C13_SAFETY_OUT".Deselect_SOS := "DB1018_SAFETY_TAGS".GROUP_4_C13_X13_Z13.SOS_Deactivate;
   "X13_SAFETY_OUT".Deselect_SOS := "DB1018_SAFETY_TAGS".GROUP_4_C13_X13_Z13.SOS_Deactivate;
   "Z13_SAFETY_OUT".Deselect_SOS := "DB1018_SAFETY_TAGS".GROUP_4_C13_X13_Z13.SOS_Deactivate;
END_REGION

REGION Network 112: GROUP 4 SAFE LIMITED SPEED DEACTIVATE
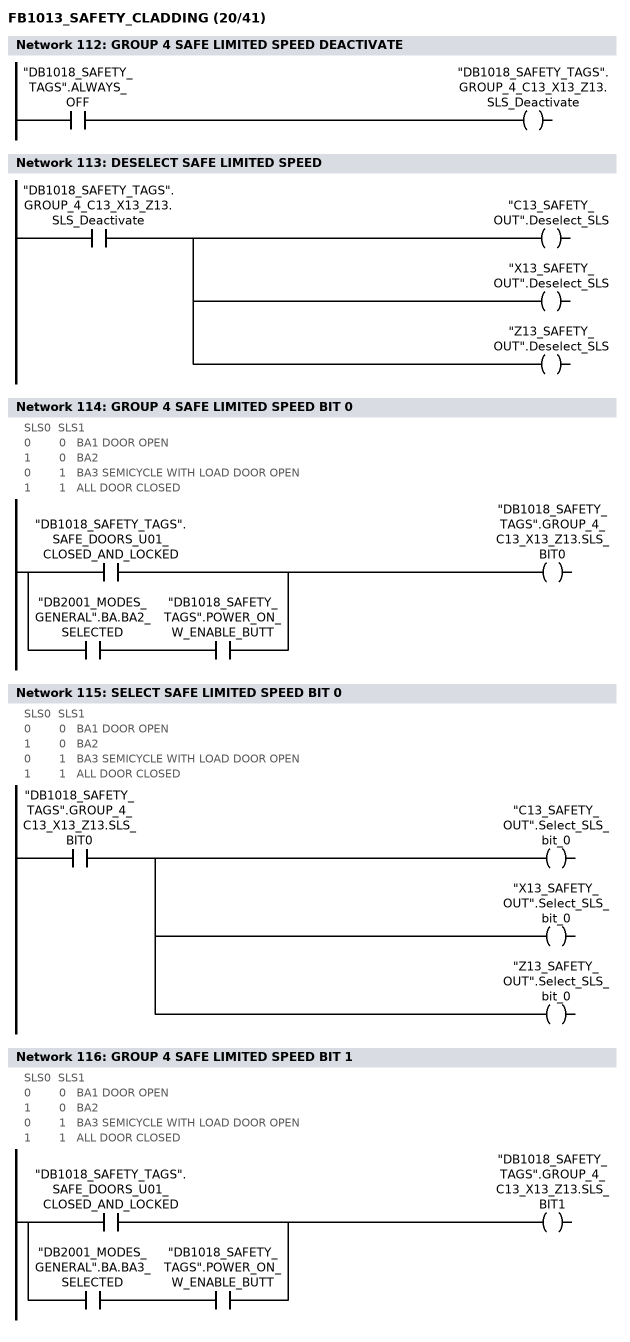
   RUNG wire#powerrail
      Contact( "DB1018_SAFETY_TAGS".ALWAYS_OFF )
      Coil( "DB1018_SAFETY_TAGS".GROUP_4_C13_X13_Z13.SLS_Deactivate )
   END_RUNG
   // the same network as SCL:
   "DB1018_SAFETY_TAGS".GROUP_4_C13_X13_Z13.SLS_Deactivate := "DB1018_SAFETY_TAGS".ALWAYS_OFF;
END_REGION

REGION Network 113: DESELECT SAFE LIMITED SPEED
   RUNG wire#powerrail
      Contact( "DB1018_SAFETY_TAGS".GROUP_4_C13_X13_Z13.SLS_Deactivate )
      wire#w1
      Coil( "C13_SAFETY_OUT".Deselect_SLS )
   END_RUNG
   RUNG wire#w1
      Coil( "X13_SAFETY_OUT".Deselect_SLS )
   END_RUNG
   RUNG wire#w1
      Coil( "Z13_SAFETY_OUT".Deselect_SLS )
   END_RUNG
   // the same network as SCL:
   "C13_SAFETY_OUT".Deselect_SLS := "DB1018_SAFETY_TAGS".GROUP_4_C13_X13_Z13.SLS_Deactivate;
   "X13_SAFETY_OUT".Deselect_SLS := "DB1018_SAFETY_TAGS".GROUP_4_C13_X13_Z13.SLS_Deactivate;
   "Z13_SAFETY_OUT".Deselect_SLS := "DB1018_SAFETY_TAGS".GROUP_4_C13_X13_Z13.SLS_Deactivate;
END_REGION

REGION Network 114: GROUP 4 SAFE LIMITED SPEED BIT 0
   // SLS0  SLS1
   //    0        0   BA1 DOOR OPEN
   //    1        0   BA2
   //    0        1   BA3 SEMICYCLE WITH LOAD DOOR OPEN
   //    1        1   ALL DOOR CLOSED
   RUNG wire#powerrail
      Contact( "DB1018_SAFETY_TAGS".SAFE_DOORS_U01_CLOSED_AND_LOCKED )
      wire#w1
      Coil( "DB1018_SAFETY_TAGS".GROUP_4_C13_X13_Z13.SLS_BIT0 )
   END_RUNG
   RUNG wire#powerrail
      Contact( "DB2001_MODES_GENERAL".BA.BA2_SELECTED )
      Contact( "DB1018_SAFETY_TAGS".POWER_ON_W_ENABLE_BUTT )
   END_RUNG wire#w1
   // the same network as SCL:
   "DB1018_SAFETY_TAGS".GROUP_4_C13_X13_Z13.SLS_BIT0 := "DB1018_SAFETY_TAGS".SAFE_DOORS_U01_CLOSED_AND_LOCKED OR ("DB2001_MODES_GENERAL".BA.BA2_SELECTED AND "DB1018_SAFETY_TAGS".POWER_ON_W_ENABLE_BUTT);
END_REGION

REGION Network 115: SELECT SAFE LIMITED SPEED BIT 0
   // SLS0  SLS1
   //    0        0   BA1 DOOR OPEN
   //    1        0   BA2
   //    0        1   BA3 SEMICYCLE WITH LOAD DOOR OPEN
   //    1        1   ALL DOOR CLOSED
   RUNG wire#powerrail
      Contact( "DB1018_SAFETY_TAGS".GROUP_4_C13_X13_Z13.SLS_BIT0 )
      wire#w1
      Coil( "C13_SAFETY_OUT".Select_SLS_bit_0 )
   END_RUNG
   RUNG wire#w1
      Coil( "X13_SAFETY_OUT".Select_SLS_bit_0 )
   END_RUNG
   RUNG wire#w1
      Coil( "Z13_SAFETY_OUT".Select_SLS_bit_0 )
   END_RUNG
   // the same network as SCL:
   "C13_SAFETY_OUT".Select_SLS_bit_0 := "DB1018_SAFETY_TAGS".GROUP_4_C13_X13_Z13.SLS_BIT0;
   "X13_SAFETY_OUT".Select_SLS_bit_0 := "DB1018_SAFETY_TAGS".GROUP_4_C13_X13_Z13.SLS_BIT0;
   "Z13_SAFETY_OUT".Select_SLS_bit_0 := "DB1018_SAFETY_TAGS".GROUP_4_C13_X13_Z13.SLS_BIT0;
END_REGION

REGION Network 116: GROUP 4 SAFE LIMITED SPEED BIT 1
   // SLS0  SLS1
   //    0        0   BA1 DOOR OPEN
   //    1        0   BA2
   //    0        1   BA3 SEMICYCLE WITH LOAD DOOR OPEN
   //    1        1   ALL DOOR CLOSED
   RUNG wire#powerrail
      Contact( "DB1018_SAFETY_TAGS".SAFE_DOORS_U01_CLOSED_AND_LOCKED )
      wire#w1
      Coil( "DB1018_SAFETY_TAGS".GROUP_4_C13_X13_Z13.SLS_BIT1 )
   END_RUNG
   RUNG wire#powerrail
      Contact( "DB2001_MODES_GENERAL".BA.BA3_SELECTED )
      Contact( "DB1018_SAFETY_TAGS".POWER_ON_W_ENABLE_BUTT )
   END_RUNG wire#w1
   // the same network as SCL:
   "DB1018_SAFETY_TAGS".GROUP_4_C13_X13_Z13.SLS_BIT1 := "DB1018_SAFETY_TAGS".SAFE_DOORS_U01_CLOSED_AND_LOCKED OR ("DB2001_MODES_GENERAL".BA.BA3_SELECTED AND "DB1018_SAFETY_TAGS".POWER_ON_W_ENABLE_BUTT);
END_REGION

REGION Network 117: SELECT SAFE LIMITED SPEED BIT 1
   // SLS0  SLS1
   //    0        0   BA1 DOOR OPEN
   //    1        0   BA2
   //    0        1   BA3 SEMICYCLE WITH LOAD DOOR OPEN
   //    1        1   ALL DOOR CLOSED
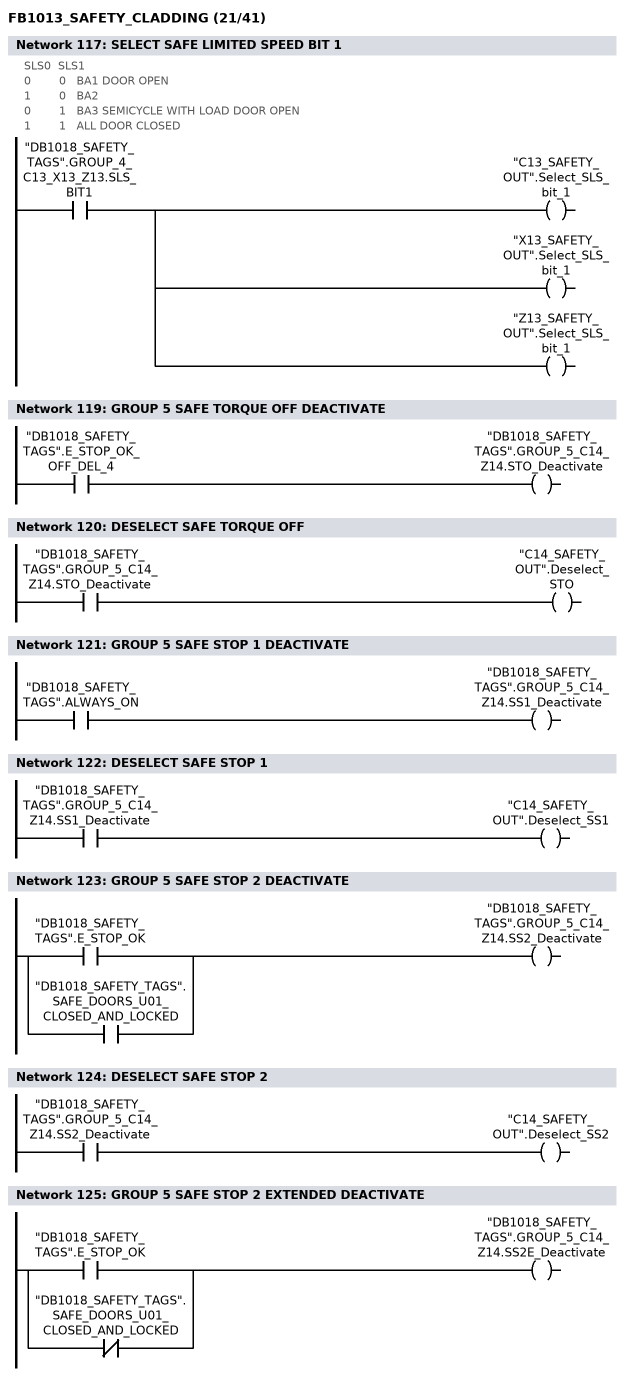
   RUNG wire#powerrail
      Contact( "DB1018_SAFETY_TAGS".GROUP_4_C13_X13_Z13.SLS_BIT1 )
      wire#w1
      Coil( "C13_SAFETY_OUT".Select_SLS_bit_1 )
   END_RUNG
   RUNG wire#w1
      Coil( "X13_SAFETY_OUT".Select_SLS_bit_1 )
   END_RUNG
   RUNG wire#w1
      Coil( "Z13_SAFETY_OUT".Select_SLS_bit_1 )
   END_RUNG
   // the same network as SCL:
   "C13_SAFETY_OUT".Select_SLS_bit_1 := "DB1018_SAFETY_TAGS".GROUP_4_C13_X13_Z13.SLS_BIT1;
   "X13_SAFETY_OUT".Select_SLS_bit_1 := "DB1018_SAFETY_TAGS".GROUP_4_C13_X13_Z13.SLS_BIT1;
   "Z13_SAFETY_OUT".Select_SLS_bit_1 := "DB1018_SAFETY_TAGS".GROUP_4_C13_X13_Z13.SLS_BIT1;
END_REGION

REGION Network 118: *************** GROUP 5 - C14 ***************
END_REGION

REGION Network 119: GROUP 5 SAFE TORQUE OFF DEACTIVATE
   RUNG wire#powerrail
      Contact( "DB1018_SAFETY_TAGS".E_STOP_OK_OFF_DEL_4 )
      Coil( "DB1018_SAFETY_TAGS".GROUP_5_C14_Z14.STO_Deactivate )
   END_RUNG
   // the same network as SCL:
   "DB1018_SAFETY_TAGS".GROUP_5_C14_Z14.STO_Deactivate := "DB1018_SAFETY_TAGS".E_STOP_OK_OFF_DEL_4;
END_REGION

REGION Network 120: DESELECT SAFE TORQUE OFF
   RUNG wire#powerrail
      Contact( "DB1018_SAFETY_TAGS".GROUP_5_C14_Z14.STO_Deactivate )
      Coil( "C14_SAFETY_OUT".Deselect_STO )
   END_RUNG
   // the same network as SCL:
   "C14_SAFETY_OUT".Deselect_STO := "DB1018_SAFETY_TAGS".GROUP_5_C14_Z14.STO_Deactivate;
END_REGION

REGION Network 121: GROUP 5 SAFE STOP 1 DEACTIVATE
   RUNG wire#powerrail
      Contact( "DB1018_SAFETY_TAGS".ALWAYS_ON )
      Coil( "DB1018_SAFETY_TAGS".GROUP_5_C14_Z14.SS1_Deactivate )
   END_RUNG
   // the same network as SCL:
   "DB1018_SAFETY_TAGS".GROUP_5_C14_Z14.SS1_Deactivate := "DB1018_SAFETY_TAGS".ALWAYS_ON;
END_REGION

REGION Network 122: DESELECT SAFE STOP 1
   RUNG wire#powerrail
      Contact( "DB1018_SAFETY_TAGS".GROUP_5_C14_Z14.SS1_Deactivate )
      Coil( "C14_SAFETY_OUT".Deselect_SS1 )
   END_RUNG
   // the same network as SCL:
   "C14_SAFETY_OUT".Deselect_SS1 := "DB1018_SAFETY_TAGS".GROUP_5_C14_Z14.SS1_Deactivate;
END_REGION

REGION Network 123: GROUP 5 SAFE STOP 2 DEACTIVATE
   RUNG wire#powerrail
      Contact( "DB1018_SAFETY_TAGS".E_STOP_OK )
      wire#w1
      Coil( "DB1018_SAFETY_TAGS".GROUP_5_C14_Z14.SS2_Deactivate )
   END_RUNG
   RUNG wire#powerrail
      Contact( "DB1018_SAFETY_TAGS".SAFE_DOORS_U01_CLOSED_AND_LOCKED )
   END_RUNG wire#w1
   // the same network as SCL:
   "DB1018_SAFETY_TAGS".GROUP_5_C14_Z14.SS2_Deactivate := "DB1018_SAFETY_TAGS".E_STOP_OK OR "DB1018_SAFETY_TAGS".SAFE_DOORS_U01_CLOSED_AND_LOCKED;
END_REGION

REGION Network 124: DESELECT SAFE STOP 2
   RUNG wire#powerrail
      Contact( "DB1018_SAFETY_TAGS".GROUP_5_C14_Z14.SS2_Deactivate )
      Coil( "C14_SAFETY_OUT".Deselect_SS2 )
   END_RUNG
   // the same network as SCL:
   "C14_SAFETY_OUT".Deselect_SS2 := "DB1018_SAFETY_TAGS".GROUP_5_C14_Z14.SS2_Deactivate;
END_REGION

REGION Network 125: GROUP 5 SAFE STOP 2 EXTENDED DEACTIVATE
   RUNG wire#powerrail
      Contact( "DB1018_SAFETY_TAGS".E_STOP_OK )
      wire#w1
      Coil( "DB1018_SAFETY_TAGS".GROUP_5_C14_Z14.SS2E_Deactivate )
   END_RUNG
   RUNG wire#powerrail
      I_Contact( "DB1018_SAFETY_TAGS".SAFE_DOORS_U01_CLOSED_AND_LOCKED )
   END_RUNG wire#w1
   // the same network as SCL:
   "DB1018_SAFETY_TAGS".GROUP_5_C14_Z14.SS2E_Deactivate := "DB1018_SAFETY_TAGS".E_STOP_OK OR NOT "DB1018_SAFETY_TAGS".SAFE_DOORS_U01_CLOSED_AND_LOCKED;
END_REGION

REGION Network 126: DESELECT SAFE STOP 2 EXTENDED
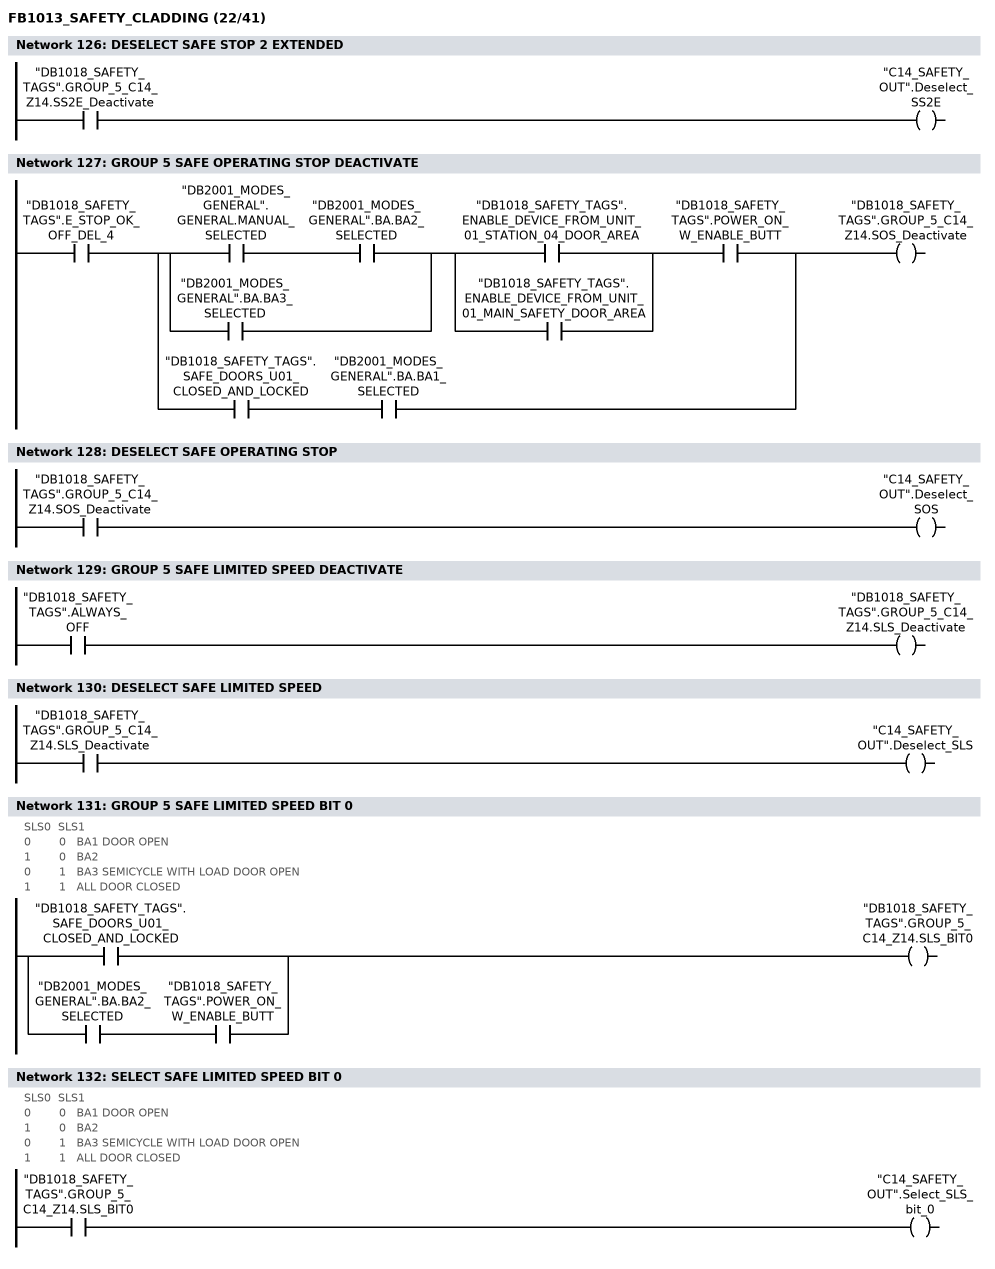
   RUNG wire#powerrail
      Contact( "DB1018_SAFETY_TAGS".GROUP_5_C14_Z14.SS2E_Deactivate )
      Coil( "C14_SAFETY_OUT".Deselect_SS2E )
   END_RUNG
   // the same network as SCL:
   "C14_SAFETY_OUT".Deselect_SS2E := "DB1018_SAFETY_TAGS".GROUP_5_C14_Z14.SS2E_Deactivate;
END_REGION

REGION Network 127: GROUP 5 SAFE OPERATING STOP DEACTIVATE
   RUNG wire#powerrail
      Contact( "DB1018_SAFETY_TAGS".E_STOP_OK_OFF_DEL_4 )
      wire#w1
      Contact( "DB2001_MODES_GENERAL".GENERAL.MANUAL_SELECTED )
      Contact( "DB2001_MODES_GENERAL".BA.BA2_SELECTED )
      wire#w2
      Contact( "DB1018_SAFETY_TAGS".ENABLE_DEVICE_FROM_UNIT_01_STATION_04_DOOR_AREA )
      wire#w3
      Contact( "DB1018_SAFETY_TAGS".POWER_ON_W_ENABLE_BUTT )
      wire#w4
      Coil( "DB1018_SAFETY_TAGS".GROUP_5_C14_Z14.SOS_Deactivate )
   END_RUNG
   RUNG wire#w1
      Contact( "DB2001_MODES_GENERAL".BA.BA3_SELECTED )
   END_RUNG wire#w2
   RUNG wire#w2
      Contact( "DB1018_SAFETY_TAGS".ENABLE_DEVICE_FROM_UNIT_01_MAIN_SAFETY_DOOR_AREA )
   END_RUNG wire#w3
   RUNG wire#w1
      Contact( "DB1018_SAFETY_TAGS".SAFE_DOORS_U01_CLOSED_AND_LOCKED )
      Contact( "DB2001_MODES_GENERAL".BA.BA1_SELECTED )
   END_RUNG wire#w4
   // the same network as SCL:
   "DB1018_SAFETY_TAGS".GROUP_5_C14_Z14.SOS_Deactivate := "DB1018_SAFETY_TAGS".E_STOP_OK_OFF_DEL_4 AND (((("DB2001_MODES_GENERAL".GENERAL.MANUAL_SELECTED AND "DB2001_MODES_GENERAL".BA.BA2_SELECTED) OR "DB2001_MODES_GENERAL".BA.BA3_SELECTED) AND ("DB1018_SAFETY_TAGS".ENABLE_DEVICE_FROM_UNIT_01_STATION_04_DOOR_AREA OR "DB1018_SAFETY_TAGS".ENABLE_DEVICE_FROM_UNIT_01_MAIN_SAFETY_DOOR_AREA) AND "DB1018_SAFETY_TAGS".POWER_ON_W_ENABLE_BUTT) OR ("DB1018_SAFETY_TAGS".SAFE_DOORS_U01_CLOSED_AND_LOCKED AND "DB2001_MODES_GENERAL".BA.BA1_SELECTED));
END_REGION

REGION Network 128: DESELECT SAFE OPERATING STOP
   RUNG wire#powerrail
      Contact( "DB1018_SAFETY_TAGS".GROUP_5_C14_Z14.SOS_Deactivate )
      Coil( "C14_SAFETY_OUT".Deselect_SOS )
   END_RUNG
   // the same network as SCL:
   "C14_SAFETY_OUT".Deselect_SOS := "DB1018_SAFETY_TAGS".GROUP_5_C14_Z14.SOS_Deactivate;
END_REGION

REGION Network 129: GROUP 5 SAFE LIMITED SPEED DEACTIVATE
   RUNG wire#powerrail
      Contact( "DB1018_SAFETY_TAGS".ALWAYS_OFF )
      Coil( "DB1018_SAFETY_TAGS".GROUP_5_C14_Z14.SLS_Deactivate )
   END_RUNG
   // the same network as SCL:
   "DB1018_SAFETY_TAGS".GROUP_5_C14_Z14.SLS_Deactivate := "DB1018_SAFETY_TAGS".ALWAYS_OFF;
END_REGION

REGION Network 130: DESELECT SAFE LIMITED SPEED
   RUNG wire#powerrail
      Contact( "DB1018_SAFETY_TAGS".GROUP_5_C14_Z14.SLS_Deactivate )
      Coil( "C14_SAFETY_OUT".Deselect_SLS )
   END_RUNG
   // the same network as SCL:
   "C14_SAFETY_OUT".Deselect_SLS := "DB1018_SAFETY_TAGS".GROUP_5_C14_Z14.SLS_Deactivate;
END_REGION

REGION Network 131: GROUP 5 SAFE LIMITED SPEED BIT 0
   // SLS0  SLS1
   //    0        0   BA1 DOOR OPEN
   //    1        0   BA2
   //    0        1   BA3 SEMICYCLE WITH LOAD DOOR OPEN
   //    1        1   ALL DOOR CLOSED
   RUNG wire#powerrail
      Contact( "DB1018_SAFETY_TAGS".SAFE_DOORS_U01_CLOSED_AND_LOCKED )
      wire#w1
      Coil( "DB1018_SAFETY_TAGS".GROUP_5_C14_Z14.SLS_BIT0 )
   END_RUNG
   RUNG wire#powerrail
      Contact( "DB2001_MODES_GENERAL".BA.BA2_SELECTED )
      Contact( "DB1018_SAFETY_TAGS".POWER_ON_W_ENABLE_BUTT )
   END_RUNG wire#w1
   // the same network as SCL:
   "DB1018_SAFETY_TAGS".GROUP_5_C14_Z14.SLS_BIT0 := "DB1018_SAFETY_TAGS".SAFE_DOORS_U01_CLOSED_AND_LOCKED OR ("DB2001_MODES_GENERAL".BA.BA2_SELECTED AND "DB1018_SAFETY_TAGS".POWER_ON_W_ENABLE_BUTT);
END_REGION

REGION Network 132: SELECT SAFE LIMITED SPEED BIT 0
   // SLS0  SLS1
   //    0        0   BA1 DOOR OPEN
   //    1        0   BA2
   //    0        1   BA3 SEMICYCLE WITH LOAD DOOR OPEN
   //    1        1   ALL DOOR CLOSED
   RUNG wire#powerrail
      Contact( "DB1018_SAFETY_TAGS".GROUP_5_C14_Z14.SLS_BIT0 )
      Coil( "C14_SAFETY_OUT".Select_SLS_bit_0 )
   END_RUNG
   // the same network as SCL:
   "C14_SAFETY_OUT".Select_SLS_bit_0 := "DB1018_SAFETY_TAGS".GROUP_5_C14_Z14.SLS_BIT0;
END_REGION

REGION Network 133: GROUP 5 SAFE LIMITED SPEED BIT 1
   // SLS0  SLS1
   //    0        0   BA1 DOOR OPEN
   //    1        0   BA2
   //    0        1   BA3 SEMICYCLE WITH LOAD DOOR OPEN
   //    1        1   ALL DOOR CLOSED
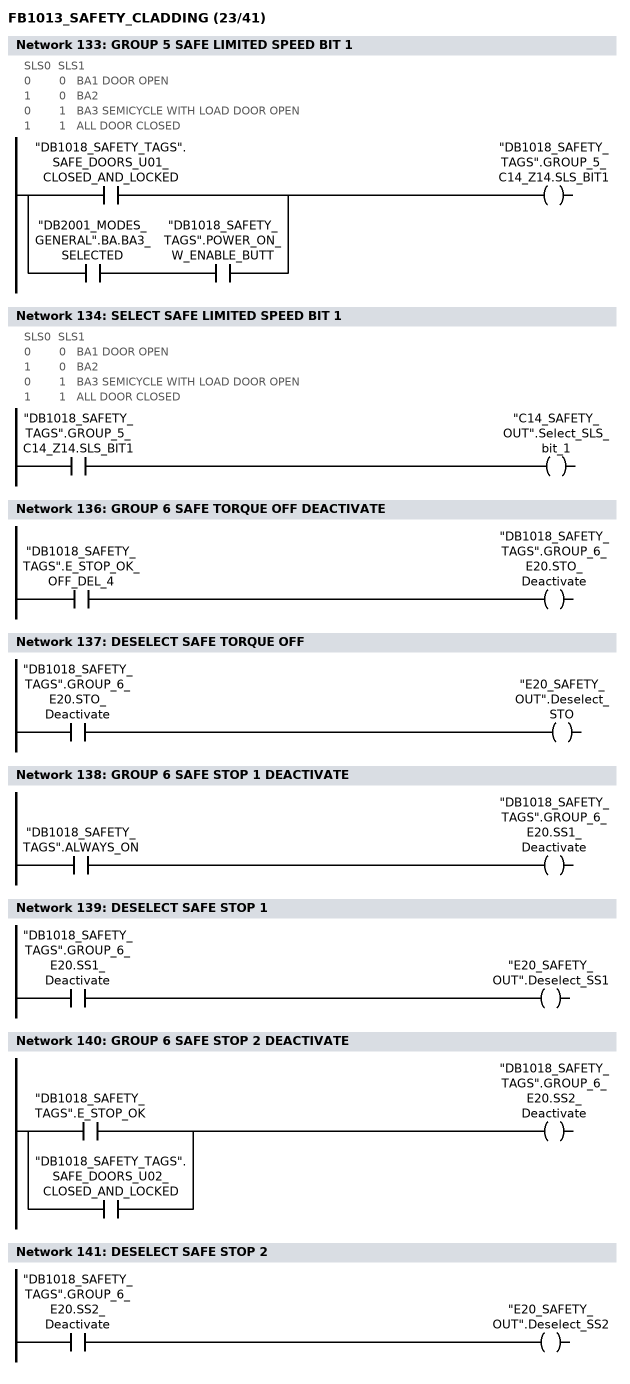
   RUNG wire#powerrail
      Contact( "DB1018_SAFETY_TAGS".SAFE_DOORS_U01_CLOSED_AND_LOCKED )
      wire#w1
      Coil( "DB1018_SAFETY_TAGS".GROUP_5_C14_Z14.SLS_BIT1 )
   END_RUNG
   RUNG wire#powerrail
      Contact( "DB2001_MODES_GENERAL".BA.BA3_SELECTED )
      Contact( "DB1018_SAFETY_TAGS".POWER_ON_W_ENABLE_BUTT )
   END_RUNG wire#w1
   // the same network as SCL:
   "DB1018_SAFETY_TAGS".GROUP_5_C14_Z14.SLS_BIT1 := "DB1018_SAFETY_TAGS".SAFE_DOORS_U01_CLOSED_AND_LOCKED OR ("DB2001_MODES_GENERAL".BA.BA3_SELECTED AND "DB1018_SAFETY_TAGS".POWER_ON_W_ENABLE_BUTT);
END_REGION

REGION Network 134: SELECT SAFE LIMITED SPEED BIT 1
   // SLS0  SLS1
   //    0        0   BA1 DOOR OPEN
   //    1        0   BA2
   //    0        1   BA3 SEMICYCLE WITH LOAD DOOR OPEN
   //    1        1   ALL DOOR CLOSED
   RUNG wire#powerrail
      Contact( "DB1018_SAFETY_TAGS".GROUP_5_C14_Z14.SLS_BIT1 )
      Coil( "C14_SAFETY_OUT".Select_SLS_bit_1 )
   END_RUNG
   // the same network as SCL:
   "C14_SAFETY_OUT".Select_SLS_bit_1 := "DB1018_SAFETY_TAGS".GROUP_5_C14_Z14.SLS_BIT1;
END_REGION

REGION Network 135: *************** GROUP 6 - E20 ***************
END_REGION

REGION Network 136: GROUP 6 SAFE TORQUE OFF DEACTIVATE
   RUNG wire#powerrail
      Contact( "DB1018_SAFETY_TAGS".E_STOP_OK_OFF_DEL_4 )
      Coil( "DB1018_SAFETY_TAGS".GROUP_6_E20.STO_Deactivate )
   END_RUNG
   // the same network as SCL:
   "DB1018_SAFETY_TAGS".GROUP_6_E20.STO_Deactivate := "DB1018_SAFETY_TAGS".E_STOP_OK_OFF_DEL_4;
END_REGION

REGION Network 137: DESELECT SAFE TORQUE OFF
   RUNG wire#powerrail
      Contact( "DB1018_SAFETY_TAGS".GROUP_6_E20.STO_Deactivate )
      Coil( "E20_SAFETY_OUT".Deselect_STO )
   END_RUNG
   // the same network as SCL:
   "E20_SAFETY_OUT".Deselect_STO := "DB1018_SAFETY_TAGS".GROUP_6_E20.STO_Deactivate;
END_REGION

